// TIA Portal V17 export
// export: Created 2025-03-07T09:17:32.1063252Z, ExportSetting WithDefaults, DisplayName Totally Integrated Automation Portal, DisplayVersion V17 Update 8, DisplayName TIA Portal Openness, DisplayVersion V17 Update 8, DisplayName TIA Portal Version Control Interface, DisplayVersion V17, DisplayName SINAMICS Startdrive Advanced, DisplayVersion V17 SP2, DisplayName SINAMICS Startdrive G110M, G120, G120C, G120D, G120P, G115D, DisplayVersion V17 SP2, DisplayName SINAMICS Startdrive G130, G150, S120, S150, SINAMICS MV, S210, DisplayVersion V17 SP2, DisplayName STEP 7 Professional, DisplayVersion V17 Update 8, DisplayName SINUMERIK ONE STEP 7 Toolbox, DisplayVersion V17 Update 12, DisplayName SINUMERIK 840D sl STEP 7 Toolbox, DisplayVersion V17 Update 12, DisplayName STEP 7 Safety, DisplayVersion V17 Update 6, DisplayName WinCC Advanced, DisplayVersion V17 Update 8
FUNCTION "FC372_NCK_M_CH9_SPARE" : Void   // FC372, LAD
TITLE = Channel 1 data
{ S7_Optimized_Access := 'FALSE' }
AUTHOR : ETXETAR
VERSION : 1.0
// stored: AutoNumber false, IsIECCheckEnabled false, SetENOAutomatically false, UDAEnableTagReadback false
BEGIN

REGION Network 1: ACKNOWLEDGE M400-FIXTURE 1 CLAMP SEQUENCE (READ-IN DISABLE) / ACKNOWLEDGE M100-CLAMP SEQUENCE FIXTURE 1
   // NOTE: WHEN THERE IS NOT INDEXING TABLE AVAILABLE IN THE MACHINE DELETE 
   // DB2171.DBX5.0 AND DB2171.DBX2.0
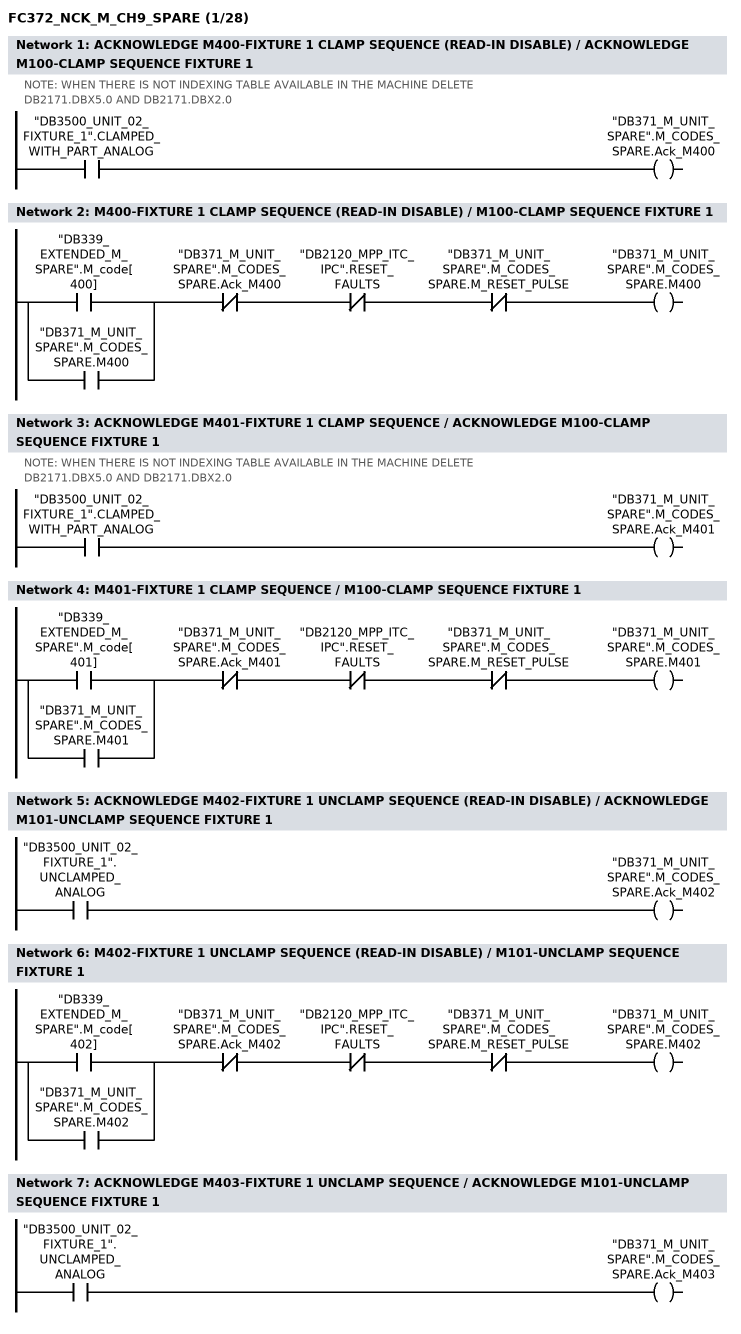
   RUNG wire#powerrail
      Contact( "DB3500_UNIT_02_FIXTURE_1".CLAMPED_WITH_PART_ANALOG )
      Coil( "DB371_M_UNIT_SPARE".M_CODES_SPARE.Ack_M400 )
   END_RUNG
   // the same network as SCL:
   "DB371_M_UNIT_SPARE".M_CODES_SPARE.Ack_M400 := "DB3500_UNIT_02_FIXTURE_1".CLAMPED_WITH_PART_ANALOG;
END_REGION

REGION Network 2: M400-FIXTURE 1 CLAMP SEQUENCE (READ-IN DISABLE) / M100-CLAMP SEQUENCE FIXTURE 1
   RUNG wire#powerrail
      Contact( "DB339_EXTENDED_M_SPARE".M_code[400] )
      wire#w1
      I_Contact( "DB371_M_UNIT_SPARE".M_CODES_SPARE.Ack_M400 )
      I_Contact( "DB2120_MPP_ITC_IPC".RESET_FAULTS )
      I_Contact( "DB371_M_UNIT_SPARE".M_CODES_SPARE.M_RESET_PULSE )
      Coil( "DB371_M_UNIT_SPARE".M_CODES_SPARE.M400 )
   END_RUNG
   RUNG wire#powerrail
      Contact( "DB371_M_UNIT_SPARE".M_CODES_SPARE.M400 )
   END_RUNG wire#w1
   // the same network as SCL:
   "DB371_M_UNIT_SPARE".M_CODES_SPARE.M400 := ("DB339_EXTENDED_M_SPARE".M_code[400] OR "DB371_M_UNIT_SPARE".M_CODES_SPARE.M400) AND NOT "DB371_M_UNIT_SPARE".M_CODES_SPARE.Ack_M400 AND NOT "DB2120_MPP_ITC_IPC".RESET_FAULTS AND NOT "DB371_M_UNIT_SPARE".M_CODES_SPARE.M_RESET_PULSE;
END_REGION

REGION Network 3: ACKNOWLEDGE M401-FIXTURE 1 CLAMP SEQUENCE / ACKNOWLEDGE M100-CLAMP SEQUENCE FIXTURE 1
   // NOTE: WHEN THERE IS NOT INDEXING TABLE AVAILABLE IN THE MACHINE DELETE 
   // DB2171.DBX5.0 AND DB2171.DBX2.0
   RUNG wire#powerrail
      Contact( "DB3500_UNIT_02_FIXTURE_1".CLAMPED_WITH_PART_ANALOG )
      Coil( "DB371_M_UNIT_SPARE".M_CODES_SPARE.Ack_M401 )
   END_RUNG
   // the same network as SCL:
   "DB371_M_UNIT_SPARE".M_CODES_SPARE.Ack_M401 := "DB3500_UNIT_02_FIXTURE_1".CLAMPED_WITH_PART_ANALOG;
END_REGION

REGION Network 4: M401-FIXTURE 1 CLAMP SEQUENCE / M100-CLAMP SEQUENCE FIXTURE 1
   RUNG wire#powerrail
      Contact( "DB339_EXTENDED_M_SPARE".M_code[401] )
      wire#w1
      I_Contact( "DB371_M_UNIT_SPARE".M_CODES_SPARE.Ack_M401 )
      I_Contact( "DB2120_MPP_ITC_IPC".RESET_FAULTS )
      I_Contact( "DB371_M_UNIT_SPARE".M_CODES_SPARE.M_RESET_PULSE )
      Coil( "DB371_M_UNIT_SPARE".M_CODES_SPARE.M401 )
   END_RUNG
   RUNG wire#powerrail
      Contact( "DB371_M_UNIT_SPARE".M_CODES_SPARE.M401 )
   END_RUNG wire#w1
   // the same network as SCL:
   "DB371_M_UNIT_SPARE".M_CODES_SPARE.M401 := ("DB339_EXTENDED_M_SPARE".M_code[401] OR "DB371_M_UNIT_SPARE".M_CODES_SPARE.M401) AND NOT "DB371_M_UNIT_SPARE".M_CODES_SPARE.Ack_M401 AND NOT "DB2120_MPP_ITC_IPC".RESET_FAULTS AND NOT "DB371_M_UNIT_SPARE".M_CODES_SPARE.M_RESET_PULSE;
END_REGION

REGION Network 5: ACKNOWLEDGE M402-FIXTURE 1 UNCLAMP SEQUENCE (READ-IN DISABLE) / ACKNOWLEDGE M101-UNCLAMP SEQUENCE FIXTURE 1
   RUNG wire#powerrail
      Contact( "DB3500_UNIT_02_FIXTURE_1".UNCLAMPED_ANALOG )
      Coil( "DB371_M_UNIT_SPARE".M_CODES_SPARE.Ack_M402 )
   END_RUNG
   // the same network as SCL:
   "DB371_M_UNIT_SPARE".M_CODES_SPARE.Ack_M402 := "DB3500_UNIT_02_FIXTURE_1".UNCLAMPED_ANALOG;
END_REGION

REGION Network 6: M402-FIXTURE 1 UNCLAMP SEQUENCE (READ-IN DISABLE) / M101-UNCLAMP SEQUENCE FIXTURE 1
   RUNG wire#powerrail
      Contact( "DB339_EXTENDED_M_SPARE".M_code[402] )
      wire#w1
      I_Contact( "DB371_M_UNIT_SPARE".M_CODES_SPARE.Ack_M402 )
      I_Contact( "DB2120_MPP_ITC_IPC".RESET_FAULTS )
      I_Contact( "DB371_M_UNIT_SPARE".M_CODES_SPARE.M_RESET_PULSE )
      Coil( "DB371_M_UNIT_SPARE".M_CODES_SPARE.M402 )
   END_RUNG
   RUNG wire#powerrail
      Contact( "DB371_M_UNIT_SPARE".M_CODES_SPARE.M402 )
   END_RUNG wire#w1
   // the same network as SCL:
   "DB371_M_UNIT_SPARE".M_CODES_SPARE.M402 := ("DB339_EXTENDED_M_SPARE".M_code[402] OR "DB371_M_UNIT_SPARE".M_CODES_SPARE.M402) AND NOT "DB371_M_UNIT_SPARE".M_CODES_SPARE.Ack_M402 AND NOT "DB2120_MPP_ITC_IPC".RESET_FAULTS AND NOT "DB371_M_UNIT_SPARE".M_CODES_SPARE.M_RESET_PULSE;
END_REGION

REGION Network 7: ACKNOWLEDGE M403-FIXTURE 1 UNCLAMP SEQUENCE / ACKNOWLEDGE M101-UNCLAMP SEQUENCE FIXTURE 1
   RUNG wire#powerrail
      Contact( "DB3500_UNIT_02_FIXTURE_1".UNCLAMPED_ANALOG )
      Coil( "DB371_M_UNIT_SPARE".M_CODES_SPARE.Ack_M403 )
   END_RUNG
   // the same network as SCL:
   "DB371_M_UNIT_SPARE".M_CODES_SPARE.Ack_M403 := "DB3500_UNIT_02_FIXTURE_1".UNCLAMPED_ANALOG;
END_REGION

REGION Network 8: M403-FIXTURE 1 UNCLAMP SEQUENCE / M101-UNCLAMP SEQUENCE FIXTURE 1
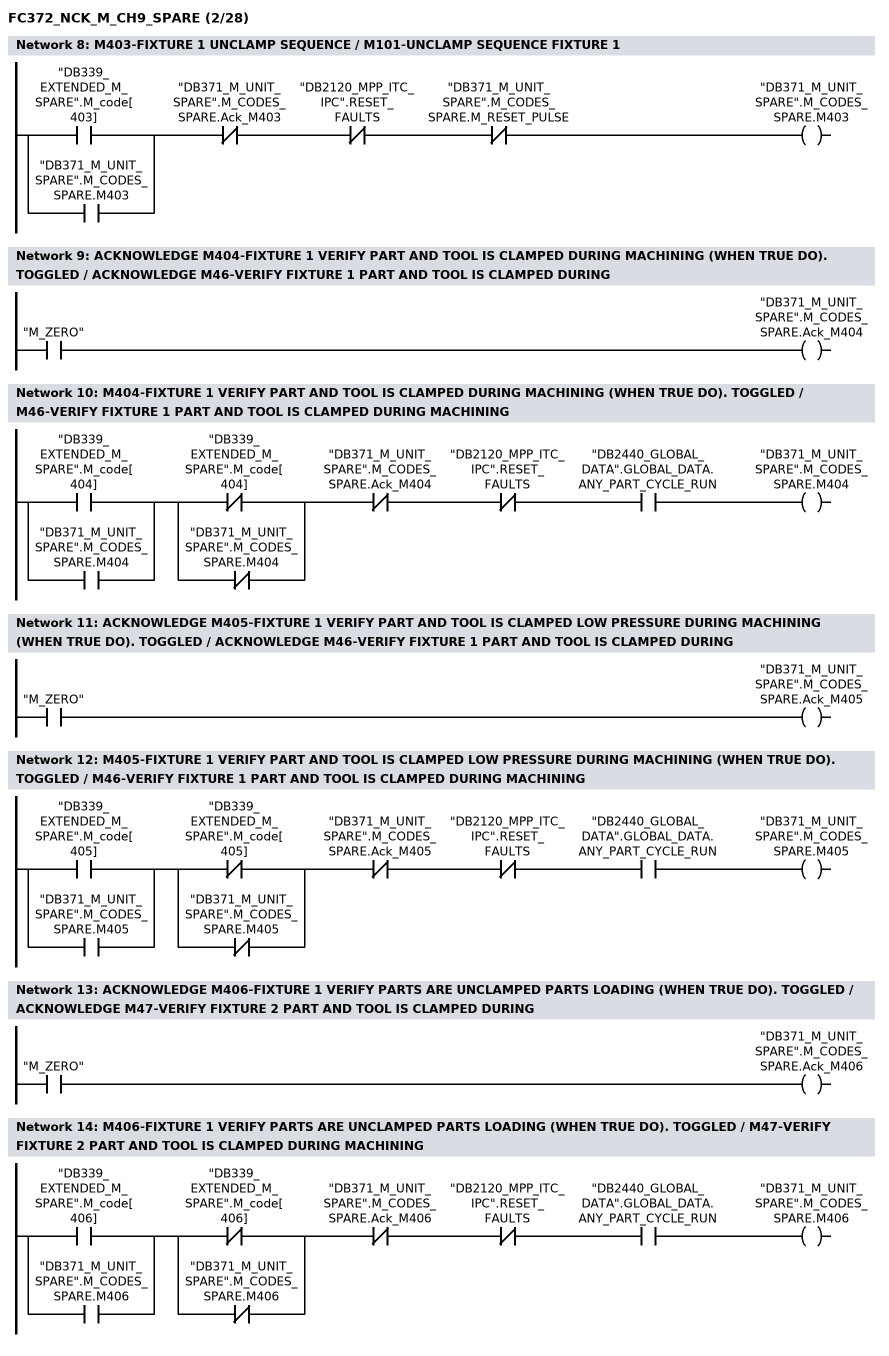
   RUNG wire#powerrail
      Contact( "DB339_EXTENDED_M_SPARE".M_code[403] )
      wire#w1
      I_Contact( "DB371_M_UNIT_SPARE".M_CODES_SPARE.Ack_M403 )
      I_Contact( "DB2120_MPP_ITC_IPC".RESET_FAULTS )
      I_Contact( "DB371_M_UNIT_SPARE".M_CODES_SPARE.M_RESET_PULSE )
      Coil( "DB371_M_UNIT_SPARE".M_CODES_SPARE.M403 )
   END_RUNG
   RUNG wire#powerrail
      Contact( "DB371_M_UNIT_SPARE".M_CODES_SPARE.M403 )
   END_RUNG wire#w1
   // the same network as SCL:
   "DB371_M_UNIT_SPARE".M_CODES_SPARE.M403 := ("DB339_EXTENDED_M_SPARE".M_code[403] OR "DB371_M_UNIT_SPARE".M_CODES_SPARE.M403) AND NOT "DB371_M_UNIT_SPARE".M_CODES_SPARE.Ack_M403 AND NOT "DB2120_MPP_ITC_IPC".RESET_FAULTS AND NOT "DB371_M_UNIT_SPARE".M_CODES_SPARE.M_RESET_PULSE;
END_REGION

REGION Network 9: ACKNOWLEDGE M404-FIXTURE 1 VERIFY PART AND TOOL IS CLAMPED DURING MACHINING (WHEN TRUE DO). TOGGLED / ACKNOWLEDGE M46-VERIFY FIXTURE 1 PART AND TOOL IS CLAMPED DURING
   RUNG wire#powerrail
      Contact( "M_ZERO" )
      Coil( "DB371_M_UNIT_SPARE".M_CODES_SPARE.Ack_M404 )
   END_RUNG
   // the same network as SCL:
   "DB371_M_UNIT_SPARE".M_CODES_SPARE.Ack_M404 := "M_ZERO";
END_REGION

REGION Network 10: M404-FIXTURE 1 VERIFY PART AND TOOL IS CLAMPED DURING MACHINING (WHEN TRUE DO). TOGGLED / M46-VERIFY FIXTURE 1 PART AND TOOL IS CLAMPED DURING MACHINING
   RUNG wire#powerrail
      Contact( "DB339_EXTENDED_M_SPARE".M_code[404] )
      wire#w1
      I_Contact( "DB339_EXTENDED_M_SPARE".M_code[404] )
      wire#w2
      I_Contact( "DB371_M_UNIT_SPARE".M_CODES_SPARE.Ack_M404 )
      I_Contact( "DB2120_MPP_ITC_IPC".RESET_FAULTS )
      Contact( "DB2440_GLOBAL_DATA".GLOBAL_DATA.ANY_PART_CYCLE_RUN )
      Coil( "DB371_M_UNIT_SPARE".M_CODES_SPARE.M404 )
   END_RUNG
   RUNG wire#powerrail
      Contact( "DB371_M_UNIT_SPARE".M_CODES_SPARE.M404 )
   END_RUNG wire#w1
   RUNG wire#w1
      I_Contact( "DB371_M_UNIT_SPARE".M_CODES_SPARE.M404 )
   END_RUNG wire#w2
   // the same network as SCL:
   "DB371_M_UNIT_SPARE".M_CODES_SPARE.M404 := ("DB339_EXTENDED_M_SPARE".M_code[404] OR "DB371_M_UNIT_SPARE".M_CODES_SPARE.M404) AND (NOT "DB339_EXTENDED_M_SPARE".M_code[404] OR NOT "DB371_M_UNIT_SPARE".M_CODES_SPARE.M404) AND NOT "DB371_M_UNIT_SPARE".M_CODES_SPARE.Ack_M404 AND NOT "DB2120_MPP_ITC_IPC".RESET_FAULTS AND "DB2440_GLOBAL_DATA".GLOBAL_DATA.ANY_PART_CYCLE_RUN;
END_REGION

REGION Network 11: ACKNOWLEDGE M405-FIXTURE 1 VERIFY PART AND TOOL IS CLAMPED LOW PRESSURE DURING MACHINING (WHEN TRUE DO). TOGGLED / ACKNOWLEDGE M46-VERIFY FIXTURE 1 PART AND TOOL IS CLAMPED DURING
   RUNG wire#powerrail
      Contact( "M_ZERO" )
      Coil( "DB371_M_UNIT_SPARE".M_CODES_SPARE.Ack_M405 )
   END_RUNG
   // the same network as SCL:
   "DB371_M_UNIT_SPARE".M_CODES_SPARE.Ack_M405 := "M_ZERO";
END_REGION

REGION Network 12: M405-FIXTURE 1 VERIFY PART AND TOOL IS CLAMPED LOW PRESSURE DURING MACHINING (WHEN TRUE DO). TOGGLED / M46-VERIFY FIXTURE 1 PART AND TOOL IS CLAMPED DURING MACHINING
   RUNG wire#powerrail
      Contact( "DB339_EXTENDED_M_SPARE".M_code[405] )
      wire#w1
      I_Contact( "DB339_EXTENDED_M_SPARE".M_code[405] )
      wire#w2
      I_Contact( "DB371_M_UNIT_SPARE".M_CODES_SPARE.Ack_M405 )
      I_Contact( "DB2120_MPP_ITC_IPC".RESET_FAULTS )
      Contact( "DB2440_GLOBAL_DATA".GLOBAL_DATA.ANY_PART_CYCLE_RUN )
      Coil( "DB371_M_UNIT_SPARE".M_CODES_SPARE.M405 )
   END_RUNG
   RUNG wire#powerrail
      Contact( "DB371_M_UNIT_SPARE".M_CODES_SPARE.M405 )
   END_RUNG wire#w1
   RUNG wire#w1
      I_Contact( "DB371_M_UNIT_SPARE".M_CODES_SPARE.M405 )
   END_RUNG wire#w2
   // the same network as SCL:
   "DB371_M_UNIT_SPARE".M_CODES_SPARE.M405 := ("DB339_EXTENDED_M_SPARE".M_code[405] OR "DB371_M_UNIT_SPARE".M_CODES_SPARE.M405) AND (NOT "DB339_EXTENDED_M_SPARE".M_code[405] OR NOT "DB371_M_UNIT_SPARE".M_CODES_SPARE.M405) AND NOT "DB371_M_UNIT_SPARE".M_CODES_SPARE.Ack_M405 AND NOT "DB2120_MPP_ITC_IPC".RESET_FAULTS AND "DB2440_GLOBAL_DATA".GLOBAL_DATA.ANY_PART_CYCLE_RUN;
END_REGION

REGION Network 13: ACKNOWLEDGE M406-FIXTURE 1 VERIFY PARTS ARE UNCLAMPED PARTS LOADING (WHEN TRUE DO). TOGGLED / ACKNOWLEDGE M47-VERIFY FIXTURE 2 PART AND TOOL IS CLAMPED DURING
   RUNG wire#powerrail
      Contact( "M_ZERO" )
      Coil( "DB371_M_UNIT_SPARE".M_CODES_SPARE.Ack_M406 )
   END_RUNG
   // the same network as SCL:
   "DB371_M_UNIT_SPARE".M_CODES_SPARE.Ack_M406 := "M_ZERO";
END_REGION

REGION Network 14: M406-FIXTURE 1 VERIFY PARTS ARE UNCLAMPED PARTS LOADING (WHEN TRUE DO). TOGGLED / M47-VERIFY FIXTURE 2 PART AND TOOL IS CLAMPED DURING MACHINING
   RUNG wire#powerrail
      Contact( "DB339_EXTENDED_M_SPARE".M_code[406] )
      wire#w1
      I_Contact( "DB339_EXTENDED_M_SPARE".M_code[406] )
      wire#w2
      I_Contact( "DB371_M_UNIT_SPARE".M_CODES_SPARE.Ack_M406 )
      I_Contact( "DB2120_MPP_ITC_IPC".RESET_FAULTS )
      Contact( "DB2440_GLOBAL_DATA".GLOBAL_DATA.ANY_PART_CYCLE_RUN )
      Coil( "DB371_M_UNIT_SPARE".M_CODES_SPARE.M406 )
   END_RUNG
   RUNG wire#powerrail
      Contact( "DB371_M_UNIT_SPARE".M_CODES_SPARE.M406 )
   END_RUNG wire#w1
   RUNG wire#w1
      I_Contact( "DB371_M_UNIT_SPARE".M_CODES_SPARE.M406 )
   END_RUNG wire#w2
   // the same network as SCL:
   "DB371_M_UNIT_SPARE".M_CODES_SPARE.M406 := ("DB339_EXTENDED_M_SPARE".M_code[406] OR "DB371_M_UNIT_SPARE".M_CODES_SPARE.M406) AND (NOT "DB339_EXTENDED_M_SPARE".M_code[406] OR NOT "DB371_M_UNIT_SPARE".M_CODES_SPARE.M406) AND NOT "DB371_M_UNIT_SPARE".M_CODES_SPARE.Ack_M406 AND NOT "DB2120_MPP_ITC_IPC".RESET_FAULTS AND "DB2440_GLOBAL_DATA".GLOBAL_DATA.ANY_PART_CYCLE_RUN;
END_REGION

REGION Network 15: ACKNOWLEDGE M407-FIXTURE 1 VERIFY FIXTURE REMAINS CLAMPED
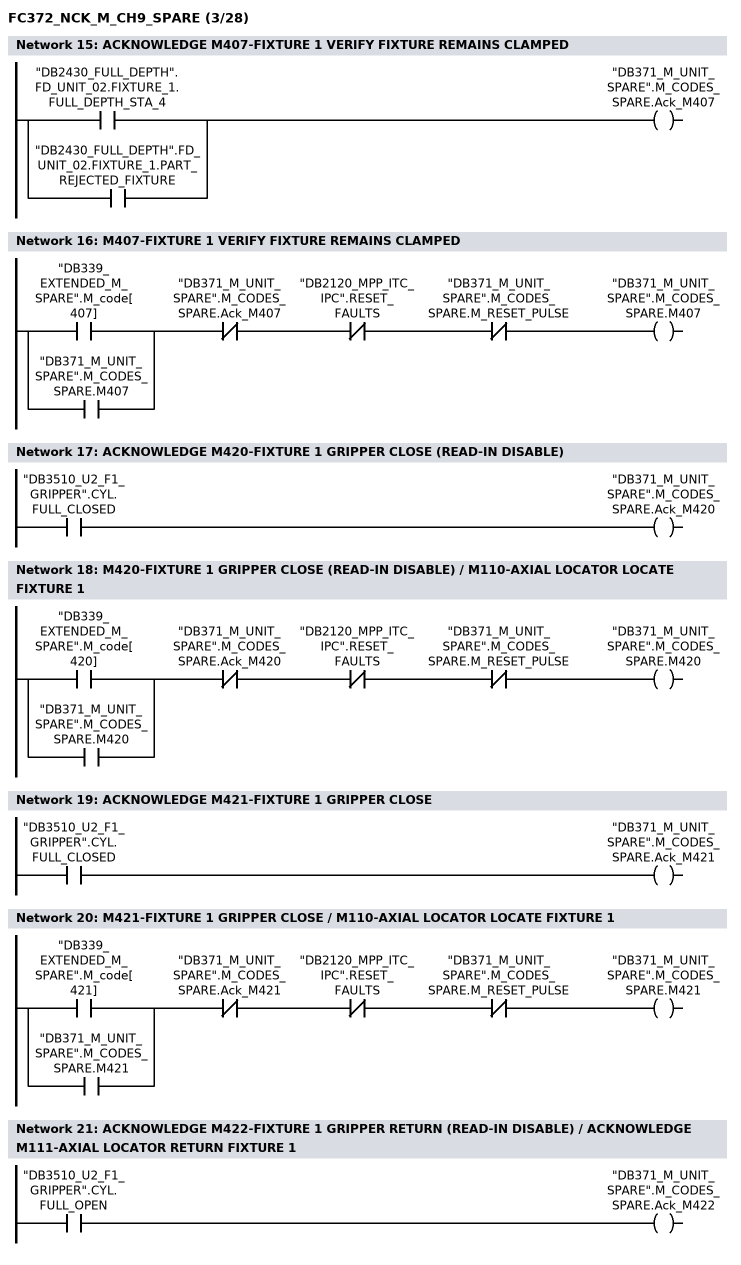
   RUNG wire#powerrail
      Contact( "DB2430_FULL_DEPTH".FD_UNIT_02.FIXTURE_1.FULL_DEPTH_STA_4 )
      wire#w1
      Coil( "DB371_M_UNIT_SPARE".M_CODES_SPARE.Ack_M407 )
   END_RUNG
   RUNG wire#powerrail
      Contact( "DB2430_FULL_DEPTH".FD_UNIT_02.FIXTURE_1.PART_REJECTED_FIXTURE )
   END_RUNG wire#w1
   // the same network as SCL:
   "DB371_M_UNIT_SPARE".M_CODES_SPARE.Ack_M407 := "DB2430_FULL_DEPTH".FD_UNIT_02.FIXTURE_1.FULL_DEPTH_STA_4 OR "DB2430_FULL_DEPTH".FD_UNIT_02.FIXTURE_1.PART_REJECTED_FIXTURE;
END_REGION

REGION Network 16: M407-FIXTURE 1 VERIFY FIXTURE REMAINS CLAMPED
   RUNG wire#powerrail
      Contact( "DB339_EXTENDED_M_SPARE".M_code[407] )
      wire#w1
      I_Contact( "DB371_M_UNIT_SPARE".M_CODES_SPARE.Ack_M407 )
      I_Contact( "DB2120_MPP_ITC_IPC".RESET_FAULTS )
      I_Contact( "DB371_M_UNIT_SPARE".M_CODES_SPARE.M_RESET_PULSE )
      Coil( "DB371_M_UNIT_SPARE".M_CODES_SPARE.M407 )
   END_RUNG
   RUNG wire#powerrail
      Contact( "DB371_M_UNIT_SPARE".M_CODES_SPARE.M407 )
   END_RUNG wire#w1
   // the same network as SCL:
   "DB371_M_UNIT_SPARE".M_CODES_SPARE.M407 := ("DB339_EXTENDED_M_SPARE".M_code[407] OR "DB371_M_UNIT_SPARE".M_CODES_SPARE.M407) AND NOT "DB371_M_UNIT_SPARE".M_CODES_SPARE.Ack_M407 AND NOT "DB2120_MPP_ITC_IPC".RESET_FAULTS AND NOT "DB371_M_UNIT_SPARE".M_CODES_SPARE.M_RESET_PULSE;
END_REGION

REGION Network 17: ACKNOWLEDGE M420-FIXTURE 1 GRIPPER CLOSE (READ-IN DISABLE)
   RUNG wire#powerrail
      Contact( "DB3510_U2_F1_GRIPPER".CYL.FULL_CLOSED )
      Coil( "DB371_M_UNIT_SPARE".M_CODES_SPARE.Ack_M420 )
   END_RUNG
   // the same network as SCL:
   "DB371_M_UNIT_SPARE".M_CODES_SPARE.Ack_M420 := "DB3510_U2_F1_GRIPPER".CYL.FULL_CLOSED;
END_REGION

REGION Network 18: M420-FIXTURE 1 GRIPPER CLOSE (READ-IN DISABLE) / M110-AXIAL LOCATOR LOCATE FIXTURE 1
   RUNG wire#powerrail
      Contact( "DB339_EXTENDED_M_SPARE".M_code[420] )
      wire#w1
      I_Contact( "DB371_M_UNIT_SPARE".M_CODES_SPARE.Ack_M420 )
      I_Contact( "DB2120_MPP_ITC_IPC".RESET_FAULTS )
      I_Contact( "DB371_M_UNIT_SPARE".M_CODES_SPARE.M_RESET_PULSE )
      Coil( "DB371_M_UNIT_SPARE".M_CODES_SPARE.M420 )
   END_RUNG
   RUNG wire#powerrail
      Contact( "DB371_M_UNIT_SPARE".M_CODES_SPARE.M420 )
   END_RUNG wire#w1
   // the same network as SCL:
   "DB371_M_UNIT_SPARE".M_CODES_SPARE.M420 := ("DB339_EXTENDED_M_SPARE".M_code[420] OR "DB371_M_UNIT_SPARE".M_CODES_SPARE.M420) AND NOT "DB371_M_UNIT_SPARE".M_CODES_SPARE.Ack_M420 AND NOT "DB2120_MPP_ITC_IPC".RESET_FAULTS AND NOT "DB371_M_UNIT_SPARE".M_CODES_SPARE.M_RESET_PULSE;
END_REGION

REGION Network 19: ACKNOWLEDGE M421-FIXTURE 1 GRIPPER CLOSE
   RUNG wire#powerrail
      Contact( "DB3510_U2_F1_GRIPPER".CYL.FULL_CLOSED )
      Coil( "DB371_M_UNIT_SPARE".M_CODES_SPARE.Ack_M421 )
   END_RUNG
   // the same network as SCL:
   "DB371_M_UNIT_SPARE".M_CODES_SPARE.Ack_M421 := "DB3510_U2_F1_GRIPPER".CYL.FULL_CLOSED;
END_REGION

REGION Network 20: M421-FIXTURE 1 GRIPPER CLOSE / M110-AXIAL LOCATOR LOCATE FIXTURE 1
   RUNG wire#powerrail
      Contact( "DB339_EXTENDED_M_SPARE".M_code[421] )
      wire#w1
      I_Contact( "DB371_M_UNIT_SPARE".M_CODES_SPARE.Ack_M421 )
      I_Contact( "DB2120_MPP_ITC_IPC".RESET_FAULTS )
      I_Contact( "DB371_M_UNIT_SPARE".M_CODES_SPARE.M_RESET_PULSE )
      Coil( "DB371_M_UNIT_SPARE".M_CODES_SPARE.M421 )
   END_RUNG
   RUNG wire#powerrail
      Contact( "DB371_M_UNIT_SPARE".M_CODES_SPARE.M421 )
   END_RUNG wire#w1
   // the same network as SCL:
   "DB371_M_UNIT_SPARE".M_CODES_SPARE.M421 := ("DB339_EXTENDED_M_SPARE".M_code[421] OR "DB371_M_UNIT_SPARE".M_CODES_SPARE.M421) AND NOT "DB371_M_UNIT_SPARE".M_CODES_SPARE.Ack_M421 AND NOT "DB2120_MPP_ITC_IPC".RESET_FAULTS AND NOT "DB371_M_UNIT_SPARE".M_CODES_SPARE.M_RESET_PULSE;
END_REGION

REGION Network 21: ACKNOWLEDGE M422-FIXTURE 1 GRIPPER RETURN (READ-IN DISABLE) / ACKNOWLEDGE M111-AXIAL LOCATOR RETURN FIXTURE 1
   RUNG wire#powerrail
      Contact( "DB3510_U2_F1_GRIPPER".CYL.FULL_OPEN )
      Coil( "DB371_M_UNIT_SPARE".M_CODES_SPARE.Ack_M422 )
   END_RUNG
   // the same network as SCL:
   "DB371_M_UNIT_SPARE".M_CODES_SPARE.Ack_M422 := "DB3510_U2_F1_GRIPPER".CYL.FULL_OPEN;
END_REGION

REGION Network 22: M422-FIXTURE 1 GRIPPER RETURN (READ-IN DISABLE) / M111-AXIAL LOCATOR RETURN FIXTURE 1
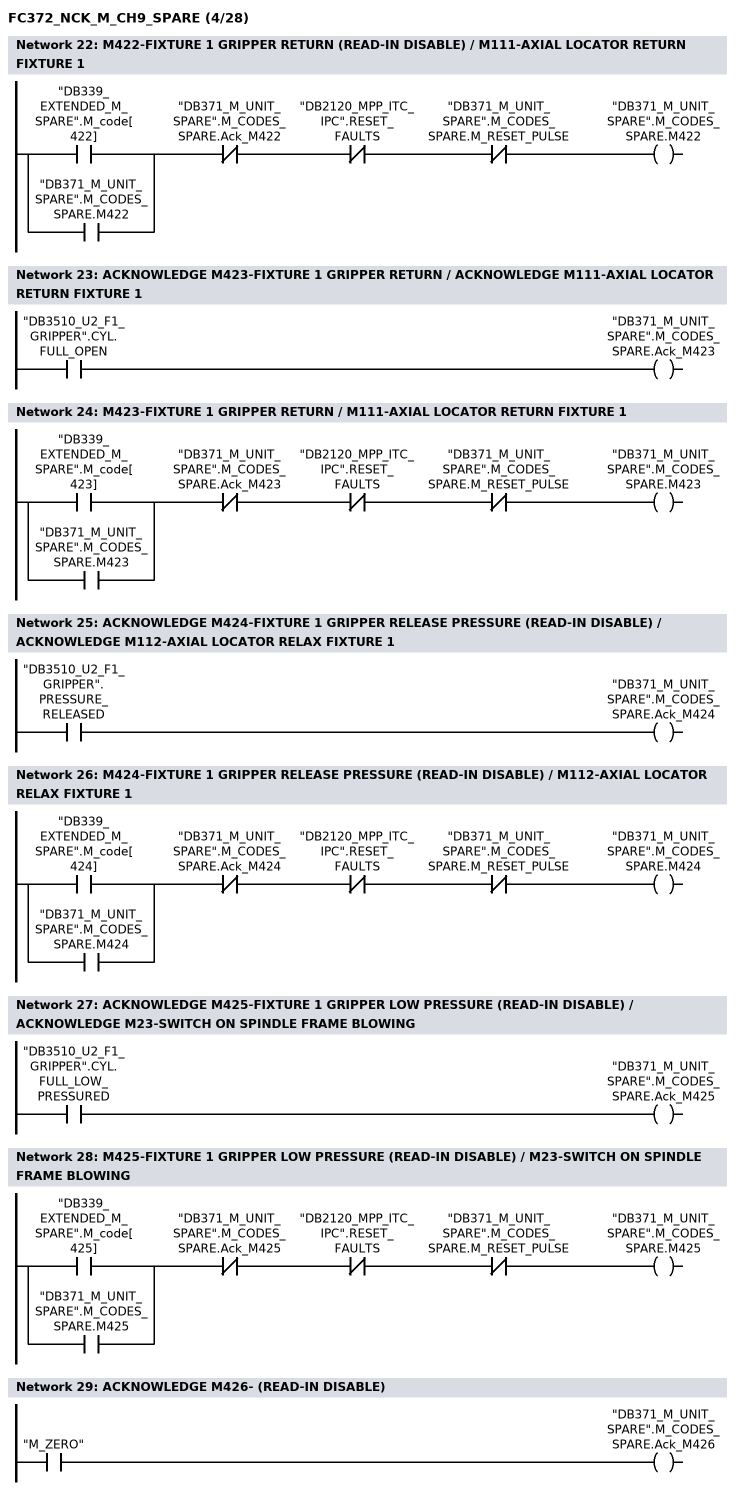
   RUNG wire#powerrail
      Contact( "DB339_EXTENDED_M_SPARE".M_code[422] )
      wire#w1
      I_Contact( "DB371_M_UNIT_SPARE".M_CODES_SPARE.Ack_M422 )
      I_Contact( "DB2120_MPP_ITC_IPC".RESET_FAULTS )
      I_Contact( "DB371_M_UNIT_SPARE".M_CODES_SPARE.M_RESET_PULSE )
      Coil( "DB371_M_UNIT_SPARE".M_CODES_SPARE.M422 )
   END_RUNG
   RUNG wire#powerrail
      Contact( "DB371_M_UNIT_SPARE".M_CODES_SPARE.M422 )
   END_RUNG wire#w1
   // the same network as SCL:
   "DB371_M_UNIT_SPARE".M_CODES_SPARE.M422 := ("DB339_EXTENDED_M_SPARE".M_code[422] OR "DB371_M_UNIT_SPARE".M_CODES_SPARE.M422) AND NOT "DB371_M_UNIT_SPARE".M_CODES_SPARE.Ack_M422 AND NOT "DB2120_MPP_ITC_IPC".RESET_FAULTS AND NOT "DB371_M_UNIT_SPARE".M_CODES_SPARE.M_RESET_PULSE;
END_REGION

REGION Network 23: ACKNOWLEDGE M423-FIXTURE 1 GRIPPER RETURN / ACKNOWLEDGE M111-AXIAL LOCATOR RETURN FIXTURE 1
   RUNG wire#powerrail
      Contact( "DB3510_U2_F1_GRIPPER".CYL.FULL_OPEN )
      Coil( "DB371_M_UNIT_SPARE".M_CODES_SPARE.Ack_M423 )
   END_RUNG
   // the same network as SCL:
   "DB371_M_UNIT_SPARE".M_CODES_SPARE.Ack_M423 := "DB3510_U2_F1_GRIPPER".CYL.FULL_OPEN;
END_REGION

REGION Network 24: M423-FIXTURE 1 GRIPPER RETURN / M111-AXIAL LOCATOR RETURN FIXTURE 1
   RUNG wire#powerrail
      Contact( "DB339_EXTENDED_M_SPARE".M_code[423] )
      wire#w1
      I_Contact( "DB371_M_UNIT_SPARE".M_CODES_SPARE.Ack_M423 )
      I_Contact( "DB2120_MPP_ITC_IPC".RESET_FAULTS )
      I_Contact( "DB371_M_UNIT_SPARE".M_CODES_SPARE.M_RESET_PULSE )
      Coil( "DB371_M_UNIT_SPARE".M_CODES_SPARE.M423 )
   END_RUNG
   RUNG wire#powerrail
      Contact( "DB371_M_UNIT_SPARE".M_CODES_SPARE.M423 )
   END_RUNG wire#w1
   // the same network as SCL:
   "DB371_M_UNIT_SPARE".M_CODES_SPARE.M423 := ("DB339_EXTENDED_M_SPARE".M_code[423] OR "DB371_M_UNIT_SPARE".M_CODES_SPARE.M423) AND NOT "DB371_M_UNIT_SPARE".M_CODES_SPARE.Ack_M423 AND NOT "DB2120_MPP_ITC_IPC".RESET_FAULTS AND NOT "DB371_M_UNIT_SPARE".M_CODES_SPARE.M_RESET_PULSE;
END_REGION

REGION Network 25: ACKNOWLEDGE M424-FIXTURE 1 GRIPPER RELEASE PRESSURE (READ-IN DISABLE) / ACKNOWLEDGE M112-AXIAL LOCATOR RELAX FIXTURE 1
   RUNG wire#powerrail
      Contact( "DB3510_U2_F1_GRIPPER".PRESSURE_RELEASED )
      Coil( "DB371_M_UNIT_SPARE".M_CODES_SPARE.Ack_M424 )
   END_RUNG
   // the same network as SCL:
   "DB371_M_UNIT_SPARE".M_CODES_SPARE.Ack_M424 := "DB3510_U2_F1_GRIPPER".PRESSURE_RELEASED;
END_REGION

REGION Network 26: M424-FIXTURE 1 GRIPPER RELEASE PRESSURE (READ-IN DISABLE) / M112-AXIAL LOCATOR RELAX FIXTURE 1
   RUNG wire#powerrail
      Contact( "DB339_EXTENDED_M_SPARE".M_code[424] )
      wire#w1
      I_Contact( "DB371_M_UNIT_SPARE".M_CODES_SPARE.Ack_M424 )
      I_Contact( "DB2120_MPP_ITC_IPC".RESET_FAULTS )
      I_Contact( "DB371_M_UNIT_SPARE".M_CODES_SPARE.M_RESET_PULSE )
      Coil( "DB371_M_UNIT_SPARE".M_CODES_SPARE.M424 )
   END_RUNG
   RUNG wire#powerrail
      Contact( "DB371_M_UNIT_SPARE".M_CODES_SPARE.M424 )
   END_RUNG wire#w1
   // the same network as SCL:
   "DB371_M_UNIT_SPARE".M_CODES_SPARE.M424 := ("DB339_EXTENDED_M_SPARE".M_code[424] OR "DB371_M_UNIT_SPARE".M_CODES_SPARE.M424) AND NOT "DB371_M_UNIT_SPARE".M_CODES_SPARE.Ack_M424 AND NOT "DB2120_MPP_ITC_IPC".RESET_FAULTS AND NOT "DB371_M_UNIT_SPARE".M_CODES_SPARE.M_RESET_PULSE;
END_REGION

REGION Network 27: ACKNOWLEDGE M425-FIXTURE 1 GRIPPER LOW PRESSURE (READ-IN DISABLE) / ACKNOWLEDGE M23-SWITCH ON SPINDLE FRAME BLOWING
   RUNG wire#powerrail
      Contact( "DB3510_U2_F1_GRIPPER".CYL.FULL_LOW_PRESSURED )
      Coil( "DB371_M_UNIT_SPARE".M_CODES_SPARE.Ack_M425 )
   END_RUNG
   // the same network as SCL:
   "DB371_M_UNIT_SPARE".M_CODES_SPARE.Ack_M425 := "DB3510_U2_F1_GRIPPER".CYL.FULL_LOW_PRESSURED;
END_REGION

REGION Network 28: M425-FIXTURE 1 GRIPPER LOW PRESSURE (READ-IN DISABLE) / M23-SWITCH ON SPINDLE FRAME BLOWING
   RUNG wire#powerrail
      Contact( "DB339_EXTENDED_M_SPARE".M_code[425] )
      wire#w1
      I_Contact( "DB371_M_UNIT_SPARE".M_CODES_SPARE.Ack_M425 )
      I_Contact( "DB2120_MPP_ITC_IPC".RESET_FAULTS )
      I_Contact( "DB371_M_UNIT_SPARE".M_CODES_SPARE.M_RESET_PULSE )
      Coil( "DB371_M_UNIT_SPARE".M_CODES_SPARE.M425 )
   END_RUNG
   RUNG wire#powerrail
      Contact( "DB371_M_UNIT_SPARE".M_CODES_SPARE.M425 )
   END_RUNG wire#w1
   // the same network as SCL:
   "DB371_M_UNIT_SPARE".M_CODES_SPARE.M425 := ("DB339_EXTENDED_M_SPARE".M_code[425] OR "DB371_M_UNIT_SPARE".M_CODES_SPARE.M425) AND NOT "DB371_M_UNIT_SPARE".M_CODES_SPARE.Ack_M425 AND NOT "DB2120_MPP_ITC_IPC".RESET_FAULTS AND NOT "DB371_M_UNIT_SPARE".M_CODES_SPARE.M_RESET_PULSE;
END_REGION

REGION Network 29: ACKNOWLEDGE M426- (READ-IN DISABLE)
   RUNG wire#powerrail
      Contact( "M_ZERO" )
      Coil( "DB371_M_UNIT_SPARE".M_CODES_SPARE.Ack_M426 )
   END_RUNG
   // the same network as SCL:
   "DB371_M_UNIT_SPARE".M_CODES_SPARE.Ack_M426 := "M_ZERO";
END_REGION

REGION Network 30: M426- (READ-IN DISABLE)
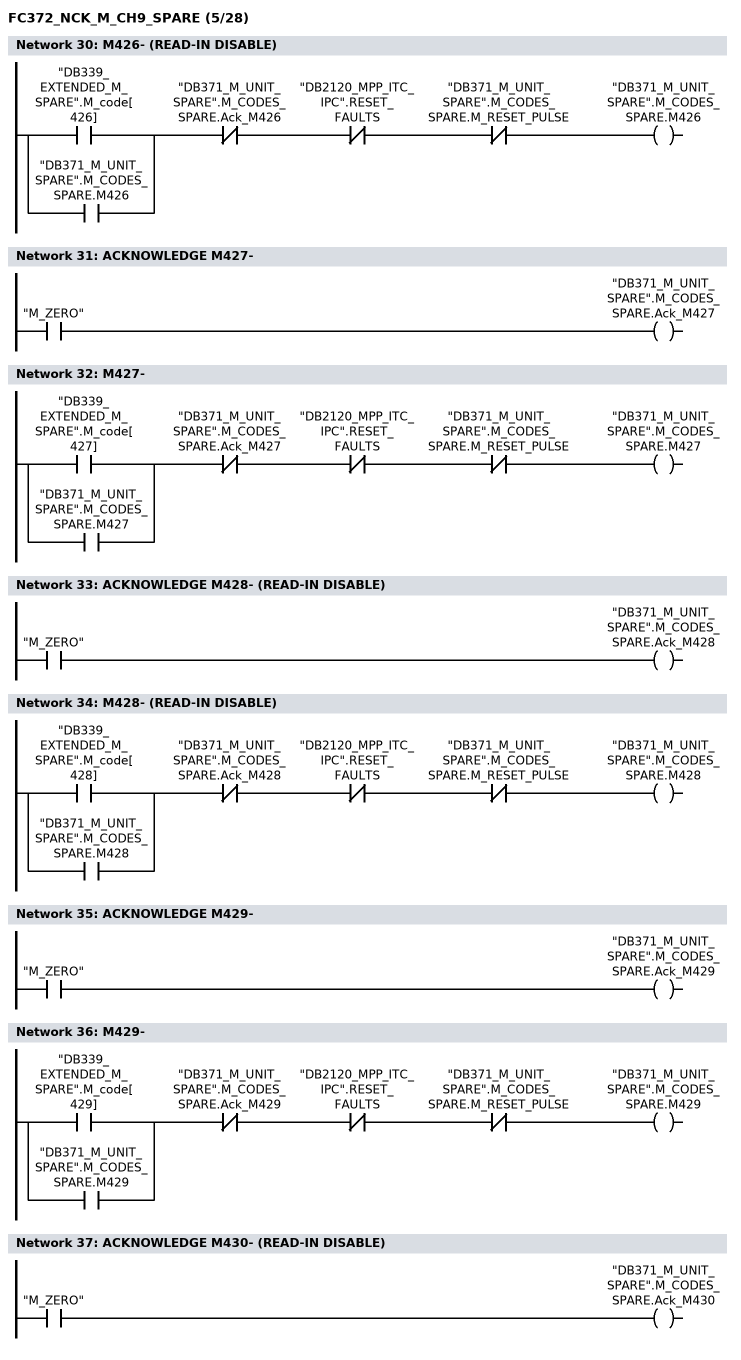
   RUNG wire#powerrail
      Contact( "DB339_EXTENDED_M_SPARE".M_code[426] )
      wire#w1
      I_Contact( "DB371_M_UNIT_SPARE".M_CODES_SPARE.Ack_M426 )
      I_Contact( "DB2120_MPP_ITC_IPC".RESET_FAULTS )
      I_Contact( "DB371_M_UNIT_SPARE".M_CODES_SPARE.M_RESET_PULSE )
      Coil( "DB371_M_UNIT_SPARE".M_CODES_SPARE.M426 )
   END_RUNG
   RUNG wire#powerrail
      Contact( "DB371_M_UNIT_SPARE".M_CODES_SPARE.M426 )
   END_RUNG wire#w1
   // the same network as SCL:
   "DB371_M_UNIT_SPARE".M_CODES_SPARE.M426 := ("DB339_EXTENDED_M_SPARE".M_code[426] OR "DB371_M_UNIT_SPARE".M_CODES_SPARE.M426) AND NOT "DB371_M_UNIT_SPARE".M_CODES_SPARE.Ack_M426 AND NOT "DB2120_MPP_ITC_IPC".RESET_FAULTS AND NOT "DB371_M_UNIT_SPARE".M_CODES_SPARE.M_RESET_PULSE;
END_REGION

REGION Network 31: ACKNOWLEDGE M427-
   RUNG wire#powerrail
      Contact( "M_ZERO" )
      Coil( "DB371_M_UNIT_SPARE".M_CODES_SPARE.Ack_M427 )
   END_RUNG
   // the same network as SCL:
   "DB371_M_UNIT_SPARE".M_CODES_SPARE.Ack_M427 := "M_ZERO";
END_REGION

REGION Network 32: M427-
   RUNG wire#powerrail
      Contact( "DB339_EXTENDED_M_SPARE".M_code[427] )
      wire#w1
      I_Contact( "DB371_M_UNIT_SPARE".M_CODES_SPARE.Ack_M427 )
      I_Contact( "DB2120_MPP_ITC_IPC".RESET_FAULTS )
      I_Contact( "DB371_M_UNIT_SPARE".M_CODES_SPARE.M_RESET_PULSE )
      Coil( "DB371_M_UNIT_SPARE".M_CODES_SPARE.M427 )
   END_RUNG
   RUNG wire#powerrail
      Contact( "DB371_M_UNIT_SPARE".M_CODES_SPARE.M427 )
   END_RUNG wire#w1
   // the same network as SCL:
   "DB371_M_UNIT_SPARE".M_CODES_SPARE.M427 := ("DB339_EXTENDED_M_SPARE".M_code[427] OR "DB371_M_UNIT_SPARE".M_CODES_SPARE.M427) AND NOT "DB371_M_UNIT_SPARE".M_CODES_SPARE.Ack_M427 AND NOT "DB2120_MPP_ITC_IPC".RESET_FAULTS AND NOT "DB371_M_UNIT_SPARE".M_CODES_SPARE.M_RESET_PULSE;
END_REGION

REGION Network 33: ACKNOWLEDGE M428- (READ-IN DISABLE)
   RUNG wire#powerrail
      Contact( "M_ZERO" )
      Coil( "DB371_M_UNIT_SPARE".M_CODES_SPARE.Ack_M428 )
   END_RUNG
   // the same network as SCL:
   "DB371_M_UNIT_SPARE".M_CODES_SPARE.Ack_M428 := "M_ZERO";
END_REGION

REGION Network 34: M428- (READ-IN DISABLE)
   RUNG wire#powerrail
      Contact( "DB339_EXTENDED_M_SPARE".M_code[428] )
      wire#w1
      I_Contact( "DB371_M_UNIT_SPARE".M_CODES_SPARE.Ack_M428 )
      I_Contact( "DB2120_MPP_ITC_IPC".RESET_FAULTS )
      I_Contact( "DB371_M_UNIT_SPARE".M_CODES_SPARE.M_RESET_PULSE )
      Coil( "DB371_M_UNIT_SPARE".M_CODES_SPARE.M428 )
   END_RUNG
   RUNG wire#powerrail
      Contact( "DB371_M_UNIT_SPARE".M_CODES_SPARE.M428 )
   END_RUNG wire#w1
   // the same network as SCL:
   "DB371_M_UNIT_SPARE".M_CODES_SPARE.M428 := ("DB339_EXTENDED_M_SPARE".M_code[428] OR "DB371_M_UNIT_SPARE".M_CODES_SPARE.M428) AND NOT "DB371_M_UNIT_SPARE".M_CODES_SPARE.Ack_M428 AND NOT "DB2120_MPP_ITC_IPC".RESET_FAULTS AND NOT "DB371_M_UNIT_SPARE".M_CODES_SPARE.M_RESET_PULSE;
END_REGION

REGION Network 35: ACKNOWLEDGE M429-
   RUNG wire#powerrail
      Contact( "M_ZERO" )
      Coil( "DB371_M_UNIT_SPARE".M_CODES_SPARE.Ack_M429 )
   END_RUNG
   // the same network as SCL:
   "DB371_M_UNIT_SPARE".M_CODES_SPARE.Ack_M429 := "M_ZERO";
END_REGION

REGION Network 36: M429-
   RUNG wire#powerrail
      Contact( "DB339_EXTENDED_M_SPARE".M_code[429] )
      wire#w1
      I_Contact( "DB371_M_UNIT_SPARE".M_CODES_SPARE.Ack_M429 )
      I_Contact( "DB2120_MPP_ITC_IPC".RESET_FAULTS )
      I_Contact( "DB371_M_UNIT_SPARE".M_CODES_SPARE.M_RESET_PULSE )
      Coil( "DB371_M_UNIT_SPARE".M_CODES_SPARE.M429 )
   END_RUNG
   RUNG wire#powerrail
      Contact( "DB371_M_UNIT_SPARE".M_CODES_SPARE.M429 )
   END_RUNG wire#w1
   // the same network as SCL:
   "DB371_M_UNIT_SPARE".M_CODES_SPARE.M429 := ("DB339_EXTENDED_M_SPARE".M_code[429] OR "DB371_M_UNIT_SPARE".M_CODES_SPARE.M429) AND NOT "DB371_M_UNIT_SPARE".M_CODES_SPARE.Ack_M429 AND NOT "DB2120_MPP_ITC_IPC".RESET_FAULTS AND NOT "DB371_M_UNIT_SPARE".M_CODES_SPARE.M_RESET_PULSE;
END_REGION

REGION Network 37: ACKNOWLEDGE M430- (READ-IN DISABLE)
   RUNG wire#powerrail
      Contact( "M_ZERO" )
      Coil( "DB371_M_UNIT_SPARE".M_CODES_SPARE.Ack_M430 )
   END_RUNG
   // the same network as SCL:
   "DB371_M_UNIT_SPARE".M_CODES_SPARE.Ack_M430 := "M_ZERO";
END_REGION

REGION Network 38: M430- (READ-IN DISABLE)
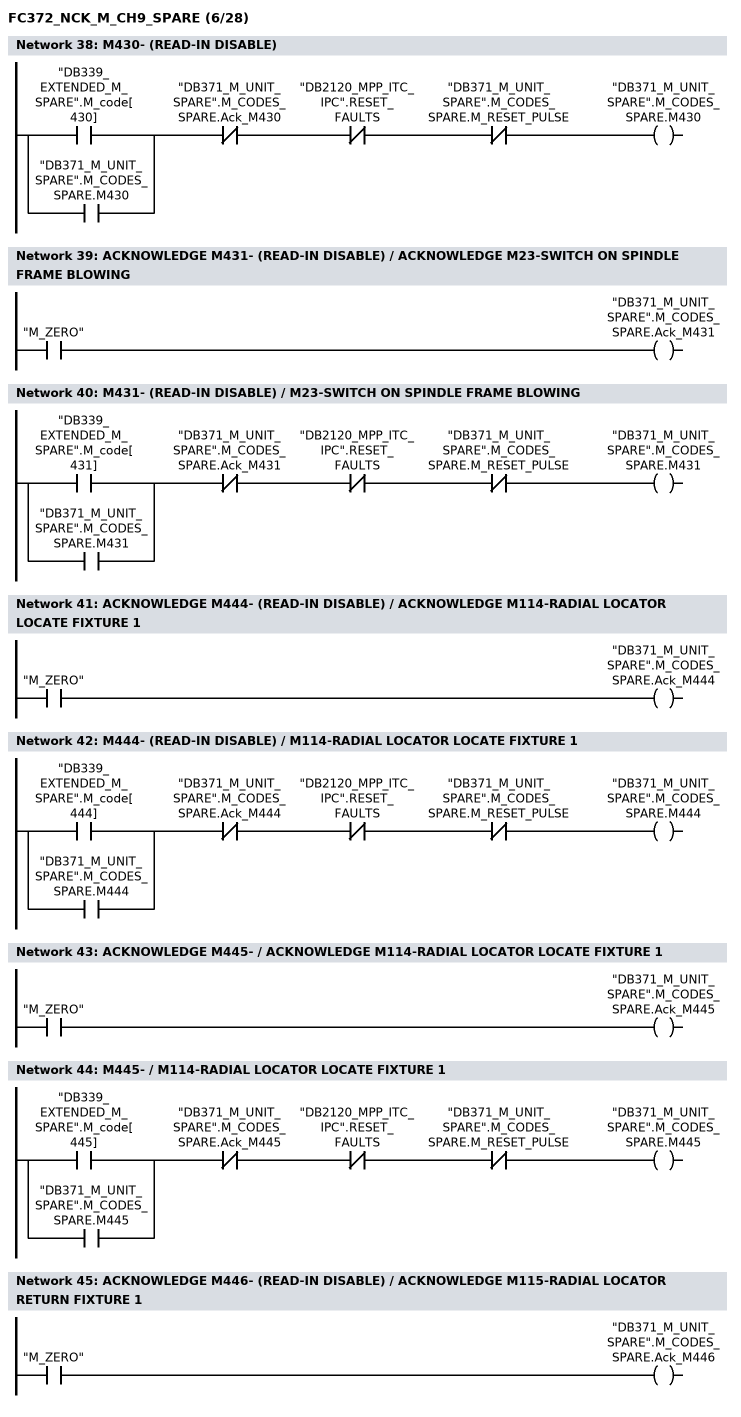
   RUNG wire#powerrail
      Contact( "DB339_EXTENDED_M_SPARE".M_code[430] )
      wire#w1
      I_Contact( "DB371_M_UNIT_SPARE".M_CODES_SPARE.Ack_M430 )
      I_Contact( "DB2120_MPP_ITC_IPC".RESET_FAULTS )
      I_Contact( "DB371_M_UNIT_SPARE".M_CODES_SPARE.M_RESET_PULSE )
      Coil( "DB371_M_UNIT_SPARE".M_CODES_SPARE.M430 )
   END_RUNG
   RUNG wire#powerrail
      Contact( "DB371_M_UNIT_SPARE".M_CODES_SPARE.M430 )
   END_RUNG wire#w1
   // the same network as SCL:
   "DB371_M_UNIT_SPARE".M_CODES_SPARE.M430 := ("DB339_EXTENDED_M_SPARE".M_code[430] OR "DB371_M_UNIT_SPARE".M_CODES_SPARE.M430) AND NOT "DB371_M_UNIT_SPARE".M_CODES_SPARE.Ack_M430 AND NOT "DB2120_MPP_ITC_IPC".RESET_FAULTS AND NOT "DB371_M_UNIT_SPARE".M_CODES_SPARE.M_RESET_PULSE;
END_REGION

REGION Network 39: ACKNOWLEDGE M431- (READ-IN DISABLE) / ACKNOWLEDGE M23-SWITCH ON SPINDLE FRAME BLOWING
   RUNG wire#powerrail
      Contact( "M_ZERO" )
      Coil( "DB371_M_UNIT_SPARE".M_CODES_SPARE.Ack_M431 )
   END_RUNG
   // the same network as SCL:
   "DB371_M_UNIT_SPARE".M_CODES_SPARE.Ack_M431 := "M_ZERO";
END_REGION

REGION Network 40: M431- (READ-IN DISABLE) / M23-SWITCH ON SPINDLE FRAME BLOWING
   RUNG wire#powerrail
      Contact( "DB339_EXTENDED_M_SPARE".M_code[431] )
      wire#w1
      I_Contact( "DB371_M_UNIT_SPARE".M_CODES_SPARE.Ack_M431 )
      I_Contact( "DB2120_MPP_ITC_IPC".RESET_FAULTS )
      I_Contact( "DB371_M_UNIT_SPARE".M_CODES_SPARE.M_RESET_PULSE )
      Coil( "DB371_M_UNIT_SPARE".M_CODES_SPARE.M431 )
   END_RUNG
   RUNG wire#powerrail
      Contact( "DB371_M_UNIT_SPARE".M_CODES_SPARE.M431 )
   END_RUNG wire#w1
   // the same network as SCL:
   "DB371_M_UNIT_SPARE".M_CODES_SPARE.M431 := ("DB339_EXTENDED_M_SPARE".M_code[431] OR "DB371_M_UNIT_SPARE".M_CODES_SPARE.M431) AND NOT "DB371_M_UNIT_SPARE".M_CODES_SPARE.Ack_M431 AND NOT "DB2120_MPP_ITC_IPC".RESET_FAULTS AND NOT "DB371_M_UNIT_SPARE".M_CODES_SPARE.M_RESET_PULSE;
END_REGION

REGION Network 41: ACKNOWLEDGE M444- (READ-IN DISABLE) / ACKNOWLEDGE M114-RADIAL LOCATOR LOCATE FIXTURE 1
   RUNG wire#powerrail
      Contact( "M_ZERO" )
      Coil( "DB371_M_UNIT_SPARE".M_CODES_SPARE.Ack_M444 )
   END_RUNG
   // the same network as SCL:
   "DB371_M_UNIT_SPARE".M_CODES_SPARE.Ack_M444 := "M_ZERO";
END_REGION

REGION Network 42: M444- (READ-IN DISABLE) / M114-RADIAL LOCATOR LOCATE FIXTURE 1
   RUNG wire#powerrail
      Contact( "DB339_EXTENDED_M_SPARE".M_code[444] )
      wire#w1
      I_Contact( "DB371_M_UNIT_SPARE".M_CODES_SPARE.Ack_M444 )
      I_Contact( "DB2120_MPP_ITC_IPC".RESET_FAULTS )
      I_Contact( "DB371_M_UNIT_SPARE".M_CODES_SPARE.M_RESET_PULSE )
      Coil( "DB371_M_UNIT_SPARE".M_CODES_SPARE.M444 )
   END_RUNG
   RUNG wire#powerrail
      Contact( "DB371_M_UNIT_SPARE".M_CODES_SPARE.M444 )
   END_RUNG wire#w1
   // the same network as SCL:
   "DB371_M_UNIT_SPARE".M_CODES_SPARE.M444 := ("DB339_EXTENDED_M_SPARE".M_code[444] OR "DB371_M_UNIT_SPARE".M_CODES_SPARE.M444) AND NOT "DB371_M_UNIT_SPARE".M_CODES_SPARE.Ack_M444 AND NOT "DB2120_MPP_ITC_IPC".RESET_FAULTS AND NOT "DB371_M_UNIT_SPARE".M_CODES_SPARE.M_RESET_PULSE;
END_REGION

REGION Network 43: ACKNOWLEDGE M445- / ACKNOWLEDGE M114-RADIAL LOCATOR LOCATE FIXTURE 1
   RUNG wire#powerrail
      Contact( "M_ZERO" )
      Coil( "DB371_M_UNIT_SPARE".M_CODES_SPARE.Ack_M445 )
   END_RUNG
   // the same network as SCL:
   "DB371_M_UNIT_SPARE".M_CODES_SPARE.Ack_M445 := "M_ZERO";
END_REGION

REGION Network 44: M445- / M114-RADIAL LOCATOR LOCATE FIXTURE 1
   RUNG wire#powerrail
      Contact( "DB339_EXTENDED_M_SPARE".M_code[445] )
      wire#w1
      I_Contact( "DB371_M_UNIT_SPARE".M_CODES_SPARE.Ack_M445 )
      I_Contact( "DB2120_MPP_ITC_IPC".RESET_FAULTS )
      I_Contact( "DB371_M_UNIT_SPARE".M_CODES_SPARE.M_RESET_PULSE )
      Coil( "DB371_M_UNIT_SPARE".M_CODES_SPARE.M445 )
   END_RUNG
   RUNG wire#powerrail
      Contact( "DB371_M_UNIT_SPARE".M_CODES_SPARE.M445 )
   END_RUNG wire#w1
   // the same network as SCL:
   "DB371_M_UNIT_SPARE".M_CODES_SPARE.M445 := ("DB339_EXTENDED_M_SPARE".M_code[445] OR "DB371_M_UNIT_SPARE".M_CODES_SPARE.M445) AND NOT "DB371_M_UNIT_SPARE".M_CODES_SPARE.Ack_M445 AND NOT "DB2120_MPP_ITC_IPC".RESET_FAULTS AND NOT "DB371_M_UNIT_SPARE".M_CODES_SPARE.M_RESET_PULSE;
END_REGION

REGION Network 45: ACKNOWLEDGE M446- (READ-IN DISABLE) / ACKNOWLEDGE M115-RADIAL LOCATOR RETURN FIXTURE 1
   RUNG wire#powerrail
      Contact( "M_ZERO" )
      Coil( "DB371_M_UNIT_SPARE".M_CODES_SPARE.Ack_M446 )
   END_RUNG
   // the same network as SCL:
   "DB371_M_UNIT_SPARE".M_CODES_SPARE.Ack_M446 := "M_ZERO";
END_REGION

REGION Network 46: M446- (READ-IN DISABLE) / M115-RADIAL LOCATOR RETURN FIXTURE 1
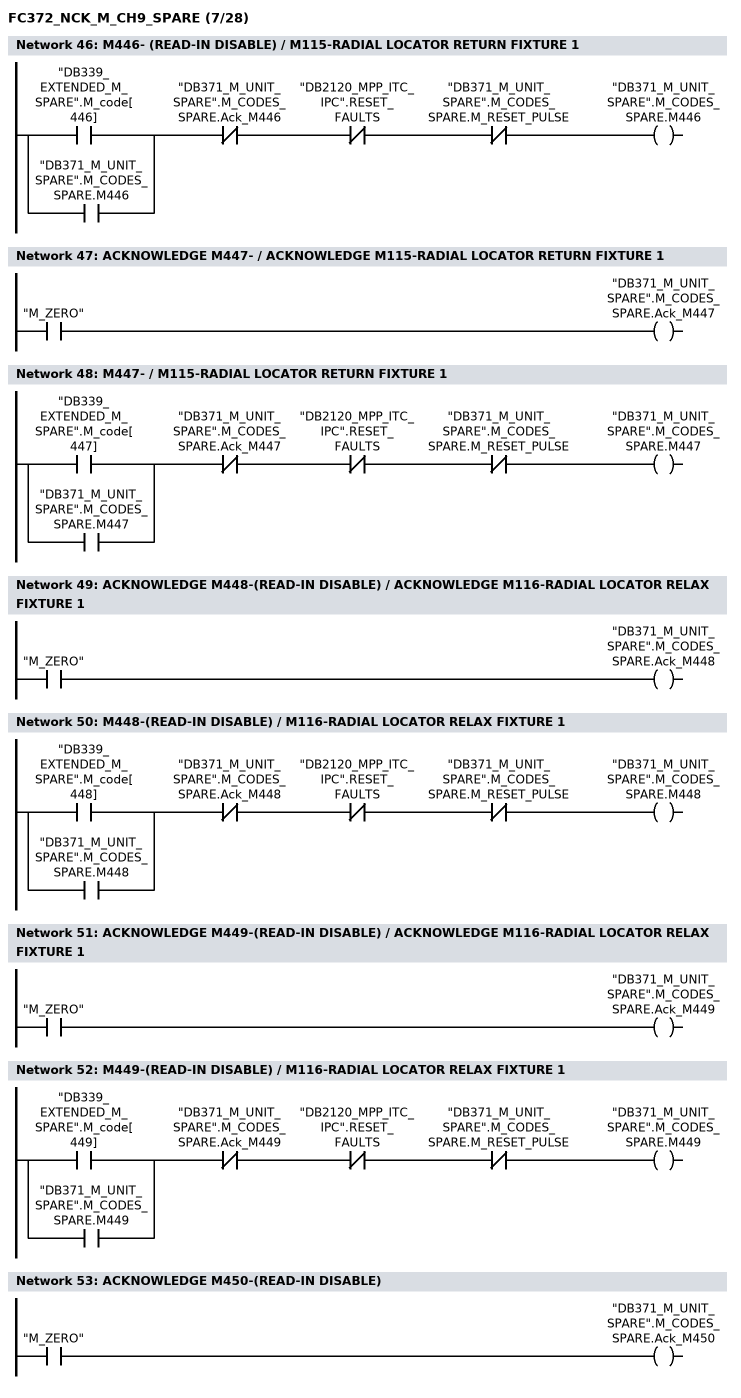
   RUNG wire#powerrail
      Contact( "DB339_EXTENDED_M_SPARE".M_code[446] )
      wire#w1
      I_Contact( "DB371_M_UNIT_SPARE".M_CODES_SPARE.Ack_M446 )
      I_Contact( "DB2120_MPP_ITC_IPC".RESET_FAULTS )
      I_Contact( "DB371_M_UNIT_SPARE".M_CODES_SPARE.M_RESET_PULSE )
      Coil( "DB371_M_UNIT_SPARE".M_CODES_SPARE.M446 )
   END_RUNG
   RUNG wire#powerrail
      Contact( "DB371_M_UNIT_SPARE".M_CODES_SPARE.M446 )
   END_RUNG wire#w1
   // the same network as SCL:
   "DB371_M_UNIT_SPARE".M_CODES_SPARE.M446 := ("DB339_EXTENDED_M_SPARE".M_code[446] OR "DB371_M_UNIT_SPARE".M_CODES_SPARE.M446) AND NOT "DB371_M_UNIT_SPARE".M_CODES_SPARE.Ack_M446 AND NOT "DB2120_MPP_ITC_IPC".RESET_FAULTS AND NOT "DB371_M_UNIT_SPARE".M_CODES_SPARE.M_RESET_PULSE;
END_REGION

REGION Network 47: ACKNOWLEDGE M447- / ACKNOWLEDGE M115-RADIAL LOCATOR RETURN FIXTURE 1
   RUNG wire#powerrail
      Contact( "M_ZERO" )
      Coil( "DB371_M_UNIT_SPARE".M_CODES_SPARE.Ack_M447 )
   END_RUNG
   // the same network as SCL:
   "DB371_M_UNIT_SPARE".M_CODES_SPARE.Ack_M447 := "M_ZERO";
END_REGION

REGION Network 48: M447- / M115-RADIAL LOCATOR RETURN FIXTURE 1
   RUNG wire#powerrail
      Contact( "DB339_EXTENDED_M_SPARE".M_code[447] )
      wire#w1
      I_Contact( "DB371_M_UNIT_SPARE".M_CODES_SPARE.Ack_M447 )
      I_Contact( "DB2120_MPP_ITC_IPC".RESET_FAULTS )
      I_Contact( "DB371_M_UNIT_SPARE".M_CODES_SPARE.M_RESET_PULSE )
      Coil( "DB371_M_UNIT_SPARE".M_CODES_SPARE.M447 )
   END_RUNG
   RUNG wire#powerrail
      Contact( "DB371_M_UNIT_SPARE".M_CODES_SPARE.M447 )
   END_RUNG wire#w1
   // the same network as SCL:
   "DB371_M_UNIT_SPARE".M_CODES_SPARE.M447 := ("DB339_EXTENDED_M_SPARE".M_code[447] OR "DB371_M_UNIT_SPARE".M_CODES_SPARE.M447) AND NOT "DB371_M_UNIT_SPARE".M_CODES_SPARE.Ack_M447 AND NOT "DB2120_MPP_ITC_IPC".RESET_FAULTS AND NOT "DB371_M_UNIT_SPARE".M_CODES_SPARE.M_RESET_PULSE;
END_REGION

REGION Network 49: ACKNOWLEDGE M448-(READ-IN DISABLE) / ACKNOWLEDGE M116-RADIAL LOCATOR RELAX FIXTURE 1
   RUNG wire#powerrail
      Contact( "M_ZERO" )
      Coil( "DB371_M_UNIT_SPARE".M_CODES_SPARE.Ack_M448 )
   END_RUNG
   // the same network as SCL:
   "DB371_M_UNIT_SPARE".M_CODES_SPARE.Ack_M448 := "M_ZERO";
END_REGION

REGION Network 50: M448-(READ-IN DISABLE) / M116-RADIAL LOCATOR RELAX FIXTURE 1
   RUNG wire#powerrail
      Contact( "DB339_EXTENDED_M_SPARE".M_code[448] )
      wire#w1
      I_Contact( "DB371_M_UNIT_SPARE".M_CODES_SPARE.Ack_M448 )
      I_Contact( "DB2120_MPP_ITC_IPC".RESET_FAULTS )
      I_Contact( "DB371_M_UNIT_SPARE".M_CODES_SPARE.M_RESET_PULSE )
      Coil( "DB371_M_UNIT_SPARE".M_CODES_SPARE.M448 )
   END_RUNG
   RUNG wire#powerrail
      Contact( "DB371_M_UNIT_SPARE".M_CODES_SPARE.M448 )
   END_RUNG wire#w1
   // the same network as SCL:
   "DB371_M_UNIT_SPARE".M_CODES_SPARE.M448 := ("DB339_EXTENDED_M_SPARE".M_code[448] OR "DB371_M_UNIT_SPARE".M_CODES_SPARE.M448) AND NOT "DB371_M_UNIT_SPARE".M_CODES_SPARE.Ack_M448 AND NOT "DB2120_MPP_ITC_IPC".RESET_FAULTS AND NOT "DB371_M_UNIT_SPARE".M_CODES_SPARE.M_RESET_PULSE;
END_REGION

REGION Network 51: ACKNOWLEDGE M449-(READ-IN DISABLE) / ACKNOWLEDGE M116-RADIAL LOCATOR RELAX FIXTURE 1
   RUNG wire#powerrail
      Contact( "M_ZERO" )
      Coil( "DB371_M_UNIT_SPARE".M_CODES_SPARE.Ack_M449 )
   END_RUNG
   // the same network as SCL:
   "DB371_M_UNIT_SPARE".M_CODES_SPARE.Ack_M449 := "M_ZERO";
END_REGION

REGION Network 52: M449-(READ-IN DISABLE) / M116-RADIAL LOCATOR RELAX FIXTURE 1
   RUNG wire#powerrail
      Contact( "DB339_EXTENDED_M_SPARE".M_code[449] )
      wire#w1
      I_Contact( "DB371_M_UNIT_SPARE".M_CODES_SPARE.Ack_M449 )
      I_Contact( "DB2120_MPP_ITC_IPC".RESET_FAULTS )
      I_Contact( "DB371_M_UNIT_SPARE".M_CODES_SPARE.M_RESET_PULSE )
      Coil( "DB371_M_UNIT_SPARE".M_CODES_SPARE.M449 )
   END_RUNG
   RUNG wire#powerrail
      Contact( "DB371_M_UNIT_SPARE".M_CODES_SPARE.M449 )
   END_RUNG wire#w1
   // the same network as SCL:
   "DB371_M_UNIT_SPARE".M_CODES_SPARE.M449 := ("DB339_EXTENDED_M_SPARE".M_code[449] OR "DB371_M_UNIT_SPARE".M_CODES_SPARE.M449) AND NOT "DB371_M_UNIT_SPARE".M_CODES_SPARE.Ack_M449 AND NOT "DB2120_MPP_ITC_IPC".RESET_FAULTS AND NOT "DB371_M_UNIT_SPARE".M_CODES_SPARE.M_RESET_PULSE;
END_REGION

REGION Network 53: ACKNOWLEDGE M450-(READ-IN DISABLE)
   RUNG wire#powerrail
      Contact( "M_ZERO" )
      Coil( "DB371_M_UNIT_SPARE".M_CODES_SPARE.Ack_M450 )
   END_RUNG
   // the same network as SCL:
   "DB371_M_UNIT_SPARE".M_CODES_SPARE.Ack_M450 := "M_ZERO";
END_REGION

REGION Network 54: M450-(READ-IN DISABLE)
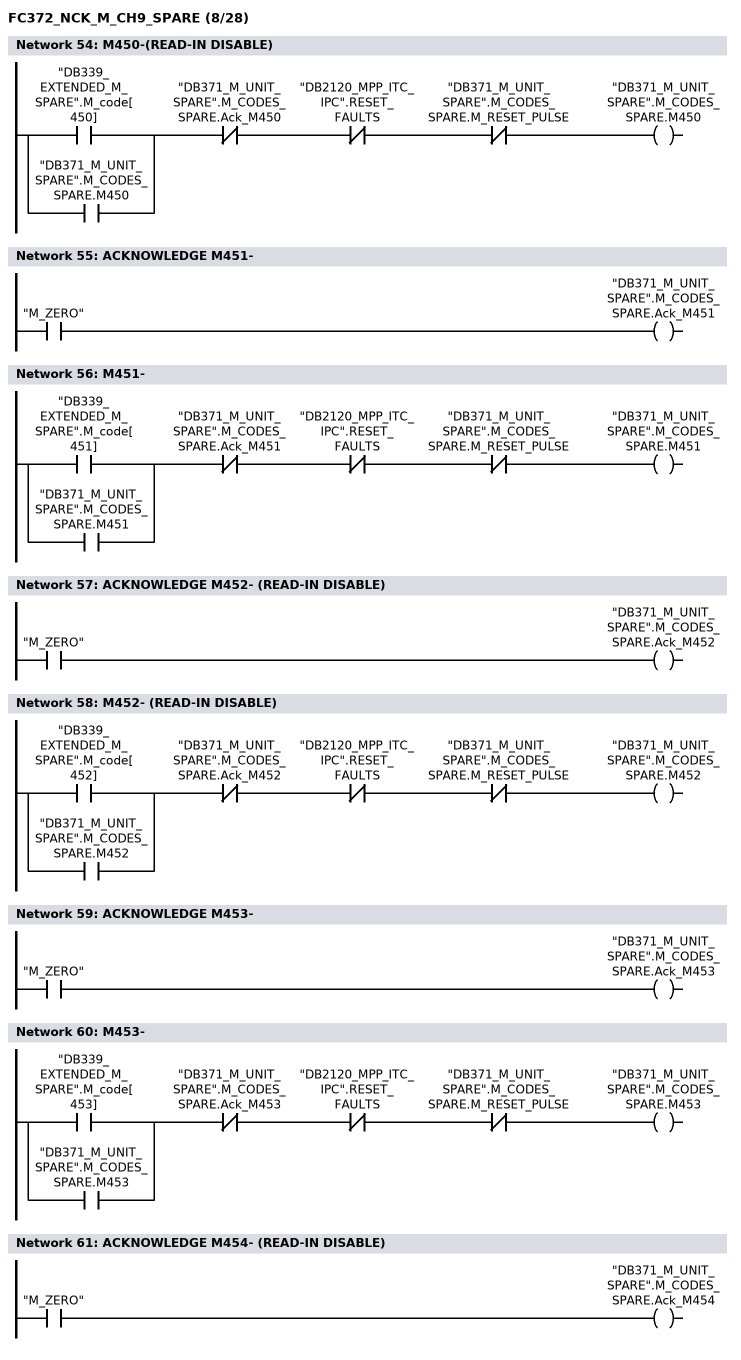
   RUNG wire#powerrail
      Contact( "DB339_EXTENDED_M_SPARE".M_code[450] )
      wire#w1
      I_Contact( "DB371_M_UNIT_SPARE".M_CODES_SPARE.Ack_M450 )
      I_Contact( "DB2120_MPP_ITC_IPC".RESET_FAULTS )
      I_Contact( "DB371_M_UNIT_SPARE".M_CODES_SPARE.M_RESET_PULSE )
      Coil( "DB371_M_UNIT_SPARE".M_CODES_SPARE.M450 )
   END_RUNG
   RUNG wire#powerrail
      Contact( "DB371_M_UNIT_SPARE".M_CODES_SPARE.M450 )
   END_RUNG wire#w1
   // the same network as SCL:
   "DB371_M_UNIT_SPARE".M_CODES_SPARE.M450 := ("DB339_EXTENDED_M_SPARE".M_code[450] OR "DB371_M_UNIT_SPARE".M_CODES_SPARE.M450) AND NOT "DB371_M_UNIT_SPARE".M_CODES_SPARE.Ack_M450 AND NOT "DB2120_MPP_ITC_IPC".RESET_FAULTS AND NOT "DB371_M_UNIT_SPARE".M_CODES_SPARE.M_RESET_PULSE;
END_REGION

REGION Network 55: ACKNOWLEDGE M451-
   RUNG wire#powerrail
      Contact( "M_ZERO" )
      Coil( "DB371_M_UNIT_SPARE".M_CODES_SPARE.Ack_M451 )
   END_RUNG
   // the same network as SCL:
   "DB371_M_UNIT_SPARE".M_CODES_SPARE.Ack_M451 := "M_ZERO";
END_REGION

REGION Network 56: M451-
   RUNG wire#powerrail
      Contact( "DB339_EXTENDED_M_SPARE".M_code[451] )
      wire#w1
      I_Contact( "DB371_M_UNIT_SPARE".M_CODES_SPARE.Ack_M451 )
      I_Contact( "DB2120_MPP_ITC_IPC".RESET_FAULTS )
      I_Contact( "DB371_M_UNIT_SPARE".M_CODES_SPARE.M_RESET_PULSE )
      Coil( "DB371_M_UNIT_SPARE".M_CODES_SPARE.M451 )
   END_RUNG
   RUNG wire#powerrail
      Contact( "DB371_M_UNIT_SPARE".M_CODES_SPARE.M451 )
   END_RUNG wire#w1
   // the same network as SCL:
   "DB371_M_UNIT_SPARE".M_CODES_SPARE.M451 := ("DB339_EXTENDED_M_SPARE".M_code[451] OR "DB371_M_UNIT_SPARE".M_CODES_SPARE.M451) AND NOT "DB371_M_UNIT_SPARE".M_CODES_SPARE.Ack_M451 AND NOT "DB2120_MPP_ITC_IPC".RESET_FAULTS AND NOT "DB371_M_UNIT_SPARE".M_CODES_SPARE.M_RESET_PULSE;
END_REGION

REGION Network 57: ACKNOWLEDGE M452- (READ-IN DISABLE)
   RUNG wire#powerrail
      Contact( "M_ZERO" )
      Coil( "DB371_M_UNIT_SPARE".M_CODES_SPARE.Ack_M452 )
   END_RUNG
   // the same network as SCL:
   "DB371_M_UNIT_SPARE".M_CODES_SPARE.Ack_M452 := "M_ZERO";
END_REGION

REGION Network 58: M452- (READ-IN DISABLE)
   RUNG wire#powerrail
      Contact( "DB339_EXTENDED_M_SPARE".M_code[452] )
      wire#w1
      I_Contact( "DB371_M_UNIT_SPARE".M_CODES_SPARE.Ack_M452 )
      I_Contact( "DB2120_MPP_ITC_IPC".RESET_FAULTS )
      I_Contact( "DB371_M_UNIT_SPARE".M_CODES_SPARE.M_RESET_PULSE )
      Coil( "DB371_M_UNIT_SPARE".M_CODES_SPARE.M452 )
   END_RUNG
   RUNG wire#powerrail
      Contact( "DB371_M_UNIT_SPARE".M_CODES_SPARE.M452 )
   END_RUNG wire#w1
   // the same network as SCL:
   "DB371_M_UNIT_SPARE".M_CODES_SPARE.M452 := ("DB339_EXTENDED_M_SPARE".M_code[452] OR "DB371_M_UNIT_SPARE".M_CODES_SPARE.M452) AND NOT "DB371_M_UNIT_SPARE".M_CODES_SPARE.Ack_M452 AND NOT "DB2120_MPP_ITC_IPC".RESET_FAULTS AND NOT "DB371_M_UNIT_SPARE".M_CODES_SPARE.M_RESET_PULSE;
END_REGION

REGION Network 59: ACKNOWLEDGE M453-
   RUNG wire#powerrail
      Contact( "M_ZERO" )
      Coil( "DB371_M_UNIT_SPARE".M_CODES_SPARE.Ack_M453 )
   END_RUNG
   // the same network as SCL:
   "DB371_M_UNIT_SPARE".M_CODES_SPARE.Ack_M453 := "M_ZERO";
END_REGION

REGION Network 60: M453-
   RUNG wire#powerrail
      Contact( "DB339_EXTENDED_M_SPARE".M_code[453] )
      wire#w1
      I_Contact( "DB371_M_UNIT_SPARE".M_CODES_SPARE.Ack_M453 )
      I_Contact( "DB2120_MPP_ITC_IPC".RESET_FAULTS )
      I_Contact( "DB371_M_UNIT_SPARE".M_CODES_SPARE.M_RESET_PULSE )
      Coil( "DB371_M_UNIT_SPARE".M_CODES_SPARE.M453 )
   END_RUNG
   RUNG wire#powerrail
      Contact( "DB371_M_UNIT_SPARE".M_CODES_SPARE.M453 )
   END_RUNG wire#w1
   // the same network as SCL:
   "DB371_M_UNIT_SPARE".M_CODES_SPARE.M453 := ("DB339_EXTENDED_M_SPARE".M_code[453] OR "DB371_M_UNIT_SPARE".M_CODES_SPARE.M453) AND NOT "DB371_M_UNIT_SPARE".M_CODES_SPARE.Ack_M453 AND NOT "DB2120_MPP_ITC_IPC".RESET_FAULTS AND NOT "DB371_M_UNIT_SPARE".M_CODES_SPARE.M_RESET_PULSE;
END_REGION

REGION Network 61: ACKNOWLEDGE M454- (READ-IN DISABLE)
   RUNG wire#powerrail
      Contact( "M_ZERO" )
      Coil( "DB371_M_UNIT_SPARE".M_CODES_SPARE.Ack_M454 )
   END_RUNG
   // the same network as SCL:
   "DB371_M_UNIT_SPARE".M_CODES_SPARE.Ack_M454 := "M_ZERO";
END_REGION

REGION Network 62: M454- (READ-IN DISABLE)
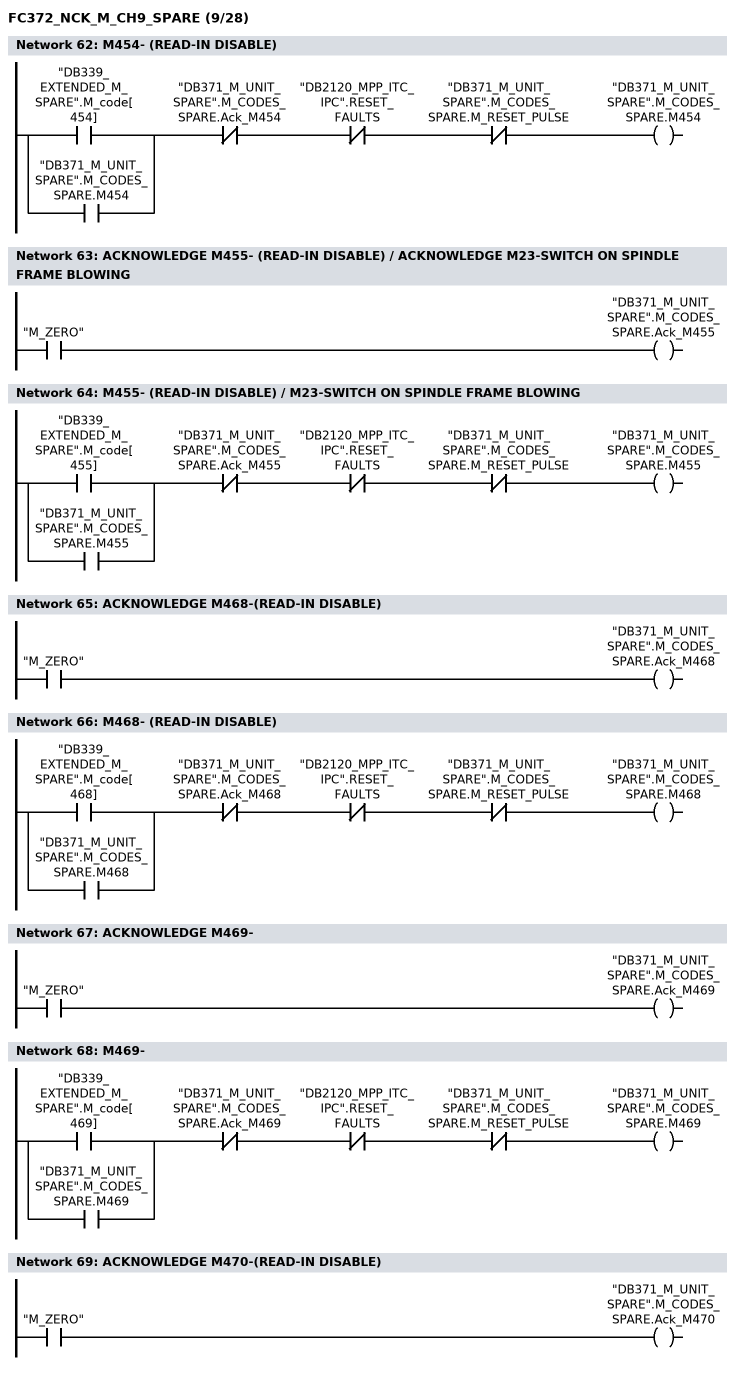
   RUNG wire#powerrail
      Contact( "DB339_EXTENDED_M_SPARE".M_code[454] )
      wire#w1
      I_Contact( "DB371_M_UNIT_SPARE".M_CODES_SPARE.Ack_M454 )
      I_Contact( "DB2120_MPP_ITC_IPC".RESET_FAULTS )
      I_Contact( "DB371_M_UNIT_SPARE".M_CODES_SPARE.M_RESET_PULSE )
      Coil( "DB371_M_UNIT_SPARE".M_CODES_SPARE.M454 )
   END_RUNG
   RUNG wire#powerrail
      Contact( "DB371_M_UNIT_SPARE".M_CODES_SPARE.M454 )
   END_RUNG wire#w1
   // the same network as SCL:
   "DB371_M_UNIT_SPARE".M_CODES_SPARE.M454 := ("DB339_EXTENDED_M_SPARE".M_code[454] OR "DB371_M_UNIT_SPARE".M_CODES_SPARE.M454) AND NOT "DB371_M_UNIT_SPARE".M_CODES_SPARE.Ack_M454 AND NOT "DB2120_MPP_ITC_IPC".RESET_FAULTS AND NOT "DB371_M_UNIT_SPARE".M_CODES_SPARE.M_RESET_PULSE;
END_REGION

REGION Network 63: ACKNOWLEDGE M455- (READ-IN DISABLE) / ACKNOWLEDGE M23-SWITCH ON SPINDLE FRAME BLOWING
   RUNG wire#powerrail
      Contact( "M_ZERO" )
      Coil( "DB371_M_UNIT_SPARE".M_CODES_SPARE.Ack_M455 )
   END_RUNG
   // the same network as SCL:
   "DB371_M_UNIT_SPARE".M_CODES_SPARE.Ack_M455 := "M_ZERO";
END_REGION

REGION Network 64: M455- (READ-IN DISABLE) / M23-SWITCH ON SPINDLE FRAME BLOWING
   RUNG wire#powerrail
      Contact( "DB339_EXTENDED_M_SPARE".M_code[455] )
      wire#w1
      I_Contact( "DB371_M_UNIT_SPARE".M_CODES_SPARE.Ack_M455 )
      I_Contact( "DB2120_MPP_ITC_IPC".RESET_FAULTS )
      I_Contact( "DB371_M_UNIT_SPARE".M_CODES_SPARE.M_RESET_PULSE )
      Coil( "DB371_M_UNIT_SPARE".M_CODES_SPARE.M455 )
   END_RUNG
   RUNG wire#powerrail
      Contact( "DB371_M_UNIT_SPARE".M_CODES_SPARE.M455 )
   END_RUNG wire#w1
   // the same network as SCL:
   "DB371_M_UNIT_SPARE".M_CODES_SPARE.M455 := ("DB339_EXTENDED_M_SPARE".M_code[455] OR "DB371_M_UNIT_SPARE".M_CODES_SPARE.M455) AND NOT "DB371_M_UNIT_SPARE".M_CODES_SPARE.Ack_M455 AND NOT "DB2120_MPP_ITC_IPC".RESET_FAULTS AND NOT "DB371_M_UNIT_SPARE".M_CODES_SPARE.M_RESET_PULSE;
END_REGION

REGION Network 65: ACKNOWLEDGE M468-(READ-IN DISABLE)
   RUNG wire#powerrail
      Contact( "M_ZERO" )
      Coil( "DB371_M_UNIT_SPARE".M_CODES_SPARE.Ack_M468 )
   END_RUNG
   // the same network as SCL:
   "DB371_M_UNIT_SPARE".M_CODES_SPARE.Ack_M468 := "M_ZERO";
END_REGION

REGION Network 66: M468- (READ-IN DISABLE)
   RUNG wire#powerrail
      Contact( "DB339_EXTENDED_M_SPARE".M_code[468] )
      wire#w1
      I_Contact( "DB371_M_UNIT_SPARE".M_CODES_SPARE.Ack_M468 )
      I_Contact( "DB2120_MPP_ITC_IPC".RESET_FAULTS )
      I_Contact( "DB371_M_UNIT_SPARE".M_CODES_SPARE.M_RESET_PULSE )
      Coil( "DB371_M_UNIT_SPARE".M_CODES_SPARE.M468 )
   END_RUNG
   RUNG wire#powerrail
      Contact( "DB371_M_UNIT_SPARE".M_CODES_SPARE.M468 )
   END_RUNG wire#w1
   // the same network as SCL:
   "DB371_M_UNIT_SPARE".M_CODES_SPARE.M468 := ("DB339_EXTENDED_M_SPARE".M_code[468] OR "DB371_M_UNIT_SPARE".M_CODES_SPARE.M468) AND NOT "DB371_M_UNIT_SPARE".M_CODES_SPARE.Ack_M468 AND NOT "DB2120_MPP_ITC_IPC".RESET_FAULTS AND NOT "DB371_M_UNIT_SPARE".M_CODES_SPARE.M_RESET_PULSE;
END_REGION

REGION Network 67: ACKNOWLEDGE M469-
   RUNG wire#powerrail
      Contact( "M_ZERO" )
      Coil( "DB371_M_UNIT_SPARE".M_CODES_SPARE.Ack_M469 )
   END_RUNG
   // the same network as SCL:
   "DB371_M_UNIT_SPARE".M_CODES_SPARE.Ack_M469 := "M_ZERO";
END_REGION

REGION Network 68: M469-
   RUNG wire#powerrail
      Contact( "DB339_EXTENDED_M_SPARE".M_code[469] )
      wire#w1
      I_Contact( "DB371_M_UNIT_SPARE".M_CODES_SPARE.Ack_M469 )
      I_Contact( "DB2120_MPP_ITC_IPC".RESET_FAULTS )
      I_Contact( "DB371_M_UNIT_SPARE".M_CODES_SPARE.M_RESET_PULSE )
      Coil( "DB371_M_UNIT_SPARE".M_CODES_SPARE.M469 )
   END_RUNG
   RUNG wire#powerrail
      Contact( "DB371_M_UNIT_SPARE".M_CODES_SPARE.M469 )
   END_RUNG wire#w1
   // the same network as SCL:
   "DB371_M_UNIT_SPARE".M_CODES_SPARE.M469 := ("DB339_EXTENDED_M_SPARE".M_code[469] OR "DB371_M_UNIT_SPARE".M_CODES_SPARE.M469) AND NOT "DB371_M_UNIT_SPARE".M_CODES_SPARE.Ack_M469 AND NOT "DB2120_MPP_ITC_IPC".RESET_FAULTS AND NOT "DB371_M_UNIT_SPARE".M_CODES_SPARE.M_RESET_PULSE;
END_REGION

REGION Network 69: ACKNOWLEDGE M470-(READ-IN DISABLE)
   RUNG wire#powerrail
      Contact( "M_ZERO" )
      Coil( "DB371_M_UNIT_SPARE".M_CODES_SPARE.Ack_M470 )
   END_RUNG
   // the same network as SCL:
   "DB371_M_UNIT_SPARE".M_CODES_SPARE.Ack_M470 := "M_ZERO";
END_REGION

REGION Network 70: M470-(READ-IN DISABLE)
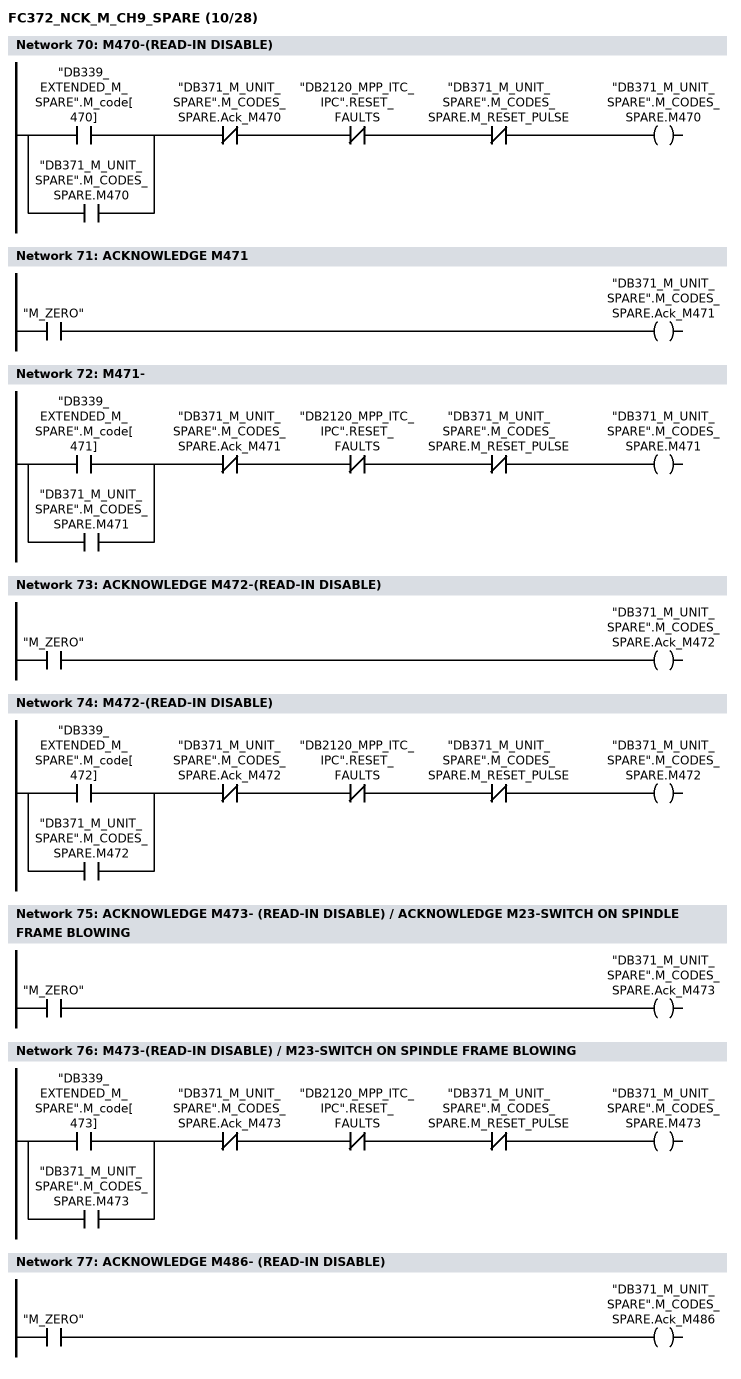
   RUNG wire#powerrail
      Contact( "DB339_EXTENDED_M_SPARE".M_code[470] )
      wire#w1
      I_Contact( "DB371_M_UNIT_SPARE".M_CODES_SPARE.Ack_M470 )
      I_Contact( "DB2120_MPP_ITC_IPC".RESET_FAULTS )
      I_Contact( "DB371_M_UNIT_SPARE".M_CODES_SPARE.M_RESET_PULSE )
      Coil( "DB371_M_UNIT_SPARE".M_CODES_SPARE.M470 )
   END_RUNG
   RUNG wire#powerrail
      Contact( "DB371_M_UNIT_SPARE".M_CODES_SPARE.M470 )
   END_RUNG wire#w1
   // the same network as SCL:
   "DB371_M_UNIT_SPARE".M_CODES_SPARE.M470 := ("DB339_EXTENDED_M_SPARE".M_code[470] OR "DB371_M_UNIT_SPARE".M_CODES_SPARE.M470) AND NOT "DB371_M_UNIT_SPARE".M_CODES_SPARE.Ack_M470 AND NOT "DB2120_MPP_ITC_IPC".RESET_FAULTS AND NOT "DB371_M_UNIT_SPARE".M_CODES_SPARE.M_RESET_PULSE;
END_REGION

REGION Network 71: ACKNOWLEDGE M471
   RUNG wire#powerrail
      Contact( "M_ZERO" )
      Coil( "DB371_M_UNIT_SPARE".M_CODES_SPARE.Ack_M471 )
   END_RUNG
   // the same network as SCL:
   "DB371_M_UNIT_SPARE".M_CODES_SPARE.Ack_M471 := "M_ZERO";
END_REGION

REGION Network 72: M471-
   RUNG wire#powerrail
      Contact( "DB339_EXTENDED_M_SPARE".M_code[471] )
      wire#w1
      I_Contact( "DB371_M_UNIT_SPARE".M_CODES_SPARE.Ack_M471 )
      I_Contact( "DB2120_MPP_ITC_IPC".RESET_FAULTS )
      I_Contact( "DB371_M_UNIT_SPARE".M_CODES_SPARE.M_RESET_PULSE )
      Coil( "DB371_M_UNIT_SPARE".M_CODES_SPARE.M471 )
   END_RUNG
   RUNG wire#powerrail
      Contact( "DB371_M_UNIT_SPARE".M_CODES_SPARE.M471 )
   END_RUNG wire#w1
   // the same network as SCL:
   "DB371_M_UNIT_SPARE".M_CODES_SPARE.M471 := ("DB339_EXTENDED_M_SPARE".M_code[471] OR "DB371_M_UNIT_SPARE".M_CODES_SPARE.M471) AND NOT "DB371_M_UNIT_SPARE".M_CODES_SPARE.Ack_M471 AND NOT "DB2120_MPP_ITC_IPC".RESET_FAULTS AND NOT "DB371_M_UNIT_SPARE".M_CODES_SPARE.M_RESET_PULSE;
END_REGION

REGION Network 73: ACKNOWLEDGE M472-(READ-IN DISABLE)
   RUNG wire#powerrail
      Contact( "M_ZERO" )
      Coil( "DB371_M_UNIT_SPARE".M_CODES_SPARE.Ack_M472 )
   END_RUNG
   // the same network as SCL:
   "DB371_M_UNIT_SPARE".M_CODES_SPARE.Ack_M472 := "M_ZERO";
END_REGION

REGION Network 74: M472-(READ-IN DISABLE)
   RUNG wire#powerrail
      Contact( "DB339_EXTENDED_M_SPARE".M_code[472] )
      wire#w1
      I_Contact( "DB371_M_UNIT_SPARE".M_CODES_SPARE.Ack_M472 )
      I_Contact( "DB2120_MPP_ITC_IPC".RESET_FAULTS )
      I_Contact( "DB371_M_UNIT_SPARE".M_CODES_SPARE.M_RESET_PULSE )
      Coil( "DB371_M_UNIT_SPARE".M_CODES_SPARE.M472 )
   END_RUNG
   RUNG wire#powerrail
      Contact( "DB371_M_UNIT_SPARE".M_CODES_SPARE.M472 )
   END_RUNG wire#w1
   // the same network as SCL:
   "DB371_M_UNIT_SPARE".M_CODES_SPARE.M472 := ("DB339_EXTENDED_M_SPARE".M_code[472] OR "DB371_M_UNIT_SPARE".M_CODES_SPARE.M472) AND NOT "DB371_M_UNIT_SPARE".M_CODES_SPARE.Ack_M472 AND NOT "DB2120_MPP_ITC_IPC".RESET_FAULTS AND NOT "DB371_M_UNIT_SPARE".M_CODES_SPARE.M_RESET_PULSE;
END_REGION

REGION Network 75: ACKNOWLEDGE M473- (READ-IN DISABLE) / ACKNOWLEDGE M23-SWITCH ON SPINDLE FRAME BLOWING
   RUNG wire#powerrail
      Contact( "M_ZERO" )
      Coil( "DB371_M_UNIT_SPARE".M_CODES_SPARE.Ack_M473 )
   END_RUNG
   // the same network as SCL:
   "DB371_M_UNIT_SPARE".M_CODES_SPARE.Ack_M473 := "M_ZERO";
END_REGION

REGION Network 76: M473-(READ-IN DISABLE) / M23-SWITCH ON SPINDLE FRAME BLOWING
   RUNG wire#powerrail
      Contact( "DB339_EXTENDED_M_SPARE".M_code[473] )
      wire#w1
      I_Contact( "DB371_M_UNIT_SPARE".M_CODES_SPARE.Ack_M473 )
      I_Contact( "DB2120_MPP_ITC_IPC".RESET_FAULTS )
      I_Contact( "DB371_M_UNIT_SPARE".M_CODES_SPARE.M_RESET_PULSE )
      Coil( "DB371_M_UNIT_SPARE".M_CODES_SPARE.M473 )
   END_RUNG
   RUNG wire#powerrail
      Contact( "DB371_M_UNIT_SPARE".M_CODES_SPARE.M473 )
   END_RUNG wire#w1
   // the same network as SCL:
   "DB371_M_UNIT_SPARE".M_CODES_SPARE.M473 := ("DB339_EXTENDED_M_SPARE".M_code[473] OR "DB371_M_UNIT_SPARE".M_CODES_SPARE.M473) AND NOT "DB371_M_UNIT_SPARE".M_CODES_SPARE.Ack_M473 AND NOT "DB2120_MPP_ITC_IPC".RESET_FAULTS AND NOT "DB371_M_UNIT_SPARE".M_CODES_SPARE.M_RESET_PULSE;
END_REGION

REGION Network 77: ACKNOWLEDGE M486- (READ-IN DISABLE)
   RUNG wire#powerrail
      Contact( "M_ZERO" )
      Coil( "DB371_M_UNIT_SPARE".M_CODES_SPARE.Ack_M486 )
   END_RUNG
   // the same network as SCL:
   "DB371_M_UNIT_SPARE".M_CODES_SPARE.Ack_M486 := "M_ZERO";
END_REGION

REGION Network 78: M486-(READ-IN DISABLE)
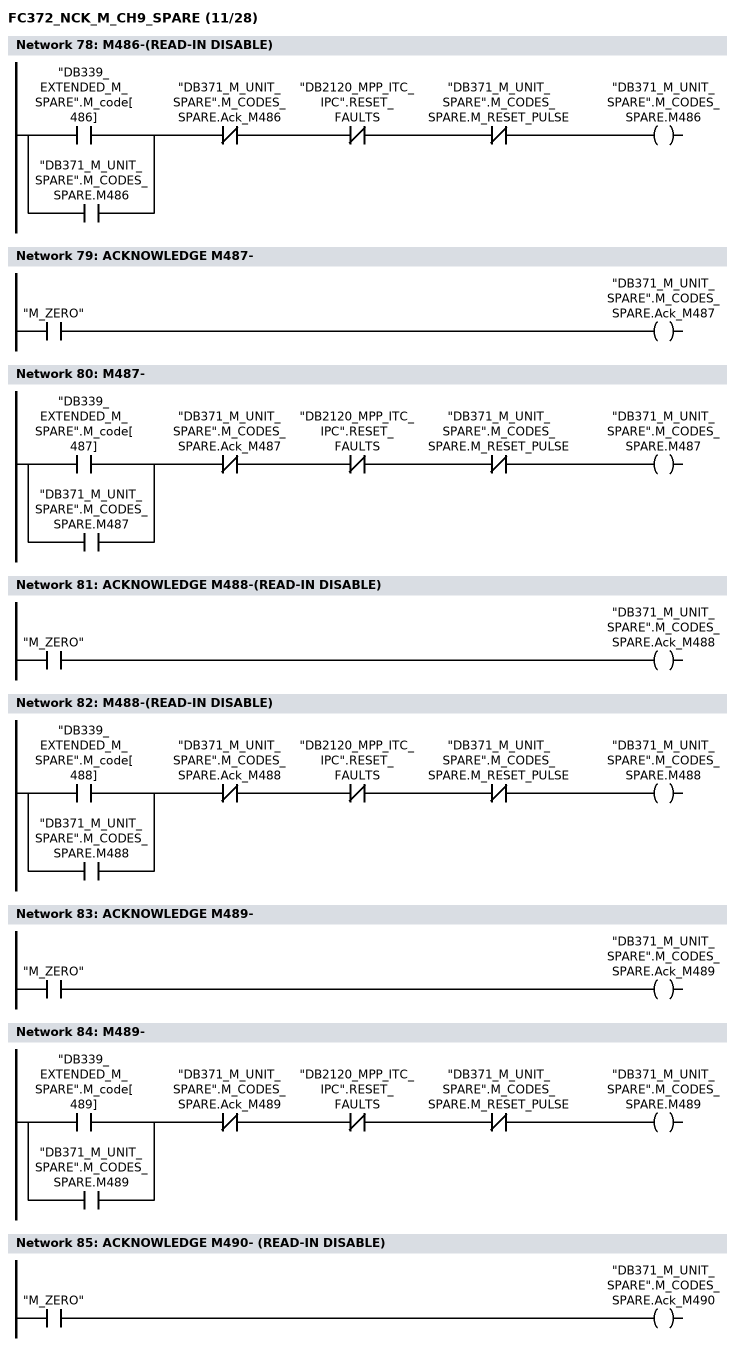
   RUNG wire#powerrail
      Contact( "DB339_EXTENDED_M_SPARE".M_code[486] )
      wire#w1
      I_Contact( "DB371_M_UNIT_SPARE".M_CODES_SPARE.Ack_M486 )
      I_Contact( "DB2120_MPP_ITC_IPC".RESET_FAULTS )
      I_Contact( "DB371_M_UNIT_SPARE".M_CODES_SPARE.M_RESET_PULSE )
      Coil( "DB371_M_UNIT_SPARE".M_CODES_SPARE.M486 )
   END_RUNG
   RUNG wire#powerrail
      Contact( "DB371_M_UNIT_SPARE".M_CODES_SPARE.M486 )
   END_RUNG wire#w1
   // the same network as SCL:
   "DB371_M_UNIT_SPARE".M_CODES_SPARE.M486 := ("DB339_EXTENDED_M_SPARE".M_code[486] OR "DB371_M_UNIT_SPARE".M_CODES_SPARE.M486) AND NOT "DB371_M_UNIT_SPARE".M_CODES_SPARE.Ack_M486 AND NOT "DB2120_MPP_ITC_IPC".RESET_FAULTS AND NOT "DB371_M_UNIT_SPARE".M_CODES_SPARE.M_RESET_PULSE;
END_REGION

REGION Network 79: ACKNOWLEDGE M487-
   RUNG wire#powerrail
      Contact( "M_ZERO" )
      Coil( "DB371_M_UNIT_SPARE".M_CODES_SPARE.Ack_M487 )
   END_RUNG
   // the same network as SCL:
   "DB371_M_UNIT_SPARE".M_CODES_SPARE.Ack_M487 := "M_ZERO";
END_REGION

REGION Network 80: M487-
   RUNG wire#powerrail
      Contact( "DB339_EXTENDED_M_SPARE".M_code[487] )
      wire#w1
      I_Contact( "DB371_M_UNIT_SPARE".M_CODES_SPARE.Ack_M487 )
      I_Contact( "DB2120_MPP_ITC_IPC".RESET_FAULTS )
      I_Contact( "DB371_M_UNIT_SPARE".M_CODES_SPARE.M_RESET_PULSE )
      Coil( "DB371_M_UNIT_SPARE".M_CODES_SPARE.M487 )
   END_RUNG
   RUNG wire#powerrail
      Contact( "DB371_M_UNIT_SPARE".M_CODES_SPARE.M487 )
   END_RUNG wire#w1
   // the same network as SCL:
   "DB371_M_UNIT_SPARE".M_CODES_SPARE.M487 := ("DB339_EXTENDED_M_SPARE".M_code[487] OR "DB371_M_UNIT_SPARE".M_CODES_SPARE.M487) AND NOT "DB371_M_UNIT_SPARE".M_CODES_SPARE.Ack_M487 AND NOT "DB2120_MPP_ITC_IPC".RESET_FAULTS AND NOT "DB371_M_UNIT_SPARE".M_CODES_SPARE.M_RESET_PULSE;
END_REGION

REGION Network 81: ACKNOWLEDGE M488-(READ-IN DISABLE)
   RUNG wire#powerrail
      Contact( "M_ZERO" )
      Coil( "DB371_M_UNIT_SPARE".M_CODES_SPARE.Ack_M488 )
   END_RUNG
   // the same network as SCL:
   "DB371_M_UNIT_SPARE".M_CODES_SPARE.Ack_M488 := "M_ZERO";
END_REGION

REGION Network 82: M488-(READ-IN DISABLE)
   RUNG wire#powerrail
      Contact( "DB339_EXTENDED_M_SPARE".M_code[488] )
      wire#w1
      I_Contact( "DB371_M_UNIT_SPARE".M_CODES_SPARE.Ack_M488 )
      I_Contact( "DB2120_MPP_ITC_IPC".RESET_FAULTS )
      I_Contact( "DB371_M_UNIT_SPARE".M_CODES_SPARE.M_RESET_PULSE )
      Coil( "DB371_M_UNIT_SPARE".M_CODES_SPARE.M488 )
   END_RUNG
   RUNG wire#powerrail
      Contact( "DB371_M_UNIT_SPARE".M_CODES_SPARE.M488 )
   END_RUNG wire#w1
   // the same network as SCL:
   "DB371_M_UNIT_SPARE".M_CODES_SPARE.M488 := ("DB339_EXTENDED_M_SPARE".M_code[488] OR "DB371_M_UNIT_SPARE".M_CODES_SPARE.M488) AND NOT "DB371_M_UNIT_SPARE".M_CODES_SPARE.Ack_M488 AND NOT "DB2120_MPP_ITC_IPC".RESET_FAULTS AND NOT "DB371_M_UNIT_SPARE".M_CODES_SPARE.M_RESET_PULSE;
END_REGION

REGION Network 83: ACKNOWLEDGE M489-
   RUNG wire#powerrail
      Contact( "M_ZERO" )
      Coil( "DB371_M_UNIT_SPARE".M_CODES_SPARE.Ack_M489 )
   END_RUNG
   // the same network as SCL:
   "DB371_M_UNIT_SPARE".M_CODES_SPARE.Ack_M489 := "M_ZERO";
END_REGION

REGION Network 84: M489-
   RUNG wire#powerrail
      Contact( "DB339_EXTENDED_M_SPARE".M_code[489] )
      wire#w1
      I_Contact( "DB371_M_UNIT_SPARE".M_CODES_SPARE.Ack_M489 )
      I_Contact( "DB2120_MPP_ITC_IPC".RESET_FAULTS )
      I_Contact( "DB371_M_UNIT_SPARE".M_CODES_SPARE.M_RESET_PULSE )
      Coil( "DB371_M_UNIT_SPARE".M_CODES_SPARE.M489 )
   END_RUNG
   RUNG wire#powerrail
      Contact( "DB371_M_UNIT_SPARE".M_CODES_SPARE.M489 )
   END_RUNG wire#w1
   // the same network as SCL:
   "DB371_M_UNIT_SPARE".M_CODES_SPARE.M489 := ("DB339_EXTENDED_M_SPARE".M_code[489] OR "DB371_M_UNIT_SPARE".M_CODES_SPARE.M489) AND NOT "DB371_M_UNIT_SPARE".M_CODES_SPARE.Ack_M489 AND NOT "DB2120_MPP_ITC_IPC".RESET_FAULTS AND NOT "DB371_M_UNIT_SPARE".M_CODES_SPARE.M_RESET_PULSE;
END_REGION

REGION Network 85: ACKNOWLEDGE M490- (READ-IN DISABLE)
   RUNG wire#powerrail
      Contact( "M_ZERO" )
      Coil( "DB371_M_UNIT_SPARE".M_CODES_SPARE.Ack_M490 )
   END_RUNG
   // the same network as SCL:
   "DB371_M_UNIT_SPARE".M_CODES_SPARE.Ack_M490 := "M_ZERO";
END_REGION

REGION Network 86: M490-(READ-IN DISABLE)
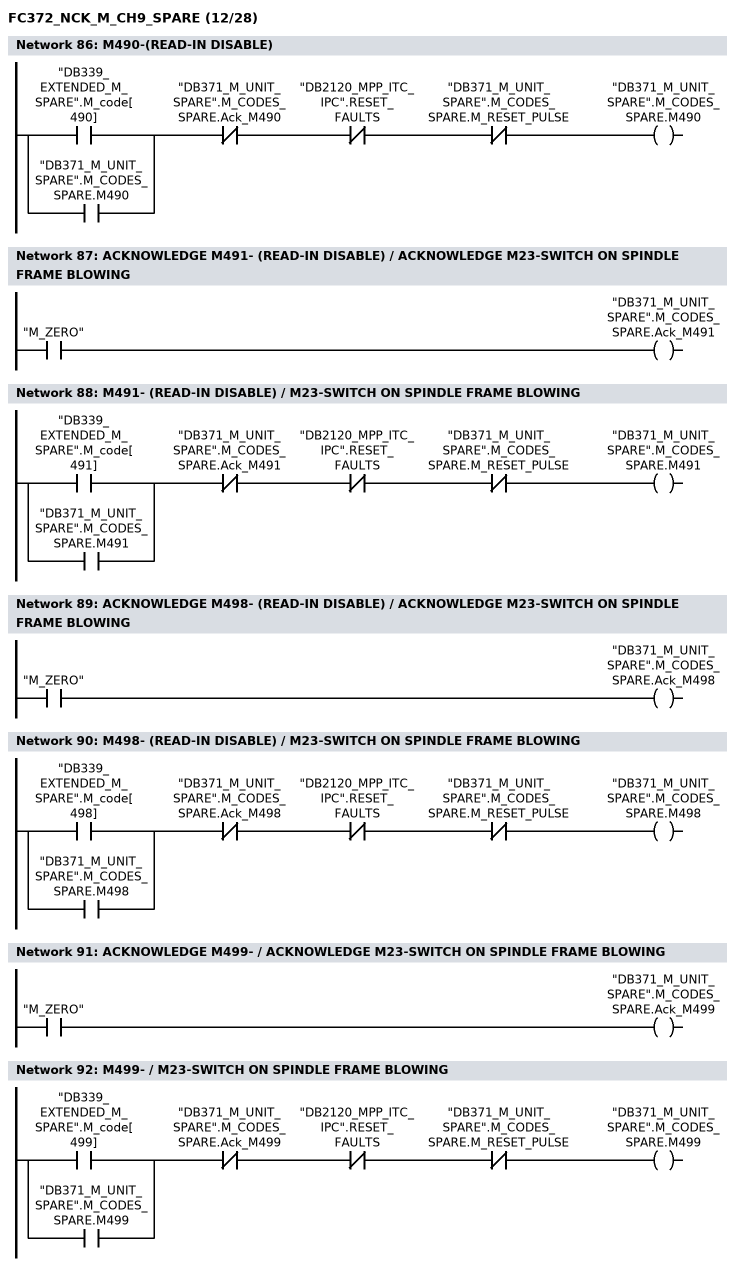
   RUNG wire#powerrail
      Contact( "DB339_EXTENDED_M_SPARE".M_code[490] )
      wire#w1
      I_Contact( "DB371_M_UNIT_SPARE".M_CODES_SPARE.Ack_M490 )
      I_Contact( "DB2120_MPP_ITC_IPC".RESET_FAULTS )
      I_Contact( "DB371_M_UNIT_SPARE".M_CODES_SPARE.M_RESET_PULSE )
      Coil( "DB371_M_UNIT_SPARE".M_CODES_SPARE.M490 )
   END_RUNG
   RUNG wire#powerrail
      Contact( "DB371_M_UNIT_SPARE".M_CODES_SPARE.M490 )
   END_RUNG wire#w1
   // the same network as SCL:
   "DB371_M_UNIT_SPARE".M_CODES_SPARE.M490 := ("DB339_EXTENDED_M_SPARE".M_code[490] OR "DB371_M_UNIT_SPARE".M_CODES_SPARE.M490) AND NOT "DB371_M_UNIT_SPARE".M_CODES_SPARE.Ack_M490 AND NOT "DB2120_MPP_ITC_IPC".RESET_FAULTS AND NOT "DB371_M_UNIT_SPARE".M_CODES_SPARE.M_RESET_PULSE;
END_REGION

REGION Network 87: ACKNOWLEDGE M491- (READ-IN DISABLE) / ACKNOWLEDGE M23-SWITCH ON SPINDLE FRAME BLOWING
   RUNG wire#powerrail
      Contact( "M_ZERO" )
      Coil( "DB371_M_UNIT_SPARE".M_CODES_SPARE.Ack_M491 )
   END_RUNG
   // the same network as SCL:
   "DB371_M_UNIT_SPARE".M_CODES_SPARE.Ack_M491 := "M_ZERO";
END_REGION

REGION Network 88: M491- (READ-IN DISABLE) / M23-SWITCH ON SPINDLE FRAME BLOWING
   RUNG wire#powerrail
      Contact( "DB339_EXTENDED_M_SPARE".M_code[491] )
      wire#w1
      I_Contact( "DB371_M_UNIT_SPARE".M_CODES_SPARE.Ack_M491 )
      I_Contact( "DB2120_MPP_ITC_IPC".RESET_FAULTS )
      I_Contact( "DB371_M_UNIT_SPARE".M_CODES_SPARE.M_RESET_PULSE )
      Coil( "DB371_M_UNIT_SPARE".M_CODES_SPARE.M491 )
   END_RUNG
   RUNG wire#powerrail
      Contact( "DB371_M_UNIT_SPARE".M_CODES_SPARE.M491 )
   END_RUNG wire#w1
   // the same network as SCL:
   "DB371_M_UNIT_SPARE".M_CODES_SPARE.M491 := ("DB339_EXTENDED_M_SPARE".M_code[491] OR "DB371_M_UNIT_SPARE".M_CODES_SPARE.M491) AND NOT "DB371_M_UNIT_SPARE".M_CODES_SPARE.Ack_M491 AND NOT "DB2120_MPP_ITC_IPC".RESET_FAULTS AND NOT "DB371_M_UNIT_SPARE".M_CODES_SPARE.M_RESET_PULSE;
END_REGION

REGION Network 89: ACKNOWLEDGE M498- (READ-IN DISABLE) / ACKNOWLEDGE M23-SWITCH ON SPINDLE FRAME BLOWING
   RUNG wire#powerrail
      Contact( "M_ZERO" )
      Coil( "DB371_M_UNIT_SPARE".M_CODES_SPARE.Ack_M498 )
   END_RUNG
   // the same network as SCL:
   "DB371_M_UNIT_SPARE".M_CODES_SPARE.Ack_M498 := "M_ZERO";
END_REGION

REGION Network 90: M498- (READ-IN DISABLE) / M23-SWITCH ON SPINDLE FRAME BLOWING
   RUNG wire#powerrail
      Contact( "DB339_EXTENDED_M_SPARE".M_code[498] )
      wire#w1
      I_Contact( "DB371_M_UNIT_SPARE".M_CODES_SPARE.Ack_M498 )
      I_Contact( "DB2120_MPP_ITC_IPC".RESET_FAULTS )
      I_Contact( "DB371_M_UNIT_SPARE".M_CODES_SPARE.M_RESET_PULSE )
      Coil( "DB371_M_UNIT_SPARE".M_CODES_SPARE.M498 )
   END_RUNG
   RUNG wire#powerrail
      Contact( "DB371_M_UNIT_SPARE".M_CODES_SPARE.M498 )
   END_RUNG wire#w1
   // the same network as SCL:
   "DB371_M_UNIT_SPARE".M_CODES_SPARE.M498 := ("DB339_EXTENDED_M_SPARE".M_code[498] OR "DB371_M_UNIT_SPARE".M_CODES_SPARE.M498) AND NOT "DB371_M_UNIT_SPARE".M_CODES_SPARE.Ack_M498 AND NOT "DB2120_MPP_ITC_IPC".RESET_FAULTS AND NOT "DB371_M_UNIT_SPARE".M_CODES_SPARE.M_RESET_PULSE;
END_REGION

REGION Network 91: ACKNOWLEDGE M499- / ACKNOWLEDGE M23-SWITCH ON SPINDLE FRAME BLOWING
   RUNG wire#powerrail
      Contact( "M_ZERO" )
      Coil( "DB371_M_UNIT_SPARE".M_CODES_SPARE.Ack_M499 )
   END_RUNG
   // the same network as SCL:
   "DB371_M_UNIT_SPARE".M_CODES_SPARE.Ack_M499 := "M_ZERO";
END_REGION

REGION Network 92: M499- / M23-SWITCH ON SPINDLE FRAME BLOWING
   RUNG wire#powerrail
      Contact( "DB339_EXTENDED_M_SPARE".M_code[499] )
      wire#w1
      I_Contact( "DB371_M_UNIT_SPARE".M_CODES_SPARE.Ack_M499 )
      I_Contact( "DB2120_MPP_ITC_IPC".RESET_FAULTS )
      I_Contact( "DB371_M_UNIT_SPARE".M_CODES_SPARE.M_RESET_PULSE )
      Coil( "DB371_M_UNIT_SPARE".M_CODES_SPARE.M499 )
   END_RUNG
   RUNG wire#powerrail
      Contact( "DB371_M_UNIT_SPARE".M_CODES_SPARE.M499 )
   END_RUNG wire#w1
   // the same network as SCL:
   "DB371_M_UNIT_SPARE".M_CODES_SPARE.M499 := ("DB339_EXTENDED_M_SPARE".M_code[499] OR "DB371_M_UNIT_SPARE".M_CODES_SPARE.M499) AND NOT "DB371_M_UNIT_SPARE".M_CODES_SPARE.Ack_M499 AND NOT "DB2120_MPP_ITC_IPC".RESET_FAULTS AND NOT "DB371_M_UNIT_SPARE".M_CODES_SPARE.M_RESET_PULSE;
END_REGION

REGION Network 93: ACKNOWLEDGE M500-FIXTURE 2 CLAMP SEQUENCE (READ-IN DISABLE) / ACKNOWLEDGE M100-CLAMP SEQUENCE FIXTURE 1
   // NOTE: WHEN THERE IS NOT INDEXING TABLE AVAILABLE IN THE MACHINE DELETE 
   // DB2171.DBX5.0 AND DB2171.DBX2.0
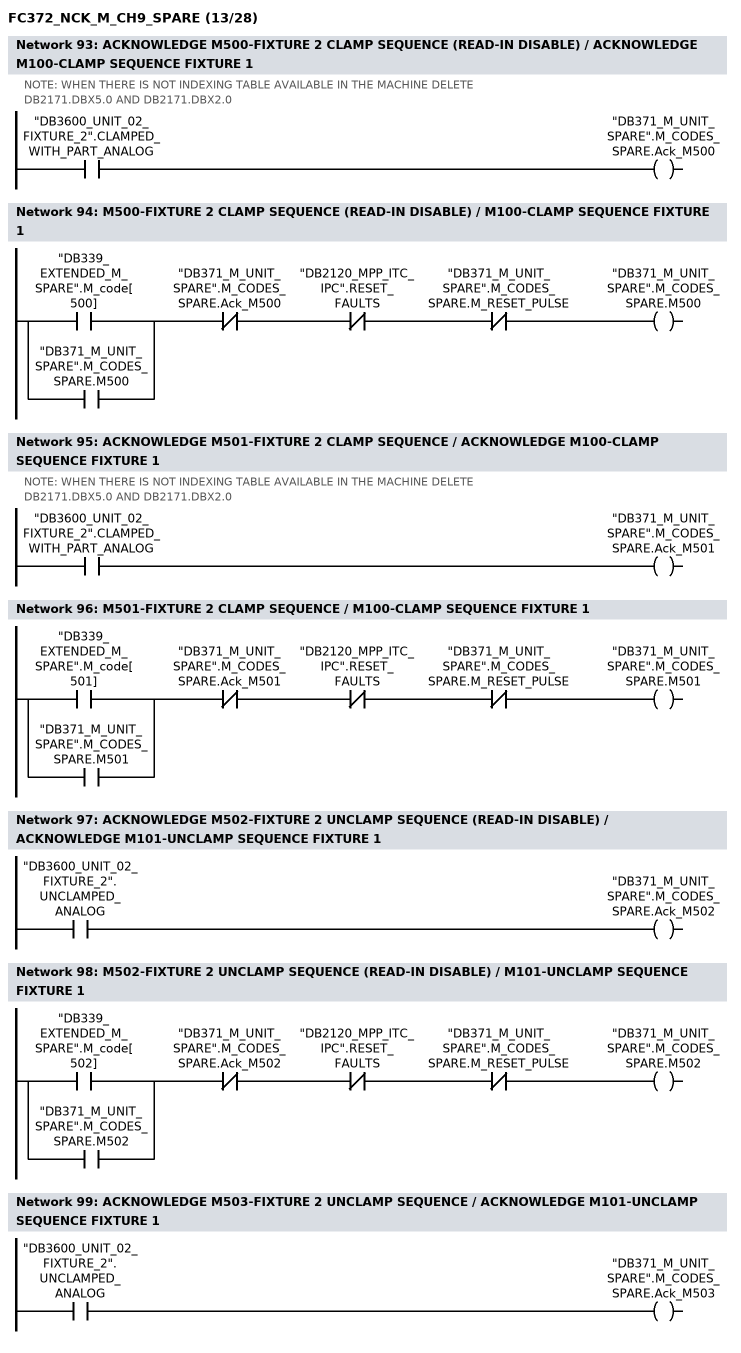
   RUNG wire#powerrail
      Contact( "DB3600_UNIT_02_FIXTURE_2".CLAMPED_WITH_PART_ANALOG )
      Coil( "DB371_M_UNIT_SPARE".M_CODES_SPARE.Ack_M500 )
   END_RUNG
   // the same network as SCL:
   "DB371_M_UNIT_SPARE".M_CODES_SPARE.Ack_M500 := "DB3600_UNIT_02_FIXTURE_2".CLAMPED_WITH_PART_ANALOG;
END_REGION

REGION Network 94: M500-FIXTURE 2 CLAMP SEQUENCE (READ-IN DISABLE) / M100-CLAMP SEQUENCE FIXTURE 1
   RUNG wire#powerrail
      Contact( "DB339_EXTENDED_M_SPARE".M_code[500] )
      wire#w1
      I_Contact( "DB371_M_UNIT_SPARE".M_CODES_SPARE.Ack_M500 )
      I_Contact( "DB2120_MPP_ITC_IPC".RESET_FAULTS )
      I_Contact( "DB371_M_UNIT_SPARE".M_CODES_SPARE.M_RESET_PULSE )
      Coil( "DB371_M_UNIT_SPARE".M_CODES_SPARE.M500 )
   END_RUNG
   RUNG wire#powerrail
      Contact( "DB371_M_UNIT_SPARE".M_CODES_SPARE.M500 )
   END_RUNG wire#w1
   // the same network as SCL:
   "DB371_M_UNIT_SPARE".M_CODES_SPARE.M500 := ("DB339_EXTENDED_M_SPARE".M_code[500] OR "DB371_M_UNIT_SPARE".M_CODES_SPARE.M500) AND NOT "DB371_M_UNIT_SPARE".M_CODES_SPARE.Ack_M500 AND NOT "DB2120_MPP_ITC_IPC".RESET_FAULTS AND NOT "DB371_M_UNIT_SPARE".M_CODES_SPARE.M_RESET_PULSE;
END_REGION

REGION Network 95: ACKNOWLEDGE M501-FIXTURE 2 CLAMP SEQUENCE / ACKNOWLEDGE M100-CLAMP SEQUENCE FIXTURE 1
   // NOTE: WHEN THERE IS NOT INDEXING TABLE AVAILABLE IN THE MACHINE DELETE 
   // DB2171.DBX5.0 AND DB2171.DBX2.0
   RUNG wire#powerrail
      Contact( "DB3600_UNIT_02_FIXTURE_2".CLAMPED_WITH_PART_ANALOG )
      Coil( "DB371_M_UNIT_SPARE".M_CODES_SPARE.Ack_M501 )
   END_RUNG
   // the same network as SCL:
   "DB371_M_UNIT_SPARE".M_CODES_SPARE.Ack_M501 := "DB3600_UNIT_02_FIXTURE_2".CLAMPED_WITH_PART_ANALOG;
END_REGION

REGION Network 96: M501-FIXTURE 2 CLAMP SEQUENCE / M100-CLAMP SEQUENCE FIXTURE 1
   RUNG wire#powerrail
      Contact( "DB339_EXTENDED_M_SPARE".M_code[501] )
      wire#w1
      I_Contact( "DB371_M_UNIT_SPARE".M_CODES_SPARE.Ack_M501 )
      I_Contact( "DB2120_MPP_ITC_IPC".RESET_FAULTS )
      I_Contact( "DB371_M_UNIT_SPARE".M_CODES_SPARE.M_RESET_PULSE )
      Coil( "DB371_M_UNIT_SPARE".M_CODES_SPARE.M501 )
   END_RUNG
   RUNG wire#powerrail
      Contact( "DB371_M_UNIT_SPARE".M_CODES_SPARE.M501 )
   END_RUNG wire#w1
   // the same network as SCL:
   "DB371_M_UNIT_SPARE".M_CODES_SPARE.M501 := ("DB339_EXTENDED_M_SPARE".M_code[501] OR "DB371_M_UNIT_SPARE".M_CODES_SPARE.M501) AND NOT "DB371_M_UNIT_SPARE".M_CODES_SPARE.Ack_M501 AND NOT "DB2120_MPP_ITC_IPC".RESET_FAULTS AND NOT "DB371_M_UNIT_SPARE".M_CODES_SPARE.M_RESET_PULSE;
END_REGION

REGION Network 97: ACKNOWLEDGE M502-FIXTURE 2 UNCLAMP SEQUENCE (READ-IN DISABLE) / ACKNOWLEDGE M101-UNCLAMP SEQUENCE FIXTURE 1
   RUNG wire#powerrail
      Contact( "DB3600_UNIT_02_FIXTURE_2".UNCLAMPED_ANALOG )
      Coil( "DB371_M_UNIT_SPARE".M_CODES_SPARE.Ack_M502 )
   END_RUNG
   // the same network as SCL:
   "DB371_M_UNIT_SPARE".M_CODES_SPARE.Ack_M502 := "DB3600_UNIT_02_FIXTURE_2".UNCLAMPED_ANALOG;
END_REGION

REGION Network 98: M502-FIXTURE 2 UNCLAMP SEQUENCE (READ-IN DISABLE) / M101-UNCLAMP SEQUENCE FIXTURE 1
   RUNG wire#powerrail
      Contact( "DB339_EXTENDED_M_SPARE".M_code[502] )
      wire#w1
      I_Contact( "DB371_M_UNIT_SPARE".M_CODES_SPARE.Ack_M502 )
      I_Contact( "DB2120_MPP_ITC_IPC".RESET_FAULTS )
      I_Contact( "DB371_M_UNIT_SPARE".M_CODES_SPARE.M_RESET_PULSE )
      Coil( "DB371_M_UNIT_SPARE".M_CODES_SPARE.M502 )
   END_RUNG
   RUNG wire#powerrail
      Contact( "DB371_M_UNIT_SPARE".M_CODES_SPARE.M502 )
   END_RUNG wire#w1
   // the same network as SCL:
   "DB371_M_UNIT_SPARE".M_CODES_SPARE.M502 := ("DB339_EXTENDED_M_SPARE".M_code[502] OR "DB371_M_UNIT_SPARE".M_CODES_SPARE.M502) AND NOT "DB371_M_UNIT_SPARE".M_CODES_SPARE.Ack_M502 AND NOT "DB2120_MPP_ITC_IPC".RESET_FAULTS AND NOT "DB371_M_UNIT_SPARE".M_CODES_SPARE.M_RESET_PULSE;
END_REGION

REGION Network 99: ACKNOWLEDGE M503-FIXTURE 2 UNCLAMP SEQUENCE / ACKNOWLEDGE M101-UNCLAMP SEQUENCE FIXTURE 1
   RUNG wire#powerrail
      Contact( "DB3600_UNIT_02_FIXTURE_2".UNCLAMPED_ANALOG )
      Coil( "DB371_M_UNIT_SPARE".M_CODES_SPARE.Ack_M503 )
   END_RUNG
   // the same network as SCL:
   "DB371_M_UNIT_SPARE".M_CODES_SPARE.Ack_M503 := "DB3600_UNIT_02_FIXTURE_2".UNCLAMPED_ANALOG;
END_REGION

REGION Network 100: M503-FIXTURE 2 UNCLAMP SEQUENCE / M101-UNCLAMP SEQUENCE FIXTURE 1
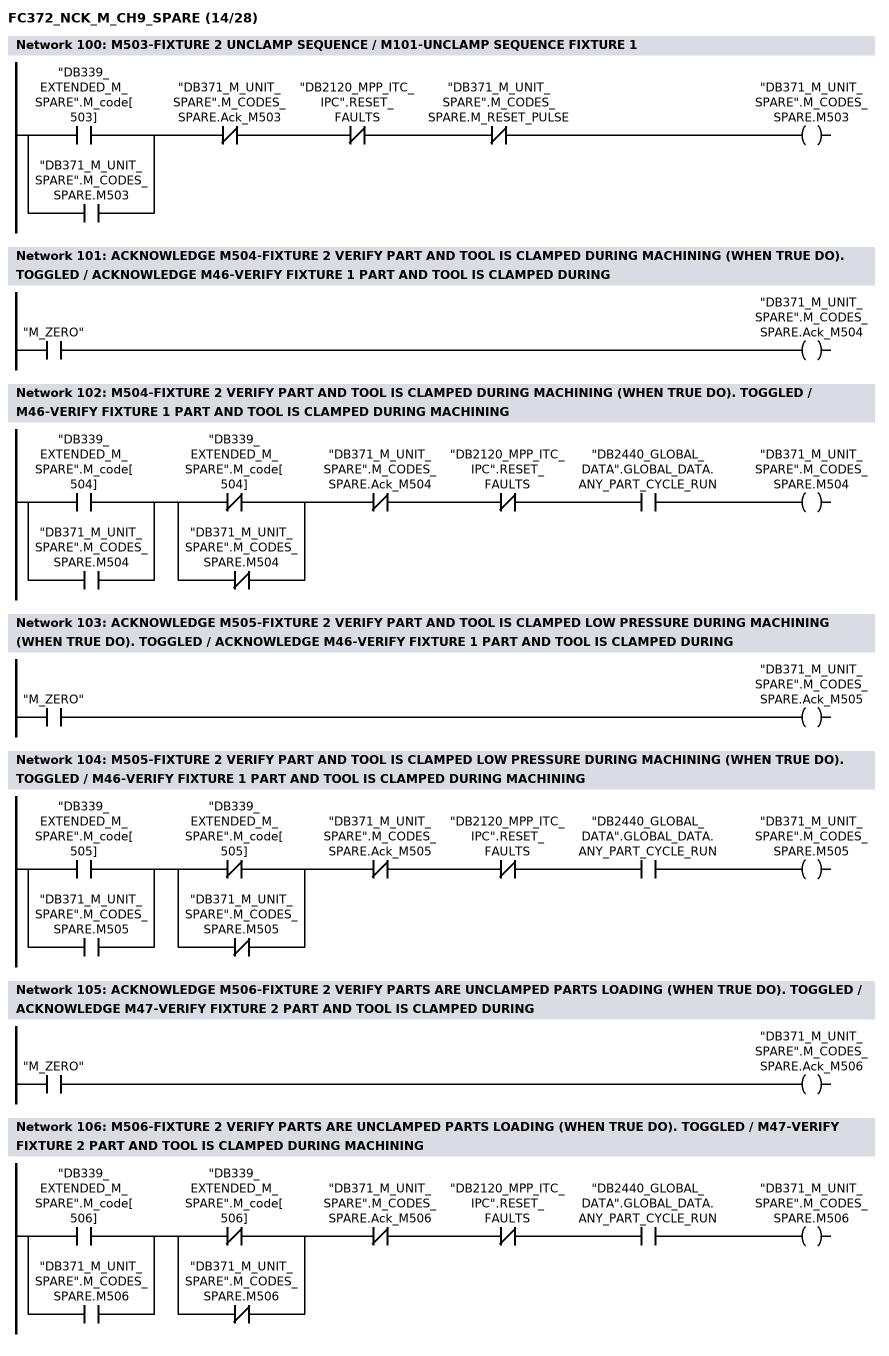
   RUNG wire#powerrail
      Contact( "DB339_EXTENDED_M_SPARE".M_code[503] )
      wire#w1
      I_Contact( "DB371_M_UNIT_SPARE".M_CODES_SPARE.Ack_M503 )
      I_Contact( "DB2120_MPP_ITC_IPC".RESET_FAULTS )
      I_Contact( "DB371_M_UNIT_SPARE".M_CODES_SPARE.M_RESET_PULSE )
      Coil( "DB371_M_UNIT_SPARE".M_CODES_SPARE.M503 )
   END_RUNG
   RUNG wire#powerrail
      Contact( "DB371_M_UNIT_SPARE".M_CODES_SPARE.M503 )
   END_RUNG wire#w1
   // the same network as SCL:
   "DB371_M_UNIT_SPARE".M_CODES_SPARE.M503 := ("DB339_EXTENDED_M_SPARE".M_code[503] OR "DB371_M_UNIT_SPARE".M_CODES_SPARE.M503) AND NOT "DB371_M_UNIT_SPARE".M_CODES_SPARE.Ack_M503 AND NOT "DB2120_MPP_ITC_IPC".RESET_FAULTS AND NOT "DB371_M_UNIT_SPARE".M_CODES_SPARE.M_RESET_PULSE;
END_REGION

REGION Network 101: ACKNOWLEDGE M504-FIXTURE 2 VERIFY PART AND TOOL IS CLAMPED DURING MACHINING (WHEN TRUE DO). TOGGLED / ACKNOWLEDGE M46-VERIFY FIXTURE 1 PART AND TOOL IS CLAMPED DURING
   RUNG wire#powerrail
      Contact( "M_ZERO" )
      Coil( "DB371_M_UNIT_SPARE".M_CODES_SPARE.Ack_M504 )
   END_RUNG
   // the same network as SCL:
   "DB371_M_UNIT_SPARE".M_CODES_SPARE.Ack_M504 := "M_ZERO";
END_REGION

REGION Network 102: M504-FIXTURE 2 VERIFY PART AND TOOL IS CLAMPED DURING MACHINING (WHEN TRUE DO). TOGGLED / M46-VERIFY FIXTURE 1 PART AND TOOL IS CLAMPED DURING MACHINING
   RUNG wire#powerrail
      Contact( "DB339_EXTENDED_M_SPARE".M_code[504] )
      wire#w1
      I_Contact( "DB339_EXTENDED_M_SPARE".M_code[504] )
      wire#w2
      I_Contact( "DB371_M_UNIT_SPARE".M_CODES_SPARE.Ack_M504 )
      I_Contact( "DB2120_MPP_ITC_IPC".RESET_FAULTS )
      Contact( "DB2440_GLOBAL_DATA".GLOBAL_DATA.ANY_PART_CYCLE_RUN )
      Coil( "DB371_M_UNIT_SPARE".M_CODES_SPARE.M504 )
   END_RUNG
   RUNG wire#powerrail
      Contact( "DB371_M_UNIT_SPARE".M_CODES_SPARE.M504 )
   END_RUNG wire#w1
   RUNG wire#w1
      I_Contact( "DB371_M_UNIT_SPARE".M_CODES_SPARE.M504 )
   END_RUNG wire#w2
   // the same network as SCL:
   "DB371_M_UNIT_SPARE".M_CODES_SPARE.M504 := ("DB339_EXTENDED_M_SPARE".M_code[504] OR "DB371_M_UNIT_SPARE".M_CODES_SPARE.M504) AND (NOT "DB339_EXTENDED_M_SPARE".M_code[504] OR NOT "DB371_M_UNIT_SPARE".M_CODES_SPARE.M504) AND NOT "DB371_M_UNIT_SPARE".M_CODES_SPARE.Ack_M504 AND NOT "DB2120_MPP_ITC_IPC".RESET_FAULTS AND "DB2440_GLOBAL_DATA".GLOBAL_DATA.ANY_PART_CYCLE_RUN;
END_REGION

REGION Network 103: ACKNOWLEDGE M505-FIXTURE 2 VERIFY PART AND TOOL IS CLAMPED LOW PRESSURE DURING MACHINING (WHEN TRUE DO). TOGGLED / ACKNOWLEDGE M46-VERIFY FIXTURE 1 PART AND TOOL IS CLAMPED DURING
   RUNG wire#powerrail
      Contact( "M_ZERO" )
      Coil( "DB371_M_UNIT_SPARE".M_CODES_SPARE.Ack_M505 )
   END_RUNG
   // the same network as SCL:
   "DB371_M_UNIT_SPARE".M_CODES_SPARE.Ack_M505 := "M_ZERO";
END_REGION

REGION Network 104: M505-FIXTURE 2 VERIFY PART AND TOOL IS CLAMPED LOW PRESSURE DURING MACHINING (WHEN TRUE DO). TOGGLED / M46-VERIFY FIXTURE 1 PART AND TOOL IS CLAMPED DURING MACHINING
   RUNG wire#powerrail
      Contact( "DB339_EXTENDED_M_SPARE".M_code[505] )
      wire#w1
      I_Contact( "DB339_EXTENDED_M_SPARE".M_code[505] )
      wire#w2
      I_Contact( "DB371_M_UNIT_SPARE".M_CODES_SPARE.Ack_M505 )
      I_Contact( "DB2120_MPP_ITC_IPC".RESET_FAULTS )
      Contact( "DB2440_GLOBAL_DATA".GLOBAL_DATA.ANY_PART_CYCLE_RUN )
      Coil( "DB371_M_UNIT_SPARE".M_CODES_SPARE.M505 )
   END_RUNG
   RUNG wire#powerrail
      Contact( "DB371_M_UNIT_SPARE".M_CODES_SPARE.M505 )
   END_RUNG wire#w1
   RUNG wire#w1
      I_Contact( "DB371_M_UNIT_SPARE".M_CODES_SPARE.M505 )
   END_RUNG wire#w2
   // the same network as SCL:
   "DB371_M_UNIT_SPARE".M_CODES_SPARE.M505 := ("DB339_EXTENDED_M_SPARE".M_code[505] OR "DB371_M_UNIT_SPARE".M_CODES_SPARE.M505) AND (NOT "DB339_EXTENDED_M_SPARE".M_code[505] OR NOT "DB371_M_UNIT_SPARE".M_CODES_SPARE.M505) AND NOT "DB371_M_UNIT_SPARE".M_CODES_SPARE.Ack_M505 AND NOT "DB2120_MPP_ITC_IPC".RESET_FAULTS AND "DB2440_GLOBAL_DATA".GLOBAL_DATA.ANY_PART_CYCLE_RUN;
END_REGION

REGION Network 105: ACKNOWLEDGE M506-FIXTURE 2 VERIFY PARTS ARE UNCLAMPED PARTS LOADING (WHEN TRUE DO). TOGGLED / ACKNOWLEDGE M47-VERIFY FIXTURE 2 PART AND TOOL IS CLAMPED DURING
   RUNG wire#powerrail
      Contact( "M_ZERO" )
      Coil( "DB371_M_UNIT_SPARE".M_CODES_SPARE.Ack_M506 )
   END_RUNG
   // the same network as SCL:
   "DB371_M_UNIT_SPARE".M_CODES_SPARE.Ack_M506 := "M_ZERO";
END_REGION

REGION Network 106: M506-FIXTURE 2 VERIFY PARTS ARE UNCLAMPED PARTS LOADING (WHEN TRUE DO). TOGGLED / M47-VERIFY FIXTURE 2 PART AND TOOL IS CLAMPED DURING MACHINING
   RUNG wire#powerrail
      Contact( "DB339_EXTENDED_M_SPARE".M_code[506] )
      wire#w1
      I_Contact( "DB339_EXTENDED_M_SPARE".M_code[506] )
      wire#w2
      I_Contact( "DB371_M_UNIT_SPARE".M_CODES_SPARE.Ack_M506 )
      I_Contact( "DB2120_MPP_ITC_IPC".RESET_FAULTS )
      Contact( "DB2440_GLOBAL_DATA".GLOBAL_DATA.ANY_PART_CYCLE_RUN )
      Coil( "DB371_M_UNIT_SPARE".M_CODES_SPARE.M506 )
   END_RUNG
   RUNG wire#powerrail
      Contact( "DB371_M_UNIT_SPARE".M_CODES_SPARE.M506 )
   END_RUNG wire#w1
   RUNG wire#w1
      I_Contact( "DB371_M_UNIT_SPARE".M_CODES_SPARE.M506 )
   END_RUNG wire#w2
   // the same network as SCL:
   "DB371_M_UNIT_SPARE".M_CODES_SPARE.M506 := ("DB339_EXTENDED_M_SPARE".M_code[506] OR "DB371_M_UNIT_SPARE".M_CODES_SPARE.M506) AND (NOT "DB339_EXTENDED_M_SPARE".M_code[506] OR NOT "DB371_M_UNIT_SPARE".M_CODES_SPARE.M506) AND NOT "DB371_M_UNIT_SPARE".M_CODES_SPARE.Ack_M506 AND NOT "DB2120_MPP_ITC_IPC".RESET_FAULTS AND "DB2440_GLOBAL_DATA".GLOBAL_DATA.ANY_PART_CYCLE_RUN;
END_REGION

REGION Network 107: ACKNOWLEDGE M507-FIXTURE 2 VERIFY FIXTURE REMAINS CLAMPED
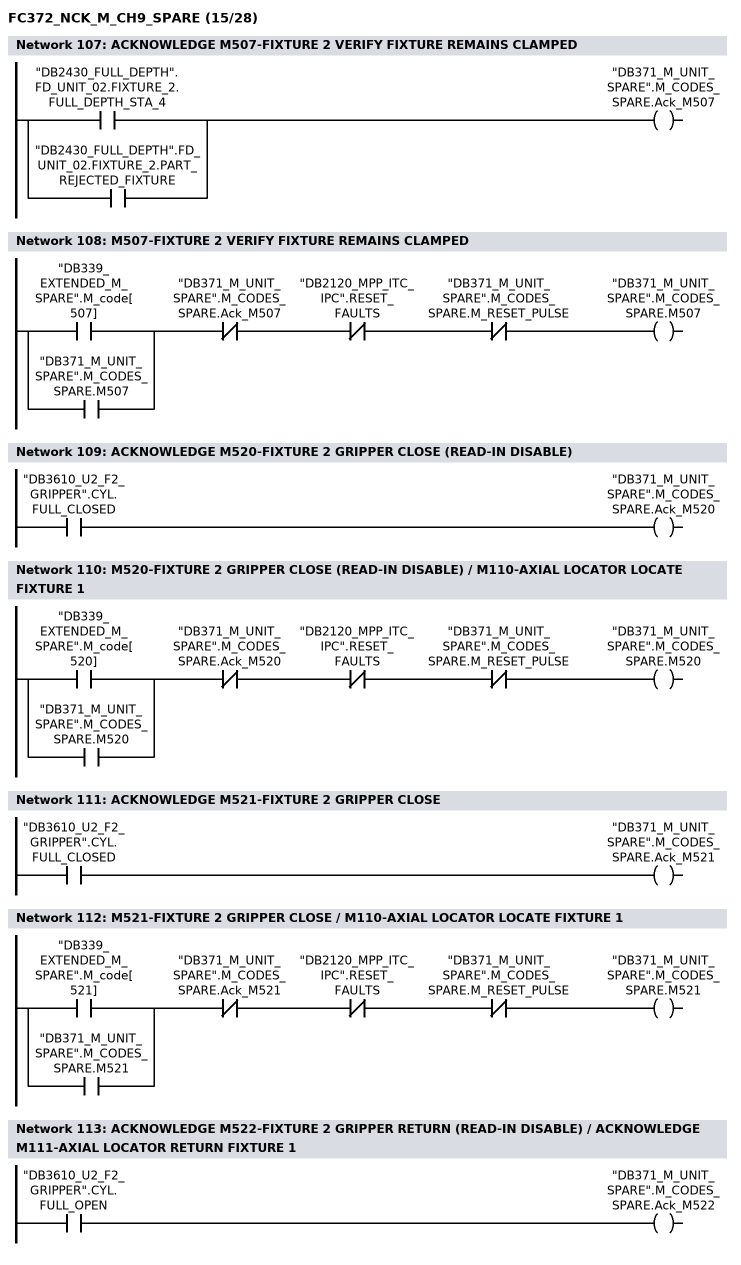
   RUNG wire#powerrail
      Contact( "DB2430_FULL_DEPTH".FD_UNIT_02.FIXTURE_2.FULL_DEPTH_STA_4 )
      wire#w1
      Coil( "DB371_M_UNIT_SPARE".M_CODES_SPARE.Ack_M507 )
   END_RUNG
   RUNG wire#powerrail
      Contact( "DB2430_FULL_DEPTH".FD_UNIT_02.FIXTURE_2.PART_REJECTED_FIXTURE )
   END_RUNG wire#w1
   // the same network as SCL:
   "DB371_M_UNIT_SPARE".M_CODES_SPARE.Ack_M507 := "DB2430_FULL_DEPTH".FD_UNIT_02.FIXTURE_2.FULL_DEPTH_STA_4 OR "DB2430_FULL_DEPTH".FD_UNIT_02.FIXTURE_2.PART_REJECTED_FIXTURE;
END_REGION

REGION Network 108: M507-FIXTURE 2 VERIFY FIXTURE REMAINS CLAMPED
   RUNG wire#powerrail
      Contact( "DB339_EXTENDED_M_SPARE".M_code[507] )
      wire#w1
      I_Contact( "DB371_M_UNIT_SPARE".M_CODES_SPARE.Ack_M507 )
      I_Contact( "DB2120_MPP_ITC_IPC".RESET_FAULTS )
      I_Contact( "DB371_M_UNIT_SPARE".M_CODES_SPARE.M_RESET_PULSE )
      Coil( "DB371_M_UNIT_SPARE".M_CODES_SPARE.M507 )
   END_RUNG
   RUNG wire#powerrail
      Contact( "DB371_M_UNIT_SPARE".M_CODES_SPARE.M507 )
   END_RUNG wire#w1
   // the same network as SCL:
   "DB371_M_UNIT_SPARE".M_CODES_SPARE.M507 := ("DB339_EXTENDED_M_SPARE".M_code[507] OR "DB371_M_UNIT_SPARE".M_CODES_SPARE.M507) AND NOT "DB371_M_UNIT_SPARE".M_CODES_SPARE.Ack_M507 AND NOT "DB2120_MPP_ITC_IPC".RESET_FAULTS AND NOT "DB371_M_UNIT_SPARE".M_CODES_SPARE.M_RESET_PULSE;
END_REGION

REGION Network 109: ACKNOWLEDGE M520-FIXTURE 2 GRIPPER CLOSE (READ-IN DISABLE)
   RUNG wire#powerrail
      Contact( "DB3610_U2_F2_GRIPPER".CYL.FULL_CLOSED )
      Coil( "DB371_M_UNIT_SPARE".M_CODES_SPARE.Ack_M520 )
   END_RUNG
   // the same network as SCL:
   "DB371_M_UNIT_SPARE".M_CODES_SPARE.Ack_M520 := "DB3610_U2_F2_GRIPPER".CYL.FULL_CLOSED;
END_REGION

REGION Network 110: M520-FIXTURE 2 GRIPPER CLOSE (READ-IN DISABLE) / M110-AXIAL LOCATOR LOCATE FIXTURE 1
   RUNG wire#powerrail
      Contact( "DB339_EXTENDED_M_SPARE".M_code[520] )
      wire#w1
      I_Contact( "DB371_M_UNIT_SPARE".M_CODES_SPARE.Ack_M520 )
      I_Contact( "DB2120_MPP_ITC_IPC".RESET_FAULTS )
      I_Contact( "DB371_M_UNIT_SPARE".M_CODES_SPARE.M_RESET_PULSE )
      Coil( "DB371_M_UNIT_SPARE".M_CODES_SPARE.M520 )
   END_RUNG
   RUNG wire#powerrail
      Contact( "DB371_M_UNIT_SPARE".M_CODES_SPARE.M520 )
   END_RUNG wire#w1
   // the same network as SCL:
   "DB371_M_UNIT_SPARE".M_CODES_SPARE.M520 := ("DB339_EXTENDED_M_SPARE".M_code[520] OR "DB371_M_UNIT_SPARE".M_CODES_SPARE.M520) AND NOT "DB371_M_UNIT_SPARE".M_CODES_SPARE.Ack_M520 AND NOT "DB2120_MPP_ITC_IPC".RESET_FAULTS AND NOT "DB371_M_UNIT_SPARE".M_CODES_SPARE.M_RESET_PULSE;
END_REGION

REGION Network 111: ACKNOWLEDGE M521-FIXTURE 2 GRIPPER CLOSE
   RUNG wire#powerrail
      Contact( "DB3610_U2_F2_GRIPPER".CYL.FULL_CLOSED )
      Coil( "DB371_M_UNIT_SPARE".M_CODES_SPARE.Ack_M521 )
   END_RUNG
   // the same network as SCL:
   "DB371_M_UNIT_SPARE".M_CODES_SPARE.Ack_M521 := "DB3610_U2_F2_GRIPPER".CYL.FULL_CLOSED;
END_REGION

REGION Network 112: M521-FIXTURE 2 GRIPPER CLOSE / M110-AXIAL LOCATOR LOCATE FIXTURE 1
   RUNG wire#powerrail
      Contact( "DB339_EXTENDED_M_SPARE".M_code[521] )
      wire#w1
      I_Contact( "DB371_M_UNIT_SPARE".M_CODES_SPARE.Ack_M521 )
      I_Contact( "DB2120_MPP_ITC_IPC".RESET_FAULTS )
      I_Contact( "DB371_M_UNIT_SPARE".M_CODES_SPARE.M_RESET_PULSE )
      Coil( "DB371_M_UNIT_SPARE".M_CODES_SPARE.M521 )
   END_RUNG
   RUNG wire#powerrail
      Contact( "DB371_M_UNIT_SPARE".M_CODES_SPARE.M521 )
   END_RUNG wire#w1
   // the same network as SCL:
   "DB371_M_UNIT_SPARE".M_CODES_SPARE.M521 := ("DB339_EXTENDED_M_SPARE".M_code[521] OR "DB371_M_UNIT_SPARE".M_CODES_SPARE.M521) AND NOT "DB371_M_UNIT_SPARE".M_CODES_SPARE.Ack_M521 AND NOT "DB2120_MPP_ITC_IPC".RESET_FAULTS AND NOT "DB371_M_UNIT_SPARE".M_CODES_SPARE.M_RESET_PULSE;
END_REGION

REGION Network 113: ACKNOWLEDGE M522-FIXTURE 2 GRIPPER RETURN (READ-IN DISABLE) / ACKNOWLEDGE M111-AXIAL LOCATOR RETURN FIXTURE 1
   RUNG wire#powerrail
      Contact( "DB3610_U2_F2_GRIPPER".CYL.FULL_OPEN )
      Coil( "DB371_M_UNIT_SPARE".M_CODES_SPARE.Ack_M522 )
   END_RUNG
   // the same network as SCL:
   "DB371_M_UNIT_SPARE".M_CODES_SPARE.Ack_M522 := "DB3610_U2_F2_GRIPPER".CYL.FULL_OPEN;
END_REGION

REGION Network 114: M522-FIXTURE 2 GRIPPER RETURN (READ-IN DISABLE) / M111-AXIAL LOCATOR RETURN FIXTURE 1
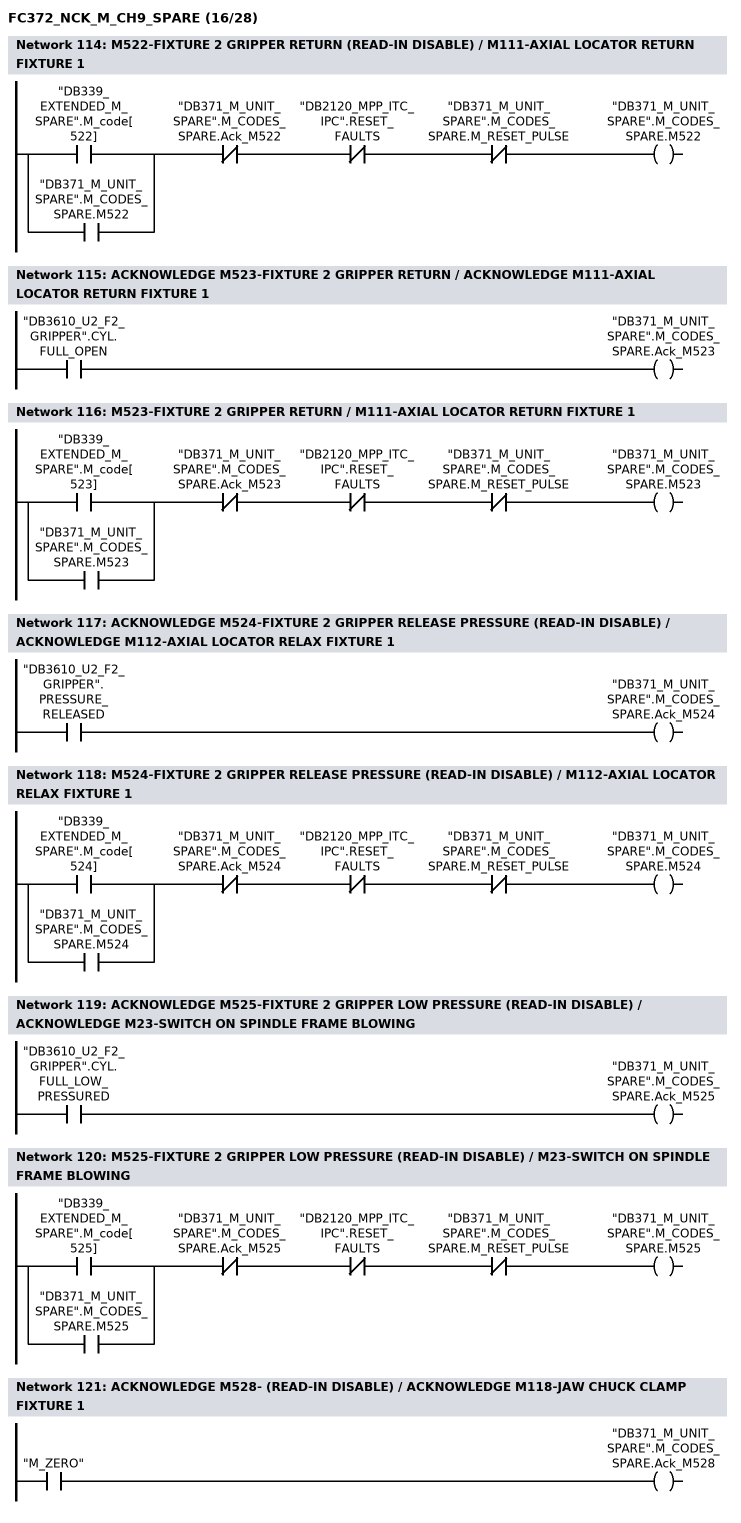
   RUNG wire#powerrail
      Contact( "DB339_EXTENDED_M_SPARE".M_code[522] )
      wire#w1
      I_Contact( "DB371_M_UNIT_SPARE".M_CODES_SPARE.Ack_M522 )
      I_Contact( "DB2120_MPP_ITC_IPC".RESET_FAULTS )
      I_Contact( "DB371_M_UNIT_SPARE".M_CODES_SPARE.M_RESET_PULSE )
      Coil( "DB371_M_UNIT_SPARE".M_CODES_SPARE.M522 )
   END_RUNG
   RUNG wire#powerrail
      Contact( "DB371_M_UNIT_SPARE".M_CODES_SPARE.M522 )
   END_RUNG wire#w1
   // the same network as SCL:
   "DB371_M_UNIT_SPARE".M_CODES_SPARE.M522 := ("DB339_EXTENDED_M_SPARE".M_code[522] OR "DB371_M_UNIT_SPARE".M_CODES_SPARE.M522) AND NOT "DB371_M_UNIT_SPARE".M_CODES_SPARE.Ack_M522 AND NOT "DB2120_MPP_ITC_IPC".RESET_FAULTS AND NOT "DB371_M_UNIT_SPARE".M_CODES_SPARE.M_RESET_PULSE;
END_REGION

REGION Network 115: ACKNOWLEDGE M523-FIXTURE 2 GRIPPER RETURN / ACKNOWLEDGE M111-AXIAL LOCATOR RETURN FIXTURE 1
   RUNG wire#powerrail
      Contact( "DB3610_U2_F2_GRIPPER".CYL.FULL_OPEN )
      Coil( "DB371_M_UNIT_SPARE".M_CODES_SPARE.Ack_M523 )
   END_RUNG
   // the same network as SCL:
   "DB371_M_UNIT_SPARE".M_CODES_SPARE.Ack_M523 := "DB3610_U2_F2_GRIPPER".CYL.FULL_OPEN;
END_REGION

REGION Network 116: M523-FIXTURE 2 GRIPPER RETURN / M111-AXIAL LOCATOR RETURN FIXTURE 1
   RUNG wire#powerrail
      Contact( "DB339_EXTENDED_M_SPARE".M_code[523] )
      wire#w1
      I_Contact( "DB371_M_UNIT_SPARE".M_CODES_SPARE.Ack_M523 )
      I_Contact( "DB2120_MPP_ITC_IPC".RESET_FAULTS )
      I_Contact( "DB371_M_UNIT_SPARE".M_CODES_SPARE.M_RESET_PULSE )
      Coil( "DB371_M_UNIT_SPARE".M_CODES_SPARE.M523 )
   END_RUNG
   RUNG wire#powerrail
      Contact( "DB371_M_UNIT_SPARE".M_CODES_SPARE.M523 )
   END_RUNG wire#w1
   // the same network as SCL:
   "DB371_M_UNIT_SPARE".M_CODES_SPARE.M523 := ("DB339_EXTENDED_M_SPARE".M_code[523] OR "DB371_M_UNIT_SPARE".M_CODES_SPARE.M523) AND NOT "DB371_M_UNIT_SPARE".M_CODES_SPARE.Ack_M523 AND NOT "DB2120_MPP_ITC_IPC".RESET_FAULTS AND NOT "DB371_M_UNIT_SPARE".M_CODES_SPARE.M_RESET_PULSE;
END_REGION

REGION Network 117: ACKNOWLEDGE M524-FIXTURE 2 GRIPPER RELEASE PRESSURE (READ-IN DISABLE) / ACKNOWLEDGE M112-AXIAL LOCATOR RELAX FIXTURE 1
   RUNG wire#powerrail
      Contact( "DB3610_U2_F2_GRIPPER".PRESSURE_RELEASED )
      Coil( "DB371_M_UNIT_SPARE".M_CODES_SPARE.Ack_M524 )
   END_RUNG
   // the same network as SCL:
   "DB371_M_UNIT_SPARE".M_CODES_SPARE.Ack_M524 := "DB3610_U2_F2_GRIPPER".PRESSURE_RELEASED;
END_REGION

REGION Network 118: M524-FIXTURE 2 GRIPPER RELEASE PRESSURE (READ-IN DISABLE) / M112-AXIAL LOCATOR RELAX FIXTURE 1
   RUNG wire#powerrail
      Contact( "DB339_EXTENDED_M_SPARE".M_code[524] )
      wire#w1
      I_Contact( "DB371_M_UNIT_SPARE".M_CODES_SPARE.Ack_M524 )
      I_Contact( "DB2120_MPP_ITC_IPC".RESET_FAULTS )
      I_Contact( "DB371_M_UNIT_SPARE".M_CODES_SPARE.M_RESET_PULSE )
      Coil( "DB371_M_UNIT_SPARE".M_CODES_SPARE.M524 )
   END_RUNG
   RUNG wire#powerrail
      Contact( "DB371_M_UNIT_SPARE".M_CODES_SPARE.M524 )
   END_RUNG wire#w1
   // the same network as SCL:
   "DB371_M_UNIT_SPARE".M_CODES_SPARE.M524 := ("DB339_EXTENDED_M_SPARE".M_code[524] OR "DB371_M_UNIT_SPARE".M_CODES_SPARE.M524) AND NOT "DB371_M_UNIT_SPARE".M_CODES_SPARE.Ack_M524 AND NOT "DB2120_MPP_ITC_IPC".RESET_FAULTS AND NOT "DB371_M_UNIT_SPARE".M_CODES_SPARE.M_RESET_PULSE;
END_REGION

REGION Network 119: ACKNOWLEDGE M525-FIXTURE 2 GRIPPER LOW PRESSURE (READ-IN DISABLE) / ACKNOWLEDGE M23-SWITCH ON SPINDLE FRAME BLOWING
   RUNG wire#powerrail
      Contact( "DB3610_U2_F2_GRIPPER".CYL.FULL_LOW_PRESSURED )
      Coil( "DB371_M_UNIT_SPARE".M_CODES_SPARE.Ack_M525 )
   END_RUNG
   // the same network as SCL:
   "DB371_M_UNIT_SPARE".M_CODES_SPARE.Ack_M525 := "DB3610_U2_F2_GRIPPER".CYL.FULL_LOW_PRESSURED;
END_REGION

REGION Network 120: M525-FIXTURE 2 GRIPPER LOW PRESSURE (READ-IN DISABLE) / M23-SWITCH ON SPINDLE FRAME BLOWING
   RUNG wire#powerrail
      Contact( "DB339_EXTENDED_M_SPARE".M_code[525] )
      wire#w1
      I_Contact( "DB371_M_UNIT_SPARE".M_CODES_SPARE.Ack_M525 )
      I_Contact( "DB2120_MPP_ITC_IPC".RESET_FAULTS )
      I_Contact( "DB371_M_UNIT_SPARE".M_CODES_SPARE.M_RESET_PULSE )
      Coil( "DB371_M_UNIT_SPARE".M_CODES_SPARE.M525 )
   END_RUNG
   RUNG wire#powerrail
      Contact( "DB371_M_UNIT_SPARE".M_CODES_SPARE.M525 )
   END_RUNG wire#w1
   // the same network as SCL:
   "DB371_M_UNIT_SPARE".M_CODES_SPARE.M525 := ("DB339_EXTENDED_M_SPARE".M_code[525] OR "DB371_M_UNIT_SPARE".M_CODES_SPARE.M525) AND NOT "DB371_M_UNIT_SPARE".M_CODES_SPARE.Ack_M525 AND NOT "DB2120_MPP_ITC_IPC".RESET_FAULTS AND NOT "DB371_M_UNIT_SPARE".M_CODES_SPARE.M_RESET_PULSE;
END_REGION

REGION Network 121: ACKNOWLEDGE M528- (READ-IN DISABLE) / ACKNOWLEDGE M118-JAW CHUCK CLAMP FIXTURE 1
   RUNG wire#powerrail
      Contact( "M_ZERO" )
      Coil( "DB371_M_UNIT_SPARE".M_CODES_SPARE.Ack_M528 )
   END_RUNG
   // the same network as SCL:
   "DB371_M_UNIT_SPARE".M_CODES_SPARE.Ack_M528 := "M_ZERO";
END_REGION

REGION Network 122: M528- (READ-IN DISABLE) / M118-JAW CHUCK CLAMP FIXTURE 1
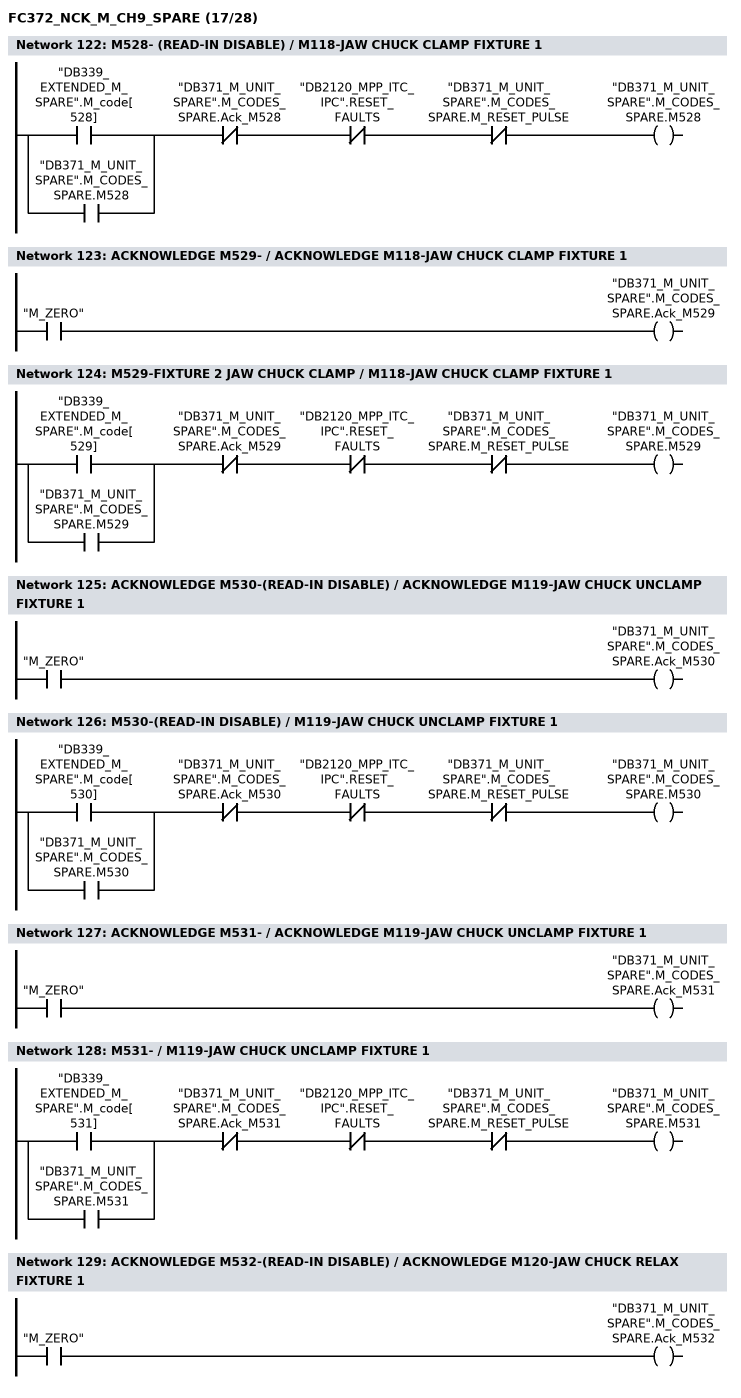
   RUNG wire#powerrail
      Contact( "DB339_EXTENDED_M_SPARE".M_code[528] )
      wire#w1
      I_Contact( "DB371_M_UNIT_SPARE".M_CODES_SPARE.Ack_M528 )
      I_Contact( "DB2120_MPP_ITC_IPC".RESET_FAULTS )
      I_Contact( "DB371_M_UNIT_SPARE".M_CODES_SPARE.M_RESET_PULSE )
      Coil( "DB371_M_UNIT_SPARE".M_CODES_SPARE.M528 )
   END_RUNG
   RUNG wire#powerrail
      Contact( "DB371_M_UNIT_SPARE".M_CODES_SPARE.M528 )
   END_RUNG wire#w1
   // the same network as SCL:
   "DB371_M_UNIT_SPARE".M_CODES_SPARE.M528 := ("DB339_EXTENDED_M_SPARE".M_code[528] OR "DB371_M_UNIT_SPARE".M_CODES_SPARE.M528) AND NOT "DB371_M_UNIT_SPARE".M_CODES_SPARE.Ack_M528 AND NOT "DB2120_MPP_ITC_IPC".RESET_FAULTS AND NOT "DB371_M_UNIT_SPARE".M_CODES_SPARE.M_RESET_PULSE;
END_REGION

REGION Network 123: ACKNOWLEDGE M529- / ACKNOWLEDGE M118-JAW CHUCK CLAMP FIXTURE 1
   RUNG wire#powerrail
      Contact( "M_ZERO" )
      Coil( "DB371_M_UNIT_SPARE".M_CODES_SPARE.Ack_M529 )
   END_RUNG
   // the same network as SCL:
   "DB371_M_UNIT_SPARE".M_CODES_SPARE.Ack_M529 := "M_ZERO";
END_REGION

REGION Network 124: M529-FIXTURE 2 JAW CHUCK CLAMP / M118-JAW CHUCK CLAMP FIXTURE 1
   RUNG wire#powerrail
      Contact( "DB339_EXTENDED_M_SPARE".M_code[529] )
      wire#w1
      I_Contact( "DB371_M_UNIT_SPARE".M_CODES_SPARE.Ack_M529 )
      I_Contact( "DB2120_MPP_ITC_IPC".RESET_FAULTS )
      I_Contact( "DB371_M_UNIT_SPARE".M_CODES_SPARE.M_RESET_PULSE )
      Coil( "DB371_M_UNIT_SPARE".M_CODES_SPARE.M529 )
   END_RUNG
   RUNG wire#powerrail
      Contact( "DB371_M_UNIT_SPARE".M_CODES_SPARE.M529 )
   END_RUNG wire#w1
   // the same network as SCL:
   "DB371_M_UNIT_SPARE".M_CODES_SPARE.M529 := ("DB339_EXTENDED_M_SPARE".M_code[529] OR "DB371_M_UNIT_SPARE".M_CODES_SPARE.M529) AND NOT "DB371_M_UNIT_SPARE".M_CODES_SPARE.Ack_M529 AND NOT "DB2120_MPP_ITC_IPC".RESET_FAULTS AND NOT "DB371_M_UNIT_SPARE".M_CODES_SPARE.M_RESET_PULSE;
END_REGION

REGION Network 125: ACKNOWLEDGE M530-(READ-IN DISABLE) / ACKNOWLEDGE M119-JAW CHUCK UNCLAMP FIXTURE 1
   RUNG wire#powerrail
      Contact( "M_ZERO" )
      Coil( "DB371_M_UNIT_SPARE".M_CODES_SPARE.Ack_M530 )
   END_RUNG
   // the same network as SCL:
   "DB371_M_UNIT_SPARE".M_CODES_SPARE.Ack_M530 := "M_ZERO";
END_REGION

REGION Network 126: M530-(READ-IN DISABLE) / M119-JAW CHUCK UNCLAMP FIXTURE 1
   RUNG wire#powerrail
      Contact( "DB339_EXTENDED_M_SPARE".M_code[530] )
      wire#w1
      I_Contact( "DB371_M_UNIT_SPARE".M_CODES_SPARE.Ack_M530 )
      I_Contact( "DB2120_MPP_ITC_IPC".RESET_FAULTS )
      I_Contact( "DB371_M_UNIT_SPARE".M_CODES_SPARE.M_RESET_PULSE )
      Coil( "DB371_M_UNIT_SPARE".M_CODES_SPARE.M530 )
   END_RUNG
   RUNG wire#powerrail
      Contact( "DB371_M_UNIT_SPARE".M_CODES_SPARE.M530 )
   END_RUNG wire#w1
   // the same network as SCL:
   "DB371_M_UNIT_SPARE".M_CODES_SPARE.M530 := ("DB339_EXTENDED_M_SPARE".M_code[530] OR "DB371_M_UNIT_SPARE".M_CODES_SPARE.M530) AND NOT "DB371_M_UNIT_SPARE".M_CODES_SPARE.Ack_M530 AND NOT "DB2120_MPP_ITC_IPC".RESET_FAULTS AND NOT "DB371_M_UNIT_SPARE".M_CODES_SPARE.M_RESET_PULSE;
END_REGION

REGION Network 127: ACKNOWLEDGE M531- / ACKNOWLEDGE M119-JAW CHUCK UNCLAMP FIXTURE 1
   RUNG wire#powerrail
      Contact( "M_ZERO" )
      Coil( "DB371_M_UNIT_SPARE".M_CODES_SPARE.Ack_M531 )
   END_RUNG
   // the same network as SCL:
   "DB371_M_UNIT_SPARE".M_CODES_SPARE.Ack_M531 := "M_ZERO";
END_REGION

REGION Network 128: M531- / M119-JAW CHUCK UNCLAMP FIXTURE 1
   RUNG wire#powerrail
      Contact( "DB339_EXTENDED_M_SPARE".M_code[531] )
      wire#w1
      I_Contact( "DB371_M_UNIT_SPARE".M_CODES_SPARE.Ack_M531 )
      I_Contact( "DB2120_MPP_ITC_IPC".RESET_FAULTS )
      I_Contact( "DB371_M_UNIT_SPARE".M_CODES_SPARE.M_RESET_PULSE )
      Coil( "DB371_M_UNIT_SPARE".M_CODES_SPARE.M531 )
   END_RUNG
   RUNG wire#powerrail
      Contact( "DB371_M_UNIT_SPARE".M_CODES_SPARE.M531 )
   END_RUNG wire#w1
   // the same network as SCL:
   "DB371_M_UNIT_SPARE".M_CODES_SPARE.M531 := ("DB339_EXTENDED_M_SPARE".M_code[531] OR "DB371_M_UNIT_SPARE".M_CODES_SPARE.M531) AND NOT "DB371_M_UNIT_SPARE".M_CODES_SPARE.Ack_M531 AND NOT "DB2120_MPP_ITC_IPC".RESET_FAULTS AND NOT "DB371_M_UNIT_SPARE".M_CODES_SPARE.M_RESET_PULSE;
END_REGION

REGION Network 129: ACKNOWLEDGE M532-(READ-IN DISABLE) / ACKNOWLEDGE M120-JAW CHUCK RELAX FIXTURE 1
   RUNG wire#powerrail
      Contact( "M_ZERO" )
      Coil( "DB371_M_UNIT_SPARE".M_CODES_SPARE.Ack_M532 )
   END_RUNG
   // the same network as SCL:
   "DB371_M_UNIT_SPARE".M_CODES_SPARE.Ack_M532 := "M_ZERO";
END_REGION

REGION Network 130: M532- (READ-IN DISABLE) / M120-JAW CHUCK RELAX FIXTURE 1
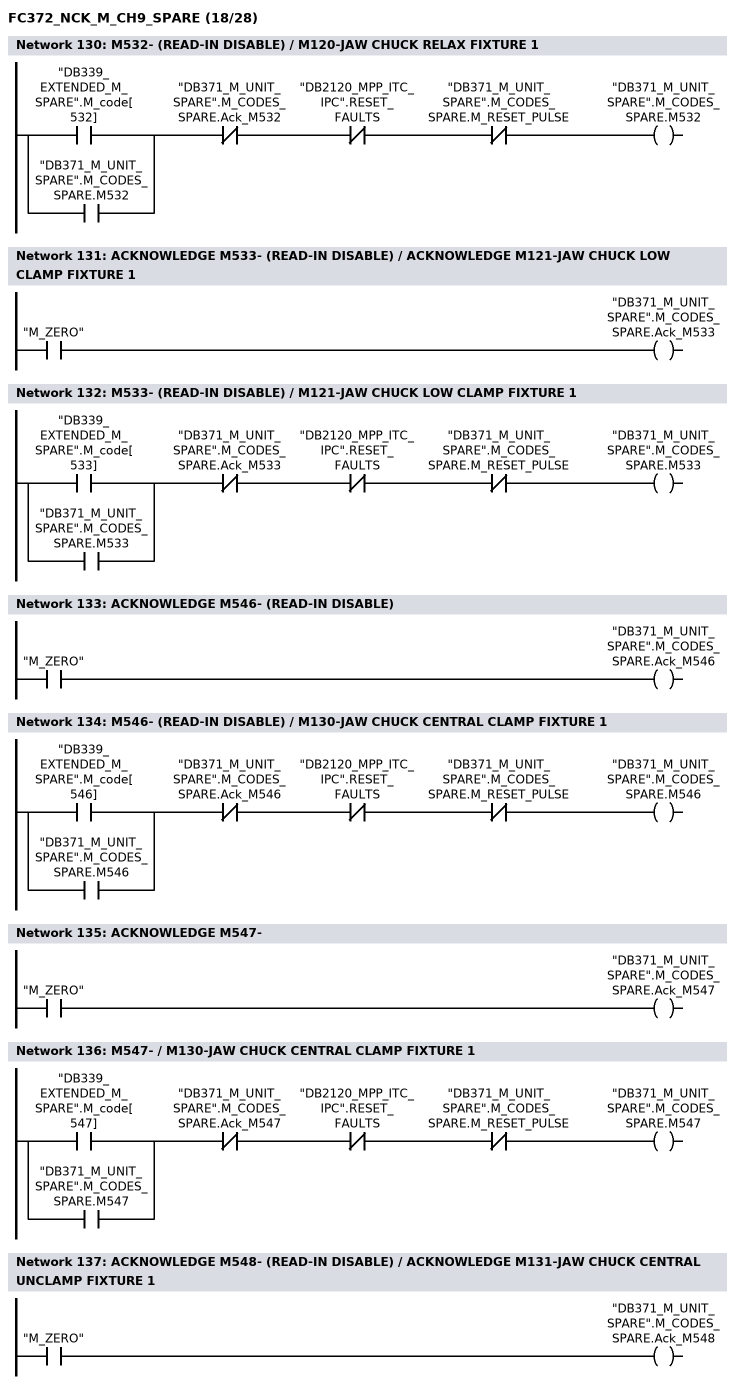
   RUNG wire#powerrail
      Contact( "DB339_EXTENDED_M_SPARE".M_code[532] )
      wire#w1
      I_Contact( "DB371_M_UNIT_SPARE".M_CODES_SPARE.Ack_M532 )
      I_Contact( "DB2120_MPP_ITC_IPC".RESET_FAULTS )
      I_Contact( "DB371_M_UNIT_SPARE".M_CODES_SPARE.M_RESET_PULSE )
      Coil( "DB371_M_UNIT_SPARE".M_CODES_SPARE.M532 )
   END_RUNG
   RUNG wire#powerrail
      Contact( "DB371_M_UNIT_SPARE".M_CODES_SPARE.M532 )
   END_RUNG wire#w1
   // the same network as SCL:
   "DB371_M_UNIT_SPARE".M_CODES_SPARE.M532 := ("DB339_EXTENDED_M_SPARE".M_code[532] OR "DB371_M_UNIT_SPARE".M_CODES_SPARE.M532) AND NOT "DB371_M_UNIT_SPARE".M_CODES_SPARE.Ack_M532 AND NOT "DB2120_MPP_ITC_IPC".RESET_FAULTS AND NOT "DB371_M_UNIT_SPARE".M_CODES_SPARE.M_RESET_PULSE;
END_REGION

REGION Network 131: ACKNOWLEDGE M533- (READ-IN DISABLE) / ACKNOWLEDGE M121-JAW CHUCK LOW CLAMP FIXTURE 1
   RUNG wire#powerrail
      Contact( "M_ZERO" )
      Coil( "DB371_M_UNIT_SPARE".M_CODES_SPARE.Ack_M533 )
   END_RUNG
   // the same network as SCL:
   "DB371_M_UNIT_SPARE".M_CODES_SPARE.Ack_M533 := "M_ZERO";
END_REGION

REGION Network 132: M533- (READ-IN DISABLE) / M121-JAW CHUCK LOW CLAMP FIXTURE 1
   RUNG wire#powerrail
      Contact( "DB339_EXTENDED_M_SPARE".M_code[533] )
      wire#w1
      I_Contact( "DB371_M_UNIT_SPARE".M_CODES_SPARE.Ack_M533 )
      I_Contact( "DB2120_MPP_ITC_IPC".RESET_FAULTS )
      I_Contact( "DB371_M_UNIT_SPARE".M_CODES_SPARE.M_RESET_PULSE )
      Coil( "DB371_M_UNIT_SPARE".M_CODES_SPARE.M533 )
   END_RUNG
   RUNG wire#powerrail
      Contact( "DB371_M_UNIT_SPARE".M_CODES_SPARE.M533 )
   END_RUNG wire#w1
   // the same network as SCL:
   "DB371_M_UNIT_SPARE".M_CODES_SPARE.M533 := ("DB339_EXTENDED_M_SPARE".M_code[533] OR "DB371_M_UNIT_SPARE".M_CODES_SPARE.M533) AND NOT "DB371_M_UNIT_SPARE".M_CODES_SPARE.Ack_M533 AND NOT "DB2120_MPP_ITC_IPC".RESET_FAULTS AND NOT "DB371_M_UNIT_SPARE".M_CODES_SPARE.M_RESET_PULSE;
END_REGION

REGION Network 133: ACKNOWLEDGE M546- (READ-IN DISABLE)
   RUNG wire#powerrail
      Contact( "M_ZERO" )
      Coil( "DB371_M_UNIT_SPARE".M_CODES_SPARE.Ack_M546 )
   END_RUNG
   // the same network as SCL:
   "DB371_M_UNIT_SPARE".M_CODES_SPARE.Ack_M546 := "M_ZERO";
END_REGION

REGION Network 134: M546- (READ-IN DISABLE) / M130-JAW CHUCK CENTRAL CLAMP FIXTURE 1
   RUNG wire#powerrail
      Contact( "DB339_EXTENDED_M_SPARE".M_code[546] )
      wire#w1
      I_Contact( "DB371_M_UNIT_SPARE".M_CODES_SPARE.Ack_M546 )
      I_Contact( "DB2120_MPP_ITC_IPC".RESET_FAULTS )
      I_Contact( "DB371_M_UNIT_SPARE".M_CODES_SPARE.M_RESET_PULSE )
      Coil( "DB371_M_UNIT_SPARE".M_CODES_SPARE.M546 )
   END_RUNG
   RUNG wire#powerrail
      Contact( "DB371_M_UNIT_SPARE".M_CODES_SPARE.M546 )
   END_RUNG wire#w1
   // the same network as SCL:
   "DB371_M_UNIT_SPARE".M_CODES_SPARE.M546 := ("DB339_EXTENDED_M_SPARE".M_code[546] OR "DB371_M_UNIT_SPARE".M_CODES_SPARE.M546) AND NOT "DB371_M_UNIT_SPARE".M_CODES_SPARE.Ack_M546 AND NOT "DB2120_MPP_ITC_IPC".RESET_FAULTS AND NOT "DB371_M_UNIT_SPARE".M_CODES_SPARE.M_RESET_PULSE;
END_REGION

REGION Network 135: ACKNOWLEDGE M547-
   RUNG wire#powerrail
      Contact( "M_ZERO" )
      Coil( "DB371_M_UNIT_SPARE".M_CODES_SPARE.Ack_M547 )
   END_RUNG
   // the same network as SCL:
   "DB371_M_UNIT_SPARE".M_CODES_SPARE.Ack_M547 := "M_ZERO";
END_REGION

REGION Network 136: M547- / M130-JAW CHUCK CENTRAL CLAMP FIXTURE 1
   RUNG wire#powerrail
      Contact( "DB339_EXTENDED_M_SPARE".M_code[547] )
      wire#w1
      I_Contact( "DB371_M_UNIT_SPARE".M_CODES_SPARE.Ack_M547 )
      I_Contact( "DB2120_MPP_ITC_IPC".RESET_FAULTS )
      I_Contact( "DB371_M_UNIT_SPARE".M_CODES_SPARE.M_RESET_PULSE )
      Coil( "DB371_M_UNIT_SPARE".M_CODES_SPARE.M547 )
   END_RUNG
   RUNG wire#powerrail
      Contact( "DB371_M_UNIT_SPARE".M_CODES_SPARE.M547 )
   END_RUNG wire#w1
   // the same network as SCL:
   "DB371_M_UNIT_SPARE".M_CODES_SPARE.M547 := ("DB339_EXTENDED_M_SPARE".M_code[547] OR "DB371_M_UNIT_SPARE".M_CODES_SPARE.M547) AND NOT "DB371_M_UNIT_SPARE".M_CODES_SPARE.Ack_M547 AND NOT "DB2120_MPP_ITC_IPC".RESET_FAULTS AND NOT "DB371_M_UNIT_SPARE".M_CODES_SPARE.M_RESET_PULSE;
END_REGION

REGION Network 137: ACKNOWLEDGE M548- (READ-IN DISABLE) / ACKNOWLEDGE M131-JAW CHUCK CENTRAL UNCLAMP FIXTURE 1
   RUNG wire#powerrail
      Contact( "M_ZERO" )
      Coil( "DB371_M_UNIT_SPARE".M_CODES_SPARE.Ack_M548 )
   END_RUNG
   // the same network as SCL:
   "DB371_M_UNIT_SPARE".M_CODES_SPARE.Ack_M548 := "M_ZERO";
END_REGION

REGION Network 138: M548- (READ-IN DISABLE) / M131-JAW CHUCK CENTRAL UNCLAMP FIXTURE 1
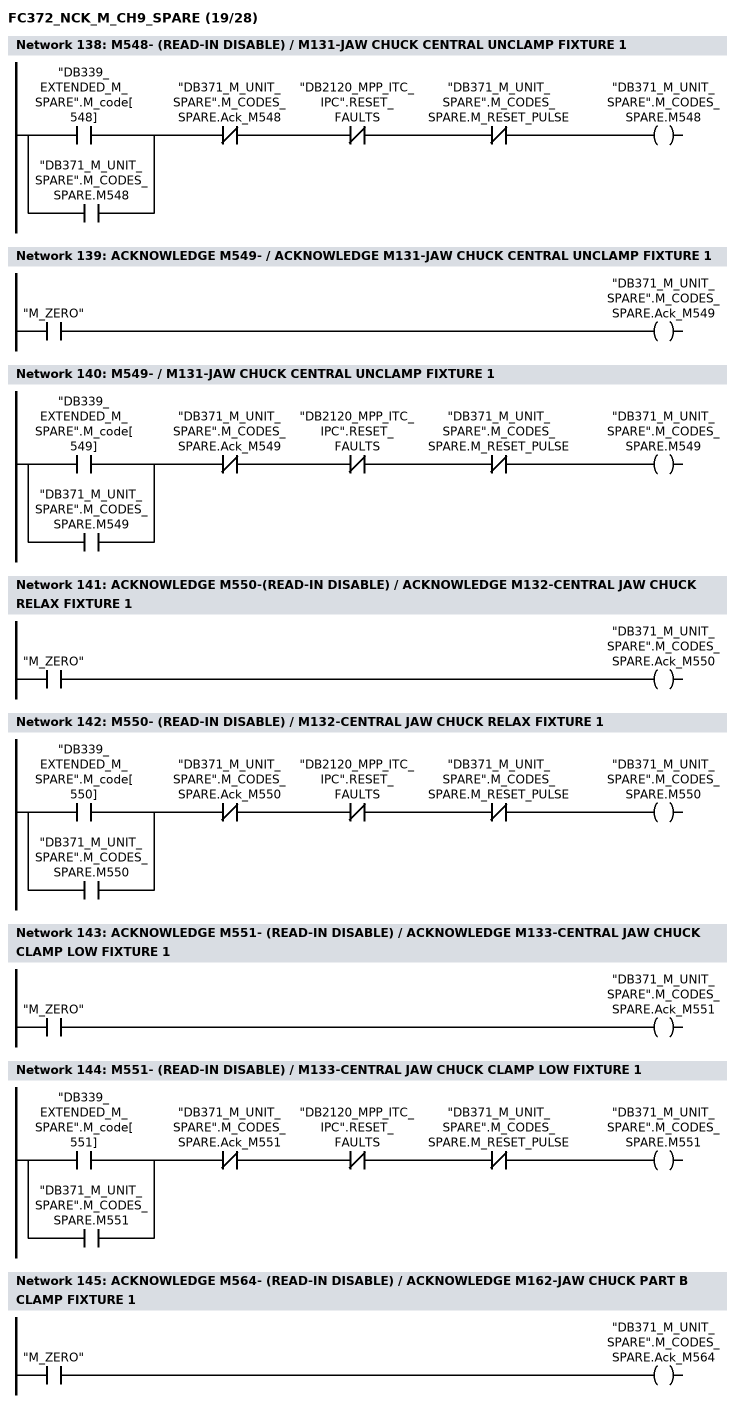
   RUNG wire#powerrail
      Contact( "DB339_EXTENDED_M_SPARE".M_code[548] )
      wire#w1
      I_Contact( "DB371_M_UNIT_SPARE".M_CODES_SPARE.Ack_M548 )
      I_Contact( "DB2120_MPP_ITC_IPC".RESET_FAULTS )
      I_Contact( "DB371_M_UNIT_SPARE".M_CODES_SPARE.M_RESET_PULSE )
      Coil( "DB371_M_UNIT_SPARE".M_CODES_SPARE.M548 )
   END_RUNG
   RUNG wire#powerrail
      Contact( "DB371_M_UNIT_SPARE".M_CODES_SPARE.M548 )
   END_RUNG wire#w1
   // the same network as SCL:
   "DB371_M_UNIT_SPARE".M_CODES_SPARE.M548 := ("DB339_EXTENDED_M_SPARE".M_code[548] OR "DB371_M_UNIT_SPARE".M_CODES_SPARE.M548) AND NOT "DB371_M_UNIT_SPARE".M_CODES_SPARE.Ack_M548 AND NOT "DB2120_MPP_ITC_IPC".RESET_FAULTS AND NOT "DB371_M_UNIT_SPARE".M_CODES_SPARE.M_RESET_PULSE;
END_REGION

REGION Network 139: ACKNOWLEDGE M549- / ACKNOWLEDGE M131-JAW CHUCK CENTRAL UNCLAMP FIXTURE 1
   RUNG wire#powerrail
      Contact( "M_ZERO" )
      Coil( "DB371_M_UNIT_SPARE".M_CODES_SPARE.Ack_M549 )
   END_RUNG
   // the same network as SCL:
   "DB371_M_UNIT_SPARE".M_CODES_SPARE.Ack_M549 := "M_ZERO";
END_REGION

REGION Network 140: M549- / M131-JAW CHUCK CENTRAL UNCLAMP FIXTURE 1
   RUNG wire#powerrail
      Contact( "DB339_EXTENDED_M_SPARE".M_code[549] )
      wire#w1
      I_Contact( "DB371_M_UNIT_SPARE".M_CODES_SPARE.Ack_M549 )
      I_Contact( "DB2120_MPP_ITC_IPC".RESET_FAULTS )
      I_Contact( "DB371_M_UNIT_SPARE".M_CODES_SPARE.M_RESET_PULSE )
      Coil( "DB371_M_UNIT_SPARE".M_CODES_SPARE.M549 )
   END_RUNG
   RUNG wire#powerrail
      Contact( "DB371_M_UNIT_SPARE".M_CODES_SPARE.M549 )
   END_RUNG wire#w1
   // the same network as SCL:
   "DB371_M_UNIT_SPARE".M_CODES_SPARE.M549 := ("DB339_EXTENDED_M_SPARE".M_code[549] OR "DB371_M_UNIT_SPARE".M_CODES_SPARE.M549) AND NOT "DB371_M_UNIT_SPARE".M_CODES_SPARE.Ack_M549 AND NOT "DB2120_MPP_ITC_IPC".RESET_FAULTS AND NOT "DB371_M_UNIT_SPARE".M_CODES_SPARE.M_RESET_PULSE;
END_REGION

REGION Network 141: ACKNOWLEDGE M550-(READ-IN DISABLE) / ACKNOWLEDGE M132-CENTRAL JAW CHUCK RELAX FIXTURE 1
   RUNG wire#powerrail
      Contact( "M_ZERO" )
      Coil( "DB371_M_UNIT_SPARE".M_CODES_SPARE.Ack_M550 )
   END_RUNG
   // the same network as SCL:
   "DB371_M_UNIT_SPARE".M_CODES_SPARE.Ack_M550 := "M_ZERO";
END_REGION

REGION Network 142: M550- (READ-IN DISABLE) / M132-CENTRAL JAW CHUCK RELAX FIXTURE 1
   RUNG wire#powerrail
      Contact( "DB339_EXTENDED_M_SPARE".M_code[550] )
      wire#w1
      I_Contact( "DB371_M_UNIT_SPARE".M_CODES_SPARE.Ack_M550 )
      I_Contact( "DB2120_MPP_ITC_IPC".RESET_FAULTS )
      I_Contact( "DB371_M_UNIT_SPARE".M_CODES_SPARE.M_RESET_PULSE )
      Coil( "DB371_M_UNIT_SPARE".M_CODES_SPARE.M550 )
   END_RUNG
   RUNG wire#powerrail
      Contact( "DB371_M_UNIT_SPARE".M_CODES_SPARE.M550 )
   END_RUNG wire#w1
   // the same network as SCL:
   "DB371_M_UNIT_SPARE".M_CODES_SPARE.M550 := ("DB339_EXTENDED_M_SPARE".M_code[550] OR "DB371_M_UNIT_SPARE".M_CODES_SPARE.M550) AND NOT "DB371_M_UNIT_SPARE".M_CODES_SPARE.Ack_M550 AND NOT "DB2120_MPP_ITC_IPC".RESET_FAULTS AND NOT "DB371_M_UNIT_SPARE".M_CODES_SPARE.M_RESET_PULSE;
END_REGION

REGION Network 143: ACKNOWLEDGE M551- (READ-IN DISABLE) / ACKNOWLEDGE M133-CENTRAL JAW CHUCK CLAMP LOW FIXTURE 1
   RUNG wire#powerrail
      Contact( "M_ZERO" )
      Coil( "DB371_M_UNIT_SPARE".M_CODES_SPARE.Ack_M551 )
   END_RUNG
   // the same network as SCL:
   "DB371_M_UNIT_SPARE".M_CODES_SPARE.Ack_M551 := "M_ZERO";
END_REGION

REGION Network 144: M551- (READ-IN DISABLE) / M133-CENTRAL JAW CHUCK CLAMP LOW FIXTURE 1
   RUNG wire#powerrail
      Contact( "DB339_EXTENDED_M_SPARE".M_code[551] )
      wire#w1
      I_Contact( "DB371_M_UNIT_SPARE".M_CODES_SPARE.Ack_M551 )
      I_Contact( "DB2120_MPP_ITC_IPC".RESET_FAULTS )
      I_Contact( "DB371_M_UNIT_SPARE".M_CODES_SPARE.M_RESET_PULSE )
      Coil( "DB371_M_UNIT_SPARE".M_CODES_SPARE.M551 )
   END_RUNG
   RUNG wire#powerrail
      Contact( "DB371_M_UNIT_SPARE".M_CODES_SPARE.M551 )
   END_RUNG wire#w1
   // the same network as SCL:
   "DB371_M_UNIT_SPARE".M_CODES_SPARE.M551 := ("DB339_EXTENDED_M_SPARE".M_code[551] OR "DB371_M_UNIT_SPARE".M_CODES_SPARE.M551) AND NOT "DB371_M_UNIT_SPARE".M_CODES_SPARE.Ack_M551 AND NOT "DB2120_MPP_ITC_IPC".RESET_FAULTS AND NOT "DB371_M_UNIT_SPARE".M_CODES_SPARE.M_RESET_PULSE;
END_REGION

REGION Network 145: ACKNOWLEDGE M564- (READ-IN DISABLE) / ACKNOWLEDGE M162-JAW CHUCK PART B CLAMP FIXTURE 1
   RUNG wire#powerrail
      Contact( "M_ZERO" )
      Coil( "DB371_M_UNIT_SPARE".M_CODES_SPARE.Ack_M564 )
   END_RUNG
   // the same network as SCL:
   "DB371_M_UNIT_SPARE".M_CODES_SPARE.Ack_M564 := "M_ZERO";
END_REGION

REGION Network 146: M564- (READ-IN DISABLE) / M162-JAW CHUCK PART B CLAMP FIXTURE 1
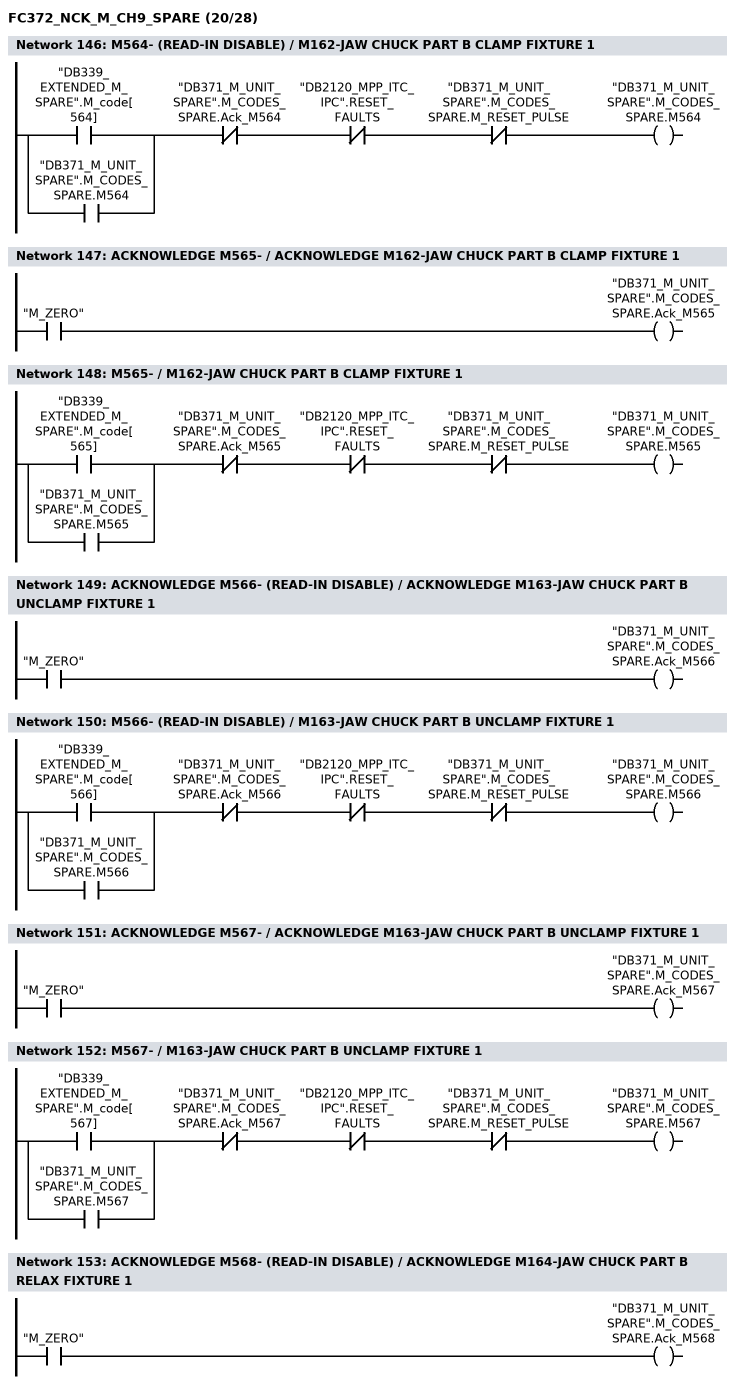
   RUNG wire#powerrail
      Contact( "DB339_EXTENDED_M_SPARE".M_code[564] )
      wire#w1
      I_Contact( "DB371_M_UNIT_SPARE".M_CODES_SPARE.Ack_M564 )
      I_Contact( "DB2120_MPP_ITC_IPC".RESET_FAULTS )
      I_Contact( "DB371_M_UNIT_SPARE".M_CODES_SPARE.M_RESET_PULSE )
      Coil( "DB371_M_UNIT_SPARE".M_CODES_SPARE.M564 )
   END_RUNG
   RUNG wire#powerrail
      Contact( "DB371_M_UNIT_SPARE".M_CODES_SPARE.M564 )
   END_RUNG wire#w1
   // the same network as SCL:
   "DB371_M_UNIT_SPARE".M_CODES_SPARE.M564 := ("DB339_EXTENDED_M_SPARE".M_code[564] OR "DB371_M_UNIT_SPARE".M_CODES_SPARE.M564) AND NOT "DB371_M_UNIT_SPARE".M_CODES_SPARE.Ack_M564 AND NOT "DB2120_MPP_ITC_IPC".RESET_FAULTS AND NOT "DB371_M_UNIT_SPARE".M_CODES_SPARE.M_RESET_PULSE;
END_REGION

REGION Network 147: ACKNOWLEDGE M565- / ACKNOWLEDGE M162-JAW CHUCK PART B CLAMP FIXTURE 1
   RUNG wire#powerrail
      Contact( "M_ZERO" )
      Coil( "DB371_M_UNIT_SPARE".M_CODES_SPARE.Ack_M565 )
   END_RUNG
   // the same network as SCL:
   "DB371_M_UNIT_SPARE".M_CODES_SPARE.Ack_M565 := "M_ZERO";
END_REGION

REGION Network 148: M565- / M162-JAW CHUCK PART B CLAMP FIXTURE 1
   RUNG wire#powerrail
      Contact( "DB339_EXTENDED_M_SPARE".M_code[565] )
      wire#w1
      I_Contact( "DB371_M_UNIT_SPARE".M_CODES_SPARE.Ack_M565 )
      I_Contact( "DB2120_MPP_ITC_IPC".RESET_FAULTS )
      I_Contact( "DB371_M_UNIT_SPARE".M_CODES_SPARE.M_RESET_PULSE )
      Coil( "DB371_M_UNIT_SPARE".M_CODES_SPARE.M565 )
   END_RUNG
   RUNG wire#powerrail
      Contact( "DB371_M_UNIT_SPARE".M_CODES_SPARE.M565 )
   END_RUNG wire#w1
   // the same network as SCL:
   "DB371_M_UNIT_SPARE".M_CODES_SPARE.M565 := ("DB339_EXTENDED_M_SPARE".M_code[565] OR "DB371_M_UNIT_SPARE".M_CODES_SPARE.M565) AND NOT "DB371_M_UNIT_SPARE".M_CODES_SPARE.Ack_M565 AND NOT "DB2120_MPP_ITC_IPC".RESET_FAULTS AND NOT "DB371_M_UNIT_SPARE".M_CODES_SPARE.M_RESET_PULSE;
END_REGION

REGION Network 149: ACKNOWLEDGE M566- (READ-IN DISABLE) / ACKNOWLEDGE M163-JAW CHUCK PART B UNCLAMP FIXTURE 1
   RUNG wire#powerrail
      Contact( "M_ZERO" )
      Coil( "DB371_M_UNIT_SPARE".M_CODES_SPARE.Ack_M566 )
   END_RUNG
   // the same network as SCL:
   "DB371_M_UNIT_SPARE".M_CODES_SPARE.Ack_M566 := "M_ZERO";
END_REGION

REGION Network 150: M566- (READ-IN DISABLE) / M163-JAW CHUCK PART B UNCLAMP FIXTURE 1
   RUNG wire#powerrail
      Contact( "DB339_EXTENDED_M_SPARE".M_code[566] )
      wire#w1
      I_Contact( "DB371_M_UNIT_SPARE".M_CODES_SPARE.Ack_M566 )
      I_Contact( "DB2120_MPP_ITC_IPC".RESET_FAULTS )
      I_Contact( "DB371_M_UNIT_SPARE".M_CODES_SPARE.M_RESET_PULSE )
      Coil( "DB371_M_UNIT_SPARE".M_CODES_SPARE.M566 )
   END_RUNG
   RUNG wire#powerrail
      Contact( "DB371_M_UNIT_SPARE".M_CODES_SPARE.M566 )
   END_RUNG wire#w1
   // the same network as SCL:
   "DB371_M_UNIT_SPARE".M_CODES_SPARE.M566 := ("DB339_EXTENDED_M_SPARE".M_code[566] OR "DB371_M_UNIT_SPARE".M_CODES_SPARE.M566) AND NOT "DB371_M_UNIT_SPARE".M_CODES_SPARE.Ack_M566 AND NOT "DB2120_MPP_ITC_IPC".RESET_FAULTS AND NOT "DB371_M_UNIT_SPARE".M_CODES_SPARE.M_RESET_PULSE;
END_REGION

REGION Network 151: ACKNOWLEDGE M567- / ACKNOWLEDGE M163-JAW CHUCK PART B UNCLAMP FIXTURE 1
   RUNG wire#powerrail
      Contact( "M_ZERO" )
      Coil( "DB371_M_UNIT_SPARE".M_CODES_SPARE.Ack_M567 )
   END_RUNG
   // the same network as SCL:
   "DB371_M_UNIT_SPARE".M_CODES_SPARE.Ack_M567 := "M_ZERO";
END_REGION

REGION Network 152: M567- / M163-JAW CHUCK PART B UNCLAMP FIXTURE 1
   RUNG wire#powerrail
      Contact( "DB339_EXTENDED_M_SPARE".M_code[567] )
      wire#w1
      I_Contact( "DB371_M_UNIT_SPARE".M_CODES_SPARE.Ack_M567 )
      I_Contact( "DB2120_MPP_ITC_IPC".RESET_FAULTS )
      I_Contact( "DB371_M_UNIT_SPARE".M_CODES_SPARE.M_RESET_PULSE )
      Coil( "DB371_M_UNIT_SPARE".M_CODES_SPARE.M567 )
   END_RUNG
   RUNG wire#powerrail
      Contact( "DB371_M_UNIT_SPARE".M_CODES_SPARE.M567 )
   END_RUNG wire#w1
   // the same network as SCL:
   "DB371_M_UNIT_SPARE".M_CODES_SPARE.M567 := ("DB339_EXTENDED_M_SPARE".M_code[567] OR "DB371_M_UNIT_SPARE".M_CODES_SPARE.M567) AND NOT "DB371_M_UNIT_SPARE".M_CODES_SPARE.Ack_M567 AND NOT "DB2120_MPP_ITC_IPC".RESET_FAULTS AND NOT "DB371_M_UNIT_SPARE".M_CODES_SPARE.M_RESET_PULSE;
END_REGION

REGION Network 153: ACKNOWLEDGE M568- (READ-IN DISABLE) / ACKNOWLEDGE M164-JAW CHUCK PART B RELAX FIXTURE 1
   RUNG wire#powerrail
      Contact( "M_ZERO" )
      Coil( "DB371_M_UNIT_SPARE".M_CODES_SPARE.Ack_M568 )
   END_RUNG
   // the same network as SCL:
   "DB371_M_UNIT_SPARE".M_CODES_SPARE.Ack_M568 := "M_ZERO";
END_REGION

REGION Network 154: M568- (READ-IN DISABLE) / M164-JAW CHUCK PART B RELAX FIXTURE 1
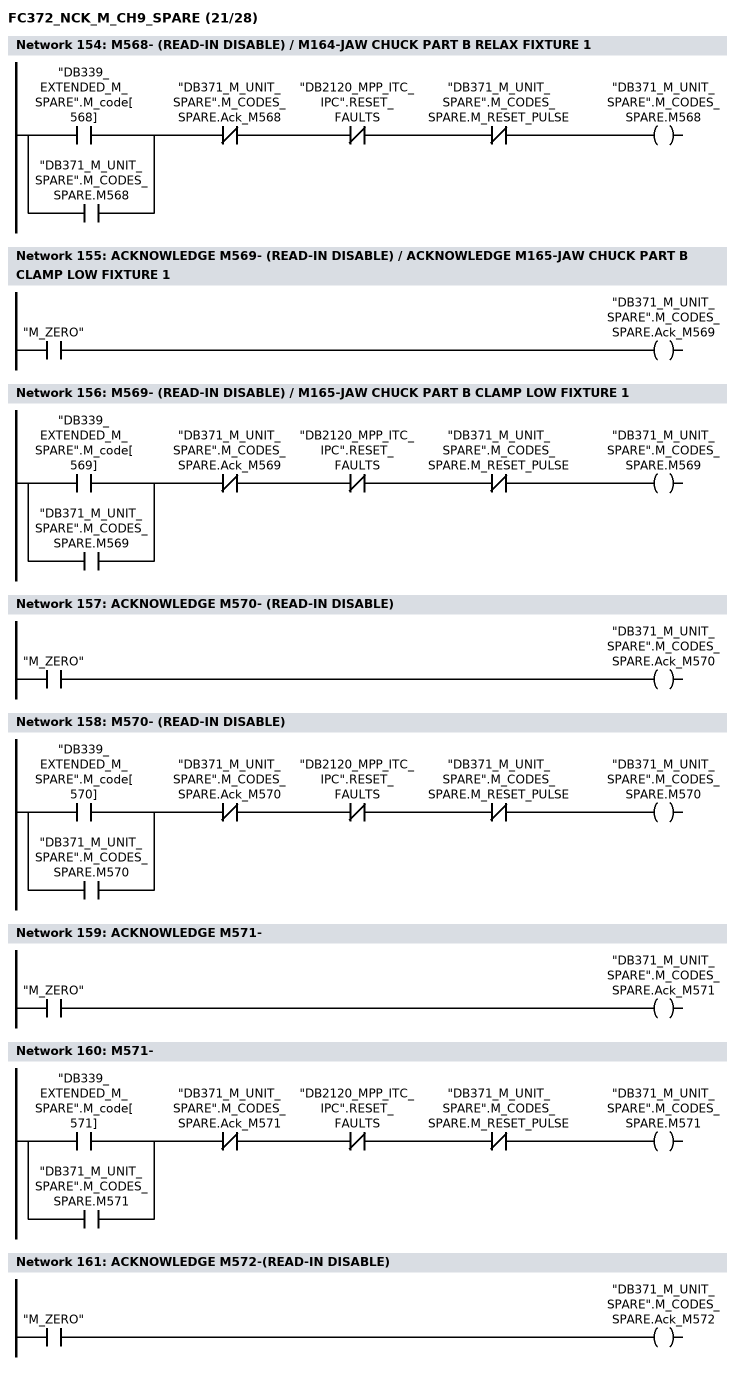
   RUNG wire#powerrail
      Contact( "DB339_EXTENDED_M_SPARE".M_code[568] )
      wire#w1
      I_Contact( "DB371_M_UNIT_SPARE".M_CODES_SPARE.Ack_M568 )
      I_Contact( "DB2120_MPP_ITC_IPC".RESET_FAULTS )
      I_Contact( "DB371_M_UNIT_SPARE".M_CODES_SPARE.M_RESET_PULSE )
      Coil( "DB371_M_UNIT_SPARE".M_CODES_SPARE.M568 )
   END_RUNG
   RUNG wire#powerrail
      Contact( "DB371_M_UNIT_SPARE".M_CODES_SPARE.M568 )
   END_RUNG wire#w1
   // the same network as SCL:
   "DB371_M_UNIT_SPARE".M_CODES_SPARE.M568 := ("DB339_EXTENDED_M_SPARE".M_code[568] OR "DB371_M_UNIT_SPARE".M_CODES_SPARE.M568) AND NOT "DB371_M_UNIT_SPARE".M_CODES_SPARE.Ack_M568 AND NOT "DB2120_MPP_ITC_IPC".RESET_FAULTS AND NOT "DB371_M_UNIT_SPARE".M_CODES_SPARE.M_RESET_PULSE;
END_REGION

REGION Network 155: ACKNOWLEDGE M569- (READ-IN DISABLE) / ACKNOWLEDGE M165-JAW CHUCK PART B CLAMP LOW FIXTURE 1
   RUNG wire#powerrail
      Contact( "M_ZERO" )
      Coil( "DB371_M_UNIT_SPARE".M_CODES_SPARE.Ack_M569 )
   END_RUNG
   // the same network as SCL:
   "DB371_M_UNIT_SPARE".M_CODES_SPARE.Ack_M569 := "M_ZERO";
END_REGION

REGION Network 156: M569- (READ-IN DISABLE) / M165-JAW CHUCK PART B CLAMP LOW FIXTURE 1
   RUNG wire#powerrail
      Contact( "DB339_EXTENDED_M_SPARE".M_code[569] )
      wire#w1
      I_Contact( "DB371_M_UNIT_SPARE".M_CODES_SPARE.Ack_M569 )
      I_Contact( "DB2120_MPP_ITC_IPC".RESET_FAULTS )
      I_Contact( "DB371_M_UNIT_SPARE".M_CODES_SPARE.M_RESET_PULSE )
      Coil( "DB371_M_UNIT_SPARE".M_CODES_SPARE.M569 )
   END_RUNG
   RUNG wire#powerrail
      Contact( "DB371_M_UNIT_SPARE".M_CODES_SPARE.M569 )
   END_RUNG wire#w1
   // the same network as SCL:
   "DB371_M_UNIT_SPARE".M_CODES_SPARE.M569 := ("DB339_EXTENDED_M_SPARE".M_code[569] OR "DB371_M_UNIT_SPARE".M_CODES_SPARE.M569) AND NOT "DB371_M_UNIT_SPARE".M_CODES_SPARE.Ack_M569 AND NOT "DB2120_MPP_ITC_IPC".RESET_FAULTS AND NOT "DB371_M_UNIT_SPARE".M_CODES_SPARE.M_RESET_PULSE;
END_REGION

REGION Network 157: ACKNOWLEDGE M570- (READ-IN DISABLE)
   RUNG wire#powerrail
      Contact( "M_ZERO" )
      Coil( "DB371_M_UNIT_SPARE".M_CODES_SPARE.Ack_M570 )
   END_RUNG
   // the same network as SCL:
   "DB371_M_UNIT_SPARE".M_CODES_SPARE.Ack_M570 := "M_ZERO";
END_REGION

REGION Network 158: M570- (READ-IN DISABLE)
   RUNG wire#powerrail
      Contact( "DB339_EXTENDED_M_SPARE".M_code[570] )
      wire#w1
      I_Contact( "DB371_M_UNIT_SPARE".M_CODES_SPARE.Ack_M570 )
      I_Contact( "DB2120_MPP_ITC_IPC".RESET_FAULTS )
      I_Contact( "DB371_M_UNIT_SPARE".M_CODES_SPARE.M_RESET_PULSE )
      Coil( "DB371_M_UNIT_SPARE".M_CODES_SPARE.M570 )
   END_RUNG
   RUNG wire#powerrail
      Contact( "DB371_M_UNIT_SPARE".M_CODES_SPARE.M570 )
   END_RUNG wire#w1
   // the same network as SCL:
   "DB371_M_UNIT_SPARE".M_CODES_SPARE.M570 := ("DB339_EXTENDED_M_SPARE".M_code[570] OR "DB371_M_UNIT_SPARE".M_CODES_SPARE.M570) AND NOT "DB371_M_UNIT_SPARE".M_CODES_SPARE.Ack_M570 AND NOT "DB2120_MPP_ITC_IPC".RESET_FAULTS AND NOT "DB371_M_UNIT_SPARE".M_CODES_SPARE.M_RESET_PULSE;
END_REGION

REGION Network 159: ACKNOWLEDGE M571-
   RUNG wire#powerrail
      Contact( "M_ZERO" )
      Coil( "DB371_M_UNIT_SPARE".M_CODES_SPARE.Ack_M571 )
   END_RUNG
   // the same network as SCL:
   "DB371_M_UNIT_SPARE".M_CODES_SPARE.Ack_M571 := "M_ZERO";
END_REGION

REGION Network 160: M571-
   RUNG wire#powerrail
      Contact( "DB339_EXTENDED_M_SPARE".M_code[571] )
      wire#w1
      I_Contact( "DB371_M_UNIT_SPARE".M_CODES_SPARE.Ack_M571 )
      I_Contact( "DB2120_MPP_ITC_IPC".RESET_FAULTS )
      I_Contact( "DB371_M_UNIT_SPARE".M_CODES_SPARE.M_RESET_PULSE )
      Coil( "DB371_M_UNIT_SPARE".M_CODES_SPARE.M571 )
   END_RUNG
   RUNG wire#powerrail
      Contact( "DB371_M_UNIT_SPARE".M_CODES_SPARE.M571 )
   END_RUNG wire#w1
   // the same network as SCL:
   "DB371_M_UNIT_SPARE".M_CODES_SPARE.M571 := ("DB339_EXTENDED_M_SPARE".M_code[571] OR "DB371_M_UNIT_SPARE".M_CODES_SPARE.M571) AND NOT "DB371_M_UNIT_SPARE".M_CODES_SPARE.Ack_M571 AND NOT "DB2120_MPP_ITC_IPC".RESET_FAULTS AND NOT "DB371_M_UNIT_SPARE".M_CODES_SPARE.M_RESET_PULSE;
END_REGION

REGION Network 161: ACKNOWLEDGE M572-(READ-IN DISABLE)
   RUNG wire#powerrail
      Contact( "M_ZERO" )
      Coil( "DB371_M_UNIT_SPARE".M_CODES_SPARE.Ack_M572 )
   END_RUNG
   // the same network as SCL:
   "DB371_M_UNIT_SPARE".M_CODES_SPARE.Ack_M572 := "M_ZERO";
END_REGION

REGION Network 162: M572-(READ-IN DISABLE)
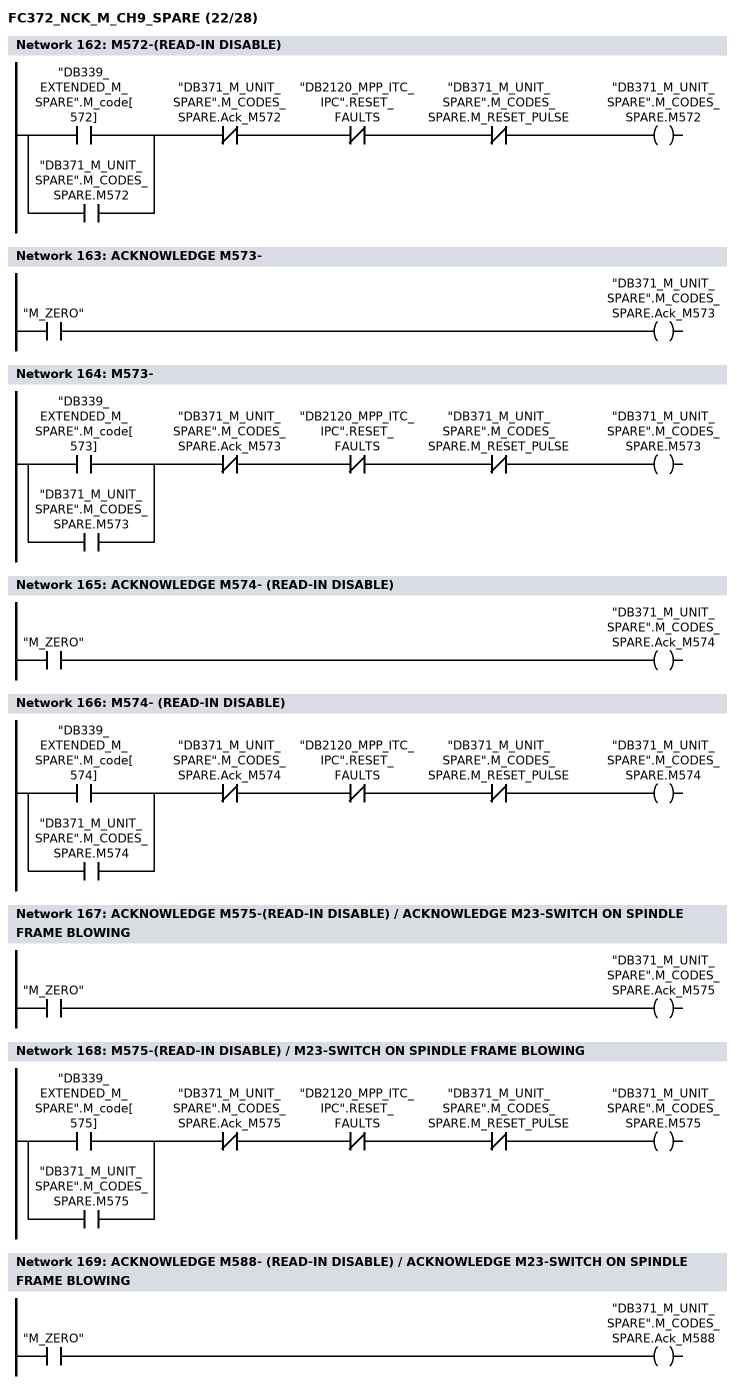
   RUNG wire#powerrail
      Contact( "DB339_EXTENDED_M_SPARE".M_code[572] )
      wire#w1
      I_Contact( "DB371_M_UNIT_SPARE".M_CODES_SPARE.Ack_M572 )
      I_Contact( "DB2120_MPP_ITC_IPC".RESET_FAULTS )
      I_Contact( "DB371_M_UNIT_SPARE".M_CODES_SPARE.M_RESET_PULSE )
      Coil( "DB371_M_UNIT_SPARE".M_CODES_SPARE.M572 )
   END_RUNG
   RUNG wire#powerrail
      Contact( "DB371_M_UNIT_SPARE".M_CODES_SPARE.M572 )
   END_RUNG wire#w1
   // the same network as SCL:
   "DB371_M_UNIT_SPARE".M_CODES_SPARE.M572 := ("DB339_EXTENDED_M_SPARE".M_code[572] OR "DB371_M_UNIT_SPARE".M_CODES_SPARE.M572) AND NOT "DB371_M_UNIT_SPARE".M_CODES_SPARE.Ack_M572 AND NOT "DB2120_MPP_ITC_IPC".RESET_FAULTS AND NOT "DB371_M_UNIT_SPARE".M_CODES_SPARE.M_RESET_PULSE;
END_REGION

REGION Network 163: ACKNOWLEDGE M573-
   RUNG wire#powerrail
      Contact( "M_ZERO" )
      Coil( "DB371_M_UNIT_SPARE".M_CODES_SPARE.Ack_M573 )
   END_RUNG
   // the same network as SCL:
   "DB371_M_UNIT_SPARE".M_CODES_SPARE.Ack_M573 := "M_ZERO";
END_REGION

